D7115 CHANNEL  ; 热压C下层Hip测试气缸下降位延时设置
D7116 CHANNEL  ; 热压C上层有料感应延时设置
D7117 CHANNEL  ; 热压C下层有料感应延时设置
D7118 CHANNEL  ; #REF!
D7119 CHANNEL  ; #REF!
D7120 CHANNEL  ; 热压C上层极耳检查输入延时设置
D7121 CHANNEL  ; 热压C下层极耳检查输入延时设置
D7122 CHANNEL  ; 进出料转移伺服准备好延时设置
D7123 CHANNEL  ; 进出料转移伺服报警延时设置
D7124 CHANNEL  ; 伸缩伺服准备好延时设置
D7125 CHANNEL  ; 伸缩伺服报警延时设置
D7126 CHANNEL  ; #REF!
D7127 CHANNEL  ; 备用11延时设置
D7128 CHANNEL  ; 加热A跳闸延时设置
D7129 CHANNEL  ; 加热B跳闸延时设置
D7130 CHANNEL  ; 加热C跳闸延时设置
D7131 CHANNEL  ; 副PLC 0.03延时设置
D7132 CHANNEL  ; 副PLC 0.04延时设置
D7133 CHANNEL  ; 副PLC 0.05延时设置
D7134 CHANNEL  ; 副PLC 0.06延时设置
D7135 CHANNEL  ; 副PLC 0.07延时设置
D7136 CHANNEL  ; 副PLC 0.08延时设置
D7137 CHANNEL  ; 副PLC 0.09延时设置
D7138 CHANNEL  ; 副PLC 0.10延时设置
D7139 CHANNEL  ; 副PLC 0.11延时设置
D7140 CHANNEL  ; 延时设置
D7141 CHANNEL  ; 延时设置
D7142 CHANNEL  ; 延时设置
D7143 CHANNEL  ; 延时设置
D7144 CHANNEL  ; 副PLC 1.00延时设置
D7145 CHANNEL  ; 副PLC 1.01延时设置
D7146 CHANNEL  ; 副PLC 1.02延时设置
D7147 CHANNEL  ; 副PLC 1.03延时设置
D7148 CHANNEL  ; 副PLC 1.04延时设置
D7149 CHANNEL  ; 副PLC 1.05延时设置
D7150 CHANNEL  ; 副PLC 1.06延时设置
D7151 CHANNEL  ; 副PLC 1.07延时设置
D7152 CHANNEL  ; 副PLC 1.08延时设置
D7153 CHANNEL  ; 副PLC 1.09延时设置
D7154 CHANNEL  ; 副PLC 1.10延时设置
D7155 CHANNEL  ; 副PLC 1.11延时设置
D7156 CHANNEL  ; 延时设置
D7157 CHANNEL  ; 延时设置
D7158 CHANNEL  ; 延时设置
D7159 CHANNEL  ; 延时设置
D7160 CHANNEL  ; 延时设置
D7161 CHANNEL  ; 出料转移机构A上升位延时设置
D7162 CHANNEL  ; 出料转移夹爪A下降位延时设置
D7163 CHANNEL  ; 出料转移夹爪A上升位延时设置
D7164 CHANNEL  ; 出料转移夹爪A1松开位延时设置
D7165 CHANNEL  ; 出料转移夹爪A1夹紧位延时设置
D7166 CHANNEL  ; 出料转移夹爪A2松开位延时设置
D7167 CHANNEL  ; 出料转移夹爪A2夹紧位延时设置
D7168 CHANNEL  ; 出料转移夹爪A3松开位延时设置
D7169 CHANNEL  ; 出料转移夹爪A3夹紧位延时设置
D7170 CHANNEL  ; 出料转移夹爪A4松开位延时设置
D7171 CHANNEL  ; 出料转移夹爪A4夹紧位延时设置
D7174 CHANNEL  ; 出料转移夹爪A1左托起张开位延时设置
D7175 CHANNEL  ; 出料转移夹爪A1左托起托起位延时设置
D7176 CHANNEL  ; 出料转移夹爪A1右托起张开位延时设置
D7177 CHANNEL  ; 出料转移夹爪A1右托起托起位延时设置
D7178 CHANNEL  ; 出料转移夹爪A2左托起张开位延时设置
D7179 CHANNEL  ; 出料转移夹爪A2左托起托起位延时设置
D7180 CHANNEL  ; 出料转移夹爪A2右托起张开位延时设置
D7181 CHANNEL  ; 出料转移夹爪A2右托起托起位延时设置
D7182 CHANNEL  ; 出料转移夹爪A3左托起张开位延时设置
D7183 CHANNEL  ; 出料转移夹爪A3左托起托起位延时设置
D7184 CHANNEL  ; 出料转移夹爪A3右托起张开位延时设置
D7185 CHANNEL  ; 出料转移夹爪A3右托起托起位延时设置
D7186 CHANNEL  ; 出料转移夹爪A4左托起张开位延时设置
D7187 CHANNEL  ; 出料转移夹爪A4左托起托起位延时设置
D7188 CHANNEL  ; 出料转移夹爪A4右托起张开位延时设置
D7189 CHANNEL  ; 出料转移夹爪A4右托起托起位延时设置
D7194 CHANNEL  ; 出料转移夹爪A1真空延时设置
D7195 CHANNEL  ; 出料转移夹爪A2真空延时设置
D7196 CHANNEL  ; 出料转移夹爪A3真空延时设置
D7197 CHANNEL  ; 出料转移夹爪A4真空延时设置
D7199 CHANNEL  ; 进料转移机构B下降位延时设置
D7200 CHANNEL  ; 进料转移机构B上升位延时设置
D7201 CHANNEL  ; 进料转移夹爪B下降位延时设置
D7202 CHANNEL  ; 进料转移夹爪B上升位延时设置
D7203 CHANNEL  ; 进料转移夹爪B1松开位延时设置
D7204 CHANNEL  ; 进料转移夹爪B1夹紧位延时设置
D7205 CHANNEL  ; 进料转移夹爪B2松开位延时设置
D7206 CHANNEL  ; 进料转移夹爪B2夹紧位延时设置
D7207 CHANNEL  ; 进料转移夹爪B3松开位延时设置
D7208 CHANNEL  ; 进料转移夹爪B3夹紧位延时设置
D7209 CHANNEL  ; 进料转移夹爪B4松开位延时设置
D7210 CHANNEL  ; 进料转移夹爪B4夹紧位延时设置
D7213 CHANNEL  ; 进料转移爪B1左上升位延时设置
D7214 CHANNEL  ; 进料转移爪B1右上升位延时设置
D7215 CHANNEL  ; 进料转移爪B2左上升位延时设置
D7216 CHANNEL  ; 进料转移爪B2右上升位延时设置
D7217 CHANNEL  ; 进料转移爪B3左上升位延时设置
D7218 CHANNEL  ; 进料转移爪B3右上升位延时设置
D7219 CHANNEL  ; 进料转移爪B4左上升位延时设置
D7220 CHANNEL  ; 进料转移爪B4右上升位延时设置
D7223 CHANNEL  ; 进料转移爪B1中间上升位延时设置
D7224 CHANNEL  ; 进料转移爪B2中间上升位延时设置
D7225 CHANNEL  ; 进料转移爪B3中间上升位延时设置
D7226 CHANNEL  ; 进料转移爪B4中间上升位延时设置
D7228 CHANNEL  ; 进料转移爪B1有料反射延时设置
D7229 CHANNEL  ; 进料转移爪B2有料反射延时设置
D7230 CHANNEL  ; 进料转移爪B3有料反射延时设置
D7231 CHANNEL  ; 进料转移爪B4有料反射延时设置
D7233 CHANNEL  ; 出料转移机构B下降位延时设置
D7234 CHANNEL  ; 出料转移机构B上升位延时设置
D7235 CHANNEL  ; 出料转移夹爪B下降位延时设置
D7236 CHANNEL  ; 出料转移夹爪B上升位延时设置
D7237 CHANNEL  ; 出料转移夹爪B1松开位延时设置
D7238 CHANNEL  ; 出料转移夹爪B1夹紧位延时设置
D7239 CHANNEL  ; 出料转移夹爪B2松开位延时设置
D7240 CHANNEL  ; 出料转移夹爪B2夹紧位延时设置
D7241 CHANNEL  ; 出料转移夹爪B3松开位延时设置
D7242 CHANNEL  ; 出料转移夹爪B3夹紧位延时设置
D7243 CHANNEL  ; 出料转移夹爪B4松开位延时设置
D7244 CHANNEL  ; 出料转移夹爪B4夹紧位延时设置
D7247 CHANNEL  ; 出料转移夹爪B1左托起张开位延时设置
D7248 CHANNEL  ; 出料转移夹爪B1左托起托起位延时设置
D7249 CHANNEL  ; 出料转移夹爪B1右托起张开位延时设置
D7250 CHANNEL  ; 出料转移夹爪B1右托起托起位延时设置
D7251 CHANNEL  ; 出料转移夹爪B2左托起张开位延时设置
D7252 CHANNEL  ; 出料转移夹爪B2左托起托起位延时设置
D7253 CHANNEL  ; 出料转移夹爪B2右托起张开位延时设置
D7254 CHANNEL  ; 出料转移夹爪B2右托起托起位延时设置
D7255 CHANNEL  ; 出料转移夹爪B3左托起张开位延时设置
D7256 CHANNEL  ; 出料转移夹爪B3左托起托起位延时设置
D7257 CHANNEL  ; 出料转移夹爪B3右托起张开位延时设置
D7258 CHANNEL  ; 出料转移夹爪B3右托起托起位延时设置
D7259 CHANNEL  ; 出料转移夹爪B4左托起张开位延时设置
D7260 CHANNEL  ; 出料转移夹爪B4左托起托起位延时设置
D7261 CHANNEL  ; 出料转移夹爪B4右托起张开位延时设置
D7262 CHANNEL  ; 出料转移夹爪B4右托起托起位延时设置
D7267 CHANNEL  ; 出料转移夹爪B1真空延时设置
D7268 CHANNEL  ; 出料转移夹爪B2真空延时设置
D7269 CHANNEL  ; 出料转移夹爪B3真空延时设置
D7270 CHANNEL  ; 出料转移夹爪B4真空延时设置
D7272 CHANNEL  ; 热压A1层加热开关延时设置
D7273 CHANNEL  ; 热压A2层加热开关延时设置
D7274 CHANNEL  ; 热压A3层加热开关延时设置
D7275 CHANNEL  ; 热压A4层加热开关延时设置
D7276 CHANNEL  ; 热压A5层加热开关延时设置
D7277 CHANNEL  ; 热压A1下压板A侧位置延时设置
D7278 CHANNEL  ; 热压A1下压板B侧位置延时设置
D7281 CHANNEL  ; 热压A3下压板A侧位置延时设置
D7282 CHANNEL  ; 热压A3下压板B侧位置延时设置
D7283 CHANNEL  ; 热压A4下压板A侧位置延时设置
D7284 CHANNEL  ; 热压A4下压板B侧位置延时设置
D7285 CHANNEL  ; 热压A5下压板A侧位置延时设置
D7286 CHANNEL  ; 热压A5下压板B侧位置延时设置
D7287 CHANNEL  ; 热压A1有料对射延时设置
D7288 CHANNEL  ; 热压A2有料对射延时设置
D7289 CHANNEL  ; 热压A3有料对射延时设置
D7290 CHANNEL  ; 热压A4有料对射延时设置
D7291 CHANNEL  ; 热压A5有料对射延时设置
D7292 CHANNEL  ; 热压A上预压平移气缸等待位延时设置
D7293 CHANNEL  ; 热压A上预压平移气缸预压位延时设置
D7294 CHANNEL  ; 热压A下预压平移气缸等待位延时设置
D7295 CHANNEL  ; 热压A下预压平移气缸预压位延时设置
D7296 CHANNEL  ; 热压A垫高气缸移出位延时设置
D7297 CHANNEL  ; 热压A垫高气缸热压位延时设置
D7298 CHANNEL  ; 热压A1HIP测试上升位延时设置
D7299 CHANNEL  ; 热压A1HIP测试下降位延时设置
D7300 CHANNEL  ; 热压A2HIP测试上升位延时设置
D7301 CHANNEL  ; 热压A2HIP测试下降位延时设置
D7302 CHANNEL  ; 热压A3HIP测试上升位延时设置
D7303 CHANNEL  ; 热压A3HIP测试下降位延时设置
D7304 CHANNEL  ; 热压A4HIP测试上升位延时设置
D7305 CHANNEL  ; 热压A4HIP测试下降位延时设置
D7306 CHANNEL  ; 热压A5HIP测试上升位延时设置
D7307 CHANNEL  ; 热压A5HIP测试下降位延时设置
D7308 CHANNEL  ; 热压A1顶升气缸缩回位延时设置
D7309 CHANNEL  ; 热压A1顶升气缸伸出位延时设置
D7310 CHANNEL  ; 热压A2顶升气缸左缩回位延时设置
D7311 CHANNEL  ; 热压A2顶升气缸左伸出位延时设置
D7312 CHANNEL  ; 热压A2顶升气缸右缩回位延时设置
D7313 CHANNEL  ; 热压A2顶升气缸右伸出位延时设置
D7314 CHANNEL  ; 热压A3顶升气缸左缩回位延时设置
D7315 CHANNEL  ; 热压A3顶升气缸左伸出位延时设置
D7316 CHANNEL  ; 热压A3顶升气缸右缩回位延时设置
D7317 CHANNEL  ; 热压A3顶升气缸右伸出位延时设置
D7318 CHANNEL  ; 热压A4顶升气缸左缩回位延时设置
D7319 CHANNEL  ; 热压A4顶升气缸左伸出位延时设置
D7320 CHANNEL  ; 热压A4顶升气缸右缩回位延时设置
D7321 CHANNEL  ; 热压A4顶升气缸右伸出位延时设置
D7322 CHANNEL  ; 热压A5顶升气缸左缩回位延时设置
D7323 CHANNEL  ; 热压A5顶升气缸左伸出位延时设置
D7324 CHANNEL  ; 热压A5顶升气缸右缩回位延时设置
D7325 CHANNEL  ; 热压A5顶升气缸右伸出位延时设置
D7326 CHANNEL  ; 热压B1层加热开关延时设置
D7327 CHANNEL  ; 热压B2层加热开关延时设置
D7328 CHANNEL  ; 热压B3层加热开关延时设置
D7329 CHANNEL  ; 热压B4层加热开关延时设置
D7330 CHANNEL  ; 热压B5层加热开关延时设置
D7331 CHANNEL  ; 热压B1下压板A侧位置延时设置
D7332 CHANNEL  ; 热压B1下压板B侧位置延时设置
D7333 CHANNEL  ; 热压B2下压板A侧位置延时设置
D7334 CHANNEL  ; 热压B2下压板B侧位置延时设置
D7335 CHANNEL  ; 热压B3下压板A侧位置延时设置
D7336 CHANNEL  ; 热压B3下压板B侧位置延时设置
D7337 CHANNEL  ; 热压B4下压板A侧位置延时设置
D7338 CHANNEL  ; 热压B4下压板B侧位置延时设置
D7339 CHANNEL  ; 热压B5下压板A侧位置延时设置
D7340 CHANNEL  ; 热压B5下压板B侧位置延时设置
D7341 CHANNEL  ; 热压B1有料对射延时设置
D7342 CHANNEL  ; 热压B2有料对射延时设置
D7343 CHANNEL  ; 热压B3有料对射延时设置
D7344 CHANNEL  ; 热压B4有料对射延时设置
D7345 CHANNEL  ; 热压B5有料对射延时设置
D7346 CHANNEL  ; 热压B上预压平移气缸等待位延时设置
D7347 CHANNEL  ; 热压B上预压平移气缸预压位延时设置
D7348 CHANNEL  ; 热压B下预压平移气缸等待位延时设置
D7349 CHANNEL  ; 热压B下预压平移气缸预压位延时设置
D7350 CHANNEL  ; 热压B垫高气缸移出位延时设置
D7351 CHANNEL  ; 热压B垫高气缸热压位延时设置
D7352 CHANNEL  ; 热压B1HIP测试上升位延时设置
D7353 CHANNEL  ; 热压B1HIP测试下降位延时设置
D7354 CHANNEL  ; 热压B2HIP测试上升位延时设置
D7355 CHANNEL  ; 热压B2HIP测试下降位延时设置
D7356 CHANNEL  ; 热压B3HIP测试上升位延时设置
D7357 CHANNEL  ; 热压B3HIP测试下降位延时设置
D7358 CHANNEL  ; 热压B4HIP测试上升位延时设置
D7359 CHANNEL  ; 热压B4HIP测试下降位延时设置
D7360 CHANNEL  ; 热压B5HIP测试上升位延时设置
D7361 CHANNEL  ; 热压B5HIP测试下降位延时设置
D7362 CHANNEL  ; 热压B1顶升气缸缩回位延时设置
D7363 CHANNEL  ; 热压B1顶升气缸伸出位延时设置
D7364 CHANNEL  ; 热压B2顶升气缸左缩回位延时设置
D7365 CHANNEL  ; 热压B2顶升气缸左伸出位延时设置
D7366 CHANNEL  ; 热压B2顶升气缸右缩回位延时设置
D7367 CHANNEL  ; 热压B2顶升气缸右伸出位延时设置
D7368 CHANNEL  ; 热压B3顶升气缸左缩回位延时设置
D7369 CHANNEL  ; 热压B3顶升气缸左伸出位延时设置
D7370 CHANNEL  ; 热压B3顶升气缸右缩回位延时设置
D7371 CHANNEL  ; 热压B3顶升气缸右伸出位延时设置
D7372 CHANNEL  ; 热压B4顶升气缸左缩回位延时设置
D7373 CHANNEL  ; 热压B4顶升气缸左伸出位延时设置
D7374 CHANNEL  ; 热压B4顶升气缸右缩回位延时设置
D7375 CHANNEL  ; 热压B4顶升气缸右伸出位延时设置
D7376 CHANNEL  ; 热压B5顶升气缸左缩回位延时设置
D7377 CHANNEL  ; 热压B5顶升气缸左伸出位延时设置
D7378 CHANNEL  ; 热压B5顶升气缸右缩回位延时设置
D7379 CHANNEL  ; 热压B5顶升气缸右伸出位延时设置
D7380 CHANNEL  ; 下料定位A下降位延时设置
D7381 CHANNEL  ; 下料定位A上升位延时设置
D7382 CHANNEL  ; 下料定位A水平位延时设置
D7383 CHANNEL  ; 下料定位A垂直位延时设置
D7384 CHANNEL  ; 下料定位A1左右松开位延时设置
D7385 CHANNEL  ; 下料定位A1左右夹紧位延时设置
D7386 CHANNEL  ; 下料定位A2左右松开位延时设置
D7387 CHANNEL  ; 下料定位A2左右夹紧位延时设置
D7388 CHANNEL  ; 下料定位A3左右松开位延时设置
D7389 CHANNEL  ; 下料定位A3左右夹紧位延时设置
D7390 CHANNEL  ; 下料定位A4左右松开位延时设置
D7391 CHANNEL  ; 下料定位A4左右夹紧位延时设置
D7394 CHANNEL  ; 下料定位A1前后松开位延时设置
D7395 CHANNEL  ; 下料定位A1前后夹紧位延时设置
D7396 CHANNEL  ; 下料定位A2前后松开位延时设置
D7397 CHANNEL  ; 下料定位A2前后夹紧位延时设置
D7398 CHANNEL  ; 下料定位A3前后松开位延时设置
D7399 CHANNEL  ; 下料定位A3前后夹紧位延时设置
D7400 CHANNEL  ; 下料定位A4前后松开位延时设置
D7401 CHANNEL  ; 下料定位A4前后夹紧位延时设置
D7404 CHANNEL  ; 下料定位A1有料感应延时设置
D7405 CHANNEL  ; 下料定位A2有料感应延时设置
D7406 CHANNEL  ; 下料定位A3有料感应延时设置
D7407 CHANNEL  ; 下料定位A4有料感应延时设置
D7409 CHANNEL  ; 下料定位A料平整检测（预留）延时设置
D7410 CHANNEL  ; 下料定位B下降位延时设置
D7411 CHANNEL  ; 下料定位B上升位延时设置
D7412 CHANNEL  ; 下料定位B水平位延时设置
D7413 CHANNEL  ; 下料定位B垂直位延时设置
D7414 CHANNEL  ; 下料定位B1左右松开位延时设置
D7415 CHANNEL  ; 下料定位B1左右夹紧位延时设置
D7416 CHANNEL  ; 下料定位B2左右松开位延时设置
D7417 CHANNEL  ; 下料定位B2左右夹紧位延时设置
D7418 CHANNEL  ; 下料定位B3左右松开位延时设置
D7419 CHANNEL  ; 下料定位B3左右夹紧位延时设置
D7420 CHANNEL  ; 下料定位B4左右松开位延时设置
D7421 CHANNEL  ; 下料定位B4左右夹紧位延时设置
D7424 CHANNEL  ; 下料定位B1前后松开位延时设置
D7425 CHANNEL  ; 下料定位B1前后夹紧位延时设置
D7426 CHANNEL  ; 下料定位B2前后松开位延时设置
D7427 CHANNEL  ; 下料定位B2前后夹紧位延时设置
D7428 CHANNEL  ; 下料定位B3前后松开位延时设置
D7429 CHANNEL  ; 下料定位B3前后夹紧位延时设置
D7430 CHANNEL  ; 下料定位B4前后松开位延时设置
D7431 CHANNEL  ; 下料定位B4前后夹紧位延时设置
D7434 CHANNEL  ; 下料定位B1有料感应延时设置
D7435 CHANNEL  ; 下料定位B2有料感应延时设置
D7436 CHANNEL  ; 下料定位B3有料感应延时设置
D7437 CHANNEL  ; 下料定位B4有料感应延时设置
D7439 CHANNEL  ; 下料定位B料平整检测（预留）延时设置
D7440 CHANNEL  ; R2左夹紧气缸1松开位延时设置
D7441 CHANNEL  ; R2左夹紧气缸1夹紧位延时设置
D7442 CHANNEL  ; R2右夹紧气缸1松开位延时设置
D7443 CHANNEL  ; R2右夹紧气缸1夹紧位延时设置
D7444 CHANNEL  ; R2左夹紧气缸2松开位延时设置
D7445 CHANNEL  ; R2左夹紧气缸2夹紧位延时设置
D7446 CHANNEL  ; R2右夹紧气缸2松开位延时设置
D7447 CHANNEL  ; R2右夹紧气缸2夹紧位延时设置
D7448 CHANNEL  ; R2左夹紧气缸3松开位延时设置
D7449 CHANNEL  ; R2左夹紧气缸3夹紧位延时设置
D7450 CHANNEL  ; R2右夹紧气缸3松开位延时设置
D7451 CHANNEL  ; R2右夹紧气缸3夹紧位延时设置
D7452 CHANNEL  ; R2左夹紧气缸4松开位延时设置
D7453 CHANNEL  ; R2左夹紧气缸4夹紧位延时设置
D7454 CHANNEL  ; R2右夹紧气缸4松开位延时设置
D7455 CHANNEL  ; R2右夹紧气缸4夹紧位延时设置
D7460 CHANNEL  ; R2左压紧1上升位延时设置
D7461 CHANNEL  ; R2右压紧1上升位延时设置
D7462 CHANNEL  ; R2左压紧2上升位延时设置
D7463 CHANNEL  ; R2右压紧2上升位延时设置
D7464 CHANNEL  ; R2左压紧3上升位延时设置
D7465 CHANNEL  ; R2右压紧3上升位延时设置
D7466 CHANNEL  ; R2左压紧4上升位延时设置
D7467 CHANNEL  ; R2右压紧4上升位延时设置
D7470 CHANNEL  ; R2有料反射光电感应1延时设置
D7471 CHANNEL  ; R2有料反射光电感应2延时设置
D7472 CHANNEL  ; R2有料反射光电感应3延时设置
D7473 CHANNEL  ; R2有料反射光电感应4延时设置
D7475 CHANNEL  ; R2下料柔性报警1延时设置
D7476 CHANNEL  ; R2下料柔性报警2延时设置
D7477 CHANNEL  ; R2下料柔性报警3延时设置
D7478 CHANNEL  ; R2下料柔性报警4延时设置
D7480 CHANNEL  ; 下料R程序运行过程中延时设置
D7481 CHANNEL  ; 下料R程序复位中延时设置
D7482 CHANNEL  ; 下料R报警中延时设置
D7483 CHANNEL  ; 下料R位置辅助1延时设置
D7484 CHANNEL  ; 下料R位置辅助2延时设置
D7486 CHANNEL  ; 下料R位置辅助4延时设置
D7492 CHANNEL  ; 接料治具有料反射1延时设置
D7493 CHANNEL  ; 接料治具有料反射2延时设置
D7494 CHANNEL  ; 接料治具有料反射3延时设置
D7495 CHANNEL  ; 接料治具有料反射4延时设置
D7496 CHANNEL  ; 接料治具有料反射5延时设置
D7497 CHANNEL  ; 接料治具有料反射6延时设置
D7498 CHANNEL  ; 接料治具有料反射7延时设置
D7499 CHANNEL  ; 接料治具有料反射8延时设置
D7500 CHANNEL  ; 扫码NG有料对射光电1延时设置
D7501 CHANNEL  ; 扫码NG有料对射光电2延时设置
D7502 CHANNEL  ; 扫码NG有料对射光电3延时设置
D7503 CHANNEL  ; 扫码NG有料对射光电4延时设置
D7505 CHANNEL  ; 扫码NG满料对射光电延时设置
D7506 CHANNEL  ; 扫码NG拉带接近1延时设置
D7507 CHANNEL  ; 扫码NG拉带接近2延时设置
D7508 CHANNEL  ; HIPNG有料对射光电1延时设置
D7509 CHANNEL  ; HIPNG有料对射光电2延时设置
D7510 CHANNEL  ; HIPNG有料对射光电3延时设置
D7511 CHANNEL  ; HIPNG有料对射光电4延时设置
D7512 CHANNEL  ; HIPNG有料对射光电5延时设置
D7513 CHANNEL  ; HIPNG满料对射光电延时设置
D7514 CHANNEL  ; HIPNG拉带接近1延时设置
D7515 CHANNEL  ; HIPNG拉带接近2延时设置
D7516 CHANNEL  ; HIPNG有料对射光电1延时设置
D7517 CHANNEL  ; 工艺NG有料对射光电2延时设置
D7518 CHANNEL  ; 工艺NG有料对射光电3延时设置
D7519 CHANNEL  ; 工艺NG有料对射光电4延时设置
D7520 CHANNEL  ; 工艺NG有料对射光电5延时设置
D7521 CHANNEL  ; 工艺NG满料对射光电延时设置
D7522 CHANNEL  ; 工艺NG拉带接近1延时设置
D7523 CHANNEL  ; 工艺NG拉带接近2延时设置
D7572 CHANNEL  ; $?St$Bk?_#[466] / 接料伺服READY延时设置 / $?St$Bk?_#[466]
D7573 CHANNEL  ; $?St$Bk?_#[467] / 接料伺服报警延时设置 / $?St$Bk?_#[467]
D7610 CHANNEL  ; 备用(上料机器人)延时设置
D7611 CHANNEL  ; 机器人不在取料区域延时设置
D7612 CHANNEL  ; 机器人不在NG区域延时设置
D7613 CHANNEL  ; 机器人不在放料A区域延时设置
D8000 CHANNEL  ; 热压模组A上压板温度设定值
D8001 CHANNEL  ; 热压模组A下压板A温度设定值
D8002 CHANNEL  ; 热压模组A下压板B温度设定值
D8003 CHANNEL  ; 热压模组A侧压板温度设定值
D8005 CHANNEL  ; 热压模组B上压板温度设定值
D8006 CHANNEL  ; 热压模组B下压板A温度设定值
D8007 CHANNEL  ; 热压模组B下压板B温度设定值
D8008 CHANNEL  ; 热压模组B侧压板温度设定值
D8010 CHANNEL  ; 热压模组A第1层上压板左温度显示值
D8011 CHANNEL  ; 热压模组A第1层上压板中温度显示值
D8012 CHANNEL  ; 热压模组A第1层上压板右温度显示值
D8013 CHANNEL  ; 热压模组A第1层下压板A左温度显示值
D8014 CHANNEL  ; 热压模组A第1层下压板A中温度显示值
D8015 CHANNEL  ; 热压模组A第1层下压板A右温度显示值
D8016 CHANNEL  ; 热压模组A第1层下压板B左温度显示值
D8017 CHANNEL  ; 热压模组A第1层下压板B中温度显示值
D8018 CHANNEL  ; 热压模组A第1层下压板B右温度显示值
D8019 CHANNEL  ; 热压模组A第1层左侧压板温度显示值
D8020 CHANNEL  ; 热压模组A第1层右侧压板温度显示值
D8025 CHANNEL  ; 1#副PLC在线信号
D8030 CHANNEL  ; 热压模组A第2层上压板左温度显示值
D8031 CHANNEL  ; 热压模组A第2层上压板中温度显示值
D8032 CHANNEL  ; 热压模组A第2层上压板右温度显示值
D8033 CHANNEL  ; 热压模组A第2层下压板A左温度显示值
D8034 CHANNEL  ; 热压模组A第2层下压板A中温度显示值
D8035 CHANNEL  ; 热压模组A第2层下压板A右温度显示值
D8036 CHANNEL  ; 热压模组A第2层下压板B左温度显示值
D8037 CHANNEL  ; 热压模组A第2层下压板B中温度显示值
D8038 CHANNEL  ; 热压模组A第2层下压板B右温度显示值
D8039 CHANNEL  ; 热压模组A第2层左侧压板温度显示值
D8040 CHANNEL  ; 热压模组A第2层右侧压板温度显示值
D8050 CHANNEL  ; 热压模组A第3层上压板左温度显示值
D8051 CHANNEL  ; 热压模组A第3层上压板中温度显示值
D8052 CHANNEL  ; 热压模组A第3层上压板右温度显示值
D8053 CHANNEL  ; 热压模组A第3层下压板A左温度显示值
D8054 CHANNEL  ; 热压模组A第3层下压板A中温度显示值
D8055 CHANNEL  ; 热压模组A第3层下压板A右温度显示值
D8056 CHANNEL  ; 热压模组A第3层下压板B左温度显示值
D8057 CHANNEL  ; 热压模组A第3层下压板B中温度显示值
D8058 CHANNEL  ; 热压模组A第3层下压板B右温度显示值
D8059 CHANNEL  ; 热压模组A第3层左侧压板温度显示值
D8060 CHANNEL  ; 热压模组A第3层右侧压板温度显示值
D8070 CHANNEL  ; 热压模组A第4层上压板左温度显示值
D8071 CHANNEL  ; 热压模组A第4层上压板中温度显示值
D8072 CHANNEL  ; 热压模组A第4层上压板右温度显示值
D8073 CHANNEL  ; 热压模组A第4层下压板A左温度显示值
D8074 CHANNEL  ; 热压模组A第4层下压板A中温度显示值
D8075 CHANNEL  ; 热压模组A第4层下压板A右温度显示值
D8076 CHANNEL  ; 热压模组A第4层下压板B左温度显示值
D8077 CHANNEL  ; 热压模组A第4层下压板B中温度显示值
D8078 CHANNEL  ; 热压模组A第4层下压板B右温度显示值
D8079 CHANNEL  ; 热压模组A第4层左侧压板温度显示值
D8080 CHANNEL  ; 热压模组A第4层右侧压板温度显示值
D8090 CHANNEL  ; 热压模组A第5层上压板左温度显示值
D8091 CHANNEL  ; 热压模组A第5层上压板中温度显示值
D8092 CHANNEL  ; 热压模组A第5层上压板右温度显示值
D8093 CHANNEL  ; 热压模组A第5层下压板A左温度显示值
D8094 CHANNEL  ; 热压模组A第5层下压板A中温度显示值
D8095 CHANNEL  ; 热压模组A第5层下压板A右温度显示值
D8096 CHANNEL  ; 热压模组A第5层下压板B左温度显示值
D8097 CHANNEL  ; 热压模组A第5层下压板B中温度显示值
D8098 CHANNEL  ; 热压模组A第5层下压板B右温度显示值
D8099 CHANNEL  ; 热压模组A第5层左侧压板温度显示值
D8100 CHANNEL  ; 热压模组A第5层右侧压板温度显示值
D8110 CHANNEL  ; 热压模组B第1层上压板左温度显示值
D8111 CHANNEL  ; 热压模组B第1层上压板中温度显示值
D8112 CHANNEL  ; 热压模组B第1层上压板右温度显示值
D8113 CHANNEL  ; 热压模组B第1层下压板A左温度显示值
D8114 CHANNEL  ; 热压模组B第1层下压板A中温度显示值
D8115 CHANNEL  ; 热压模组B第1层下压板A右温度显示值
D8116 CHANNEL  ; 热压模组B第1层下压板B左温度显示值
D8117 CHANNEL  ; 热压模组B第1层下压板B中温度显示值
D8118 CHANNEL  ; 热压模组B第1层下压板B右温度显示值
D8119 CHANNEL  ; 热压模组B第1层左侧压板温度显示值
D8120 CHANNEL  ; 热压模组B第1层右侧压板温度显示值
D8125 CHANNEL  ; 2#副PLC在线信号
D8130 CHANNEL  ; 热压模组B第2层上压板左温度显示值
D8131 CHANNEL  ; 热压模组B第2层上压板中温度显示值
D8132 CHANNEL  ; 热压模组B第2层上压板右温度显示值
D8133 CHANNEL  ; 热压模组B第2层下压板A左温度显示值
D8134 CHANNEL  ; 热压模组B第2层下压板A中温度显示值
D8135 CHANNEL  ; 热压模组B第2层下压板A右温度显示值
D8136 CHANNEL  ; 热压模组B第2层下压板B左温度显示值
D8137 CHANNEL  ; 热压模组B第2层下压板B中温度显示值
D8138 CHANNEL  ; 热压模组B第2层下压板B右温度显示值
D8139 CHANNEL  ; 热压模组B第2层左侧压板温度显示值
D8140 CHANNEL  ; 热压模组B第2层右侧压板温度显示值
D8150 CHANNEL  ; 热压模组B第3层上压板左温度显示值
D8151 CHANNEL  ; 热压模组B第3层上压板中温度显示值
D8152 CHANNEL  ; 热压模组B第3层上压板右温度显示值
D8153 CHANNEL  ; 热压模组B第3层下压板A左温度显示值
D8154 CHANNEL  ; 热压模组B第3层下压板A中温度显示值
D8155 CHANNEL  ; 热压模组B第3层下压板A右温度显示值
D8156 CHANNEL  ; 热压模组B第3层下压板B左温度显示值
D8157 CHANNEL  ; 热压模组B第3层下压板B中温度显示值
D8158 CHANNEL  ; 热压模组B第3层下压板B右温度显示值
D8159 CHANNEL  ; 热压模组B第3层左侧压板温度显示值
D8160 CHANNEL  ; 热压模组B第3层右侧压板温度显示值
D8170 CHANNEL  ; 热压模组B第4层上压板左温度显示值
D8171 CHANNEL  ; 热压模组B第4层上压板中温度显示值
D8172 CHANNEL  ; 热压模组B第4层上压板右温度显示值
D8173 CHANNEL  ; 热压模组B第4层下压板A左温度显示值
D8174 CHANNEL  ; 热压模组B第4层下压板A中温度显示值
D8175 CHANNEL  ; 热压模组B第4层下压板A右温度显示值
D8176 CHANNEL  ; 热压模组B第4层下压板B左温度显示值
D8177 CHANNEL  ; 热压模组B第4层下压板B中温度显示值
D8178 CHANNEL  ; 热压模组B第4层下压板B右温度显示值
D8179 CHANNEL  ; 热压模组B第4层左侧压板温度显示值
D8180 CHANNEL  ; 热压模组B第4层右侧压板温度显示值
D8190 CHANNEL  ; 热压模组B第5层上压板左温度显示值
D8191 CHANNEL  ; 热压模组B第5层上压板中温度显示值
D8192 CHANNEL  ; 热压模组B第5层上压板右温度显示值
D8193 CHANNEL  ; 热压模组B第5层下压板A左温度显示值
D8194 CHANNEL  ; 热压模组B第5层下压板A中温度显示值
D8195 CHANNEL  ; 热压模组B第5层下压板A右温度显示值
D8196 CHANNEL  ; 热压模组B第5层下压板B左温度显示值
D8197 CHANNEL  ; 热压模组B第5层下压板B中温度显示值
D8198 CHANNEL  ; 热压模组B第5层下压板B右温度显示值
D8199 CHANNEL  ; 热压模组B第5层左侧压板温度显示值
D8200 CHANNEL  ; 热压模组B第5层右侧压板温度显示值
D8201 CHANNEL  ; 加热控制字
D8201.00 BOOL  ; A工位加热控制全部开始
D8201.01 BOOL  ; A工位加热控制全部停止
D8201.02 BOOL  ; B工位加热控制全部开始
D8201.03 BOOL  ; B工位加热控制全部停止
D8201.04 BOOL  ; A工位AT控制全部开始
D8201.05 BOOL  ; A工位AT控制全部停止
D8201.06 BOOL  ; B工位AT控制全部开始
D8201.07 BOOL  ; B工位AT控制全部停止
D8202.00 BOOL  ; 紧急停止信号(写入副PLC)
D8202.01 BOOL  ; 复位信号(写入副PLC)
D8210 CHANNEL  ; 热压模组A加热开始
D8210.00 BOOL  ; 热压模组A第1层上压板左加热开始
D8210.01 BOOL  ; 热压模组A第1层上压板中加热开始
D8210.02 BOOL  ; 热压模组A第1层上压板右加热开始
D8210.03 BOOL  ; 热压模组A第1层下压板A左加热开始
D8210.04 BOOL  ; 热压模组A第1层下压板A中加热开始
D8210.05 BOOL  ; 热压模组A第1层下压板A右加热开始
D8210.06 BOOL  ; 热压模组A第1层下压板B左加热开始
D8210.07 BOOL  ; 热压模组A第1层下压板B中加热开始
D8210.08 BOOL  ; 热压模组A第1层下压板B右加热开始
D8210.09 BOOL  ; 热压模组A第1层左侧压板加热开始
D8210.10 BOOL  ; 热压模组A第1层右侧压板加热开始
D8211 CHANNEL  ; 热压模组B加热开始
D8211.00 BOOL  ; 热压模组A第2层上压板左加热开始
D8211.01 BOOL  ; 热压模组A第2层上压板中加热开始
D8211.02 BOOL  ; 热压模组A第2层上压板右加热开始
D8211.03 BOOL  ; 热压模组A第2层下压板A左加热开始
D8211.04 BOOL  ; 热压模组A第2层下压板A中加热开始
D8211.05 BOOL  ; 热压模组A第2层下压板A右加热开始
D8211.06 BOOL  ; 热压模组A第2层下压板B左加热开始
D8211.07 BOOL  ; 热压模组A第2层下压板B中加热开始
D8211.08 BOOL  ; 热压模组A第2层下压板B右加热开始
D8211.09 BOOL  ; 热压模组A第2层左侧压板加热开始
D8211.10 BOOL  ; 热压模组A第2层右侧压板加热开始
D8212 CHANNEL  ; 热压模组C加热开始
D8212.00 BOOL  ; 热压模组A第3层上压板左加热开始
D8212.01 BOOL  ; 热压模组A第3层上压板中加热开始
D8212.02 BOOL  ; 热压模组A第3层上压板右加热开始
D8212.03 BOOL  ; 热压模组A第3层下压板A左加热开始
D8212.04 BOOL  ; 热压模组A第3层下压板A中加热开始
D8212.05 BOOL  ; 热压模组A第3层下压板A右加热开始
D8212.06 BOOL  ; 热压模组A第3层下压板B左加热开始
D8212.07 BOOL  ; 热压模组A第3层下压板B中加热开始
D8212.08 BOOL  ; 热压模组A第3层下压板B右加热开始
D8212.09 BOOL  ; 热压模组A第3层左侧压板加热开始
D8212.10 BOOL  ; 热压模组A第3层右侧压板加热开始
D8213 CHANNEL  ; 热压模组A第4层加热开始
D8213.00 BOOL  ; 热压模组A第4层上压板左加热开始
D8213.01 BOOL  ; 热压模组A第4层上压板中加热开始
D8213.02 BOOL  ; 热压模组A第4层上压板右加热开始
D8213.03 BOOL  ; 热压模组A第4层下压板A左加热开始
D8213.04 BOOL  ; 热压模组A第4层下压板A中加热开始
D8213.05 BOOL  ; 热压模组A第4层下压板A右加热开始
D8213.06 BOOL  ; 热压模组A第4层下压板B左加热开始
D8213.07 BOOL  ; 热压模组A第4层下压板B中加热开始
D8213.08 BOOL  ; 热压模组A第4层下压板B右加热开始
D8213.09 BOOL  ; 热压模组A第4层左侧压板加热开始
D8213.10 BOOL  ; 热压模组A第4层右侧压板加热开始
D8214 CHANNEL  ; 热压模组A第5层加热开始
D8214.00 BOOL  ; 热压模组A第5层上压板左加热开始
D8214.01 BOOL  ; 热压模组A第5层上压板中加热开始
D8214.02 BOOL  ; 热压模组A第5层上压板右加热开始
D8214.03 BOOL  ; 热压模组A第5层下压板A左加热开始
D8214.04 BOOL  ; 热压模组A第5层下压板A中加热开始
D8214.05 BOOL  ; 热压模组A第5层下压板A右加热开始
D8214.06 BOOL  ; 热压模组A第5层下压板B左加热开始
D8214.07 BOOL  ; 热压模组A第5层下压板B中加热开始
D8214.08 BOOL  ; 热压模组A第5层下压板B右加热开始
D8214.09 BOOL  ; 热压模组A第5层左侧压板加热开始
D8214.10 BOOL  ; 热压模组A第5层右侧压板加热开始
D8215 CHANNEL  ; 热压模组B第1层加热开始
D8215.00 BOOL  ; 热压模组B第1层上压板左加热开始
D8215.01 BOOL  ; 热压模组B第1层上压板中加热开始
D8215.02 BOOL  ; 热压模组B第1层上压板右加热开始
D8215.03 BOOL  ; 热压模组B第1层下压板A左加热开始
D8215.04 BOOL  ; 热压模组B第1层下压板A中加热开始
D8215.05 BOOL  ; 热压模组B第1层下压板A右加热开始
D8215.06 BOOL  ; 热压模组B第1层下压板B左加热开始
D8215.07 BOOL  ; 热压模组B第1层下压板B中加热开始
D8215.08 BOOL  ; 热压模组B第1层下压板B右加热开始
D8215.09 BOOL  ; 热压模组B第1层左侧压板加热开始
D8215.10 BOOL  ; 热压模组B第1层右侧压板加热开始
D8216 CHANNEL  ; 热压模组B第2层加热开始
D8216.00 BOOL  ; 热压模组B第2层上压板左加热开始
D8216.01 BOOL  ; 热压模组B第2层上压板中加热开始
D8216.02 BOOL  ; 热压模组B第2层上压板右加热开始
D8216.03 BOOL  ; 热压模组B第2层下压板A左加热开始
D8216.04 BOOL  ; 热压模组B第2层下压板A中加热开始
D8216.05 BOOL  ; 热压模组B第2层下压板A右加热开始
D8216.06 BOOL  ; 热压模组B第2层下压板B左加热开始
D8216.07 BOOL  ; 热压模组B第2层下压板B中加热开始
D8216.08 BOOL  ; 热压模组B第2层下压板B右加热开始
D8216.09 BOOL  ; 热压模组B第2层左侧压板加热开始
D8216.10 BOOL  ; 热压模组B第2层右侧压板加热开始
D8217 CHANNEL  ; 热压模组B第3层加热开始
D8217.00 BOOL  ; 热压模组B第3层上压板左加热开始
D8217.01 BOOL  ; 热压模组B第3层上压板中加热开始
D8217.02 BOOL  ; 热压模组B第3层上压板右加热开始
D8217.03 BOOL  ; 热压模组B第3层下压板A左加热开始
D8217.04 BOOL  ; 热压模组B第3层下压板A中加热开始
D8217.05 BOOL  ; 热压模组B第3层下压板A右加热开始
D8217.06 BOOL  ; 热压模组B第3层下压板B左加热开始
D8217.07 BOOL  ; 热压模组B第3层下压板B中加热开始
D8217.08 BOOL  ; 热压模组B第3层下压板B右加热开始
D8217.09 BOOL  ; 热压模组B第3层左侧压板加热开始
D8217.10 BOOL  ; 热压模组B第3层右侧压板加热开始
D8218 CHANNEL  ; 热压模组B第4层加热开始
D8218.00 BOOL  ; 热压模组B第4层上压板左加热开始
D8218.01 BOOL  ; 热压模组B第4层上压板中加热开始
D8218.02 BOOL  ; 热压模组B第4层上压板右加热开始
D8218.03 BOOL  ; 热压模组B第4层下压板A左加热开始
D8218.04 BOOL  ; 热压模组B第4层下压板A中加热开始
D8218.05 BOOL  ; 热压模组B第4层下压板A右加热开始
D8218.06 BOOL  ; 热压模组B第4层下压板B左加热开始
D8218.07 BOOL  ; 热压模组B第4层下压板B中加热开始
D8218.08 BOOL  ; 热压模组B第4层下压板B右加热开始
D8218.09 BOOL  ; 热压模组B第4层左侧压板加热开始
D8218.10 BOOL  ; 热压模组B第4层右侧压板加热开始
D8219 CHANNEL  ; 热压模组B第5层加热开始
D8219.00 BOOL  ; 热压模组B第5层上压板左加热开始
D8219.01 BOOL  ; 热压模组B第5层上压板中加热开始
D8219.02 BOOL  ; 热压模组B第5层上压板右加热开始
D8219.03 BOOL  ; 热压模组B第5层下压板A左加热开始
D8219.04 BOOL  ; 热压模组B第5层下压板A中加热开始
D8219.05 BOOL  ; 热压模组B第5层下压板A右加热开始
D8219.06 BOOL  ; 热压模组B第5层下压板B左加热开始
D8219.07 BOOL  ; 热压模组B第5层下压板B中加热开始
D8219.08 BOOL  ; 热压模组B第5层下压板B右加热开始
D8219.09 BOOL  ; 热压模组B第5层左侧压板加热开始
D8219.10 BOOL  ; 热压模组B第5层右侧压板加热开始
D8220 CHANNEL  ; 热压模组A第1层温度自整定开始
D8220.00 BOOL  ; 热压模组A第1层上压板左温度自整定开始
D8220.01 BOOL  ; 热压模组A第1层上压板中温度自整定开始
D8220.02 BOOL  ; 热压模组A第1层上压板右温度自整定开始
D8220.03 BOOL  ; 热压模组A第1层下压板A左温度自整定开始
D8220.04 BOOL  ; 热压模组A第1层下压板A中温度自整定开始
D8220.05 BOOL  ; 热压模组A第1层下压板A右温度自整定开始
D8220.06 BOOL  ; 热压模组A第1层下压板B左温度自整定开始
D8220.07 BOOL  ; 热压模组A第1层下压板B中温度自整定开始
D8220.08 BOOL  ; 热压模组A第1层下压板B右温度自整定开始
D8220.09 BOOL  ; 热压模组A第1层左侧压板温度自整定开始
D8220.10 BOOL  ; 热压模组A第1层右侧压板温度自整定开始
D8221 CHANNEL  ; 热压模组A第2层温度自整定开始
D8221.00 BOOL  ; 热压模组A第2层上压板左温度自整定开始
D8221.01 BOOL  ; 热压模组A第2层上压板中温度自整定开始
D8221.02 BOOL  ; 热压模组A第2层上压板右温度自整定开始
D8221.03 BOOL  ; 热压模组A第2层下压板A左温度自整定开始
D8221.04 BOOL  ; 热压模组A第2层下压板A中温度自整定开始
D8221.05 BOOL  ; 热压模组A第2层下压板A右温度自整定开始
D8221.06 BOOL  ; 热压模组A第2层下压板B左温度自整定开始
D8221.07 BOOL  ; 热压模组A第2层下压板B中温度自整定开始
D8221.08 BOOL  ; 热压模组A第2层下压板B右温度自整定开始
D8221.09 BOOL  ; 热压模组A第2层左侧压板温度自整定开始
D8221.10 BOOL  ; 热压模组A第2层右侧压板温度自整定开始
D8222 CHANNEL  ; 热压模组A第3层温度自整定开始
D8222.00 BOOL  ; 热压模组A第3层上压板左温度自整定开始
D8222.01 BOOL  ; 热压模组A第3层上压板中温度自整定开始
D8222.02 BOOL  ; 热压模组A第3层上压板右温度自整定开始
D8222.03 BOOL  ; 热压模组A第3层下压板A左温度自整定开始
D8222.04 BOOL  ; 热压模组A第3层下压板A中温度自整定开始
D8222.05 BOOL  ; 热压模组A第3层下压板A右温度自整定开始
D8222.06 BOOL  ; 热压模组A第3层下压板B左温度自整定开始
D8222.07 BOOL  ; 热压模组A第3层下压板B中温度自整定开始
D8222.08 BOOL  ; 热压模组A第3层下压板B右温度自整定开始
D8222.09 BOOL  ; 热压模组A第3层左侧压板温度自整定开始
D8222.10 BOOL  ; 热压模组A第3层右侧压板温度自整定开始
D8223 CHANNEL  ; 热压模组A第4层温度自整定开始
D8223.00 BOOL  ; 热压模组A第4层上压板左温度自整定开始
D8223.01 BOOL  ; 热压模组A第4层上压板中温度自整定开始
D8223.02 BOOL  ; 热压模组A第4层上压板右温度自整定开始
D8223.03 BOOL  ; 热压模组A第4层下压板A左温度自整定开始
D8223.04 BOOL  ; 热压模组A第4层下压板A中温度自整定开始
D8223.05 BOOL  ; 热压模组A第4层下压板A右温度自整定开始
D8223.06 BOOL  ; 热压模组A第4层下压板B左温度自整定开始
D8223.07 BOOL  ; 热压模组A第4层下压板B中温度自整定开始
D8223.08 BOOL  ; 热压模组A第4层下压板B右温度自整定开始
D8223.09 BOOL  ; 热压模组A第4层左侧压板温度自整定开始
D8223.10 BOOL  ; 热压模组A第4层右侧压板温度自整定开始
D8224 CHANNEL  ; 热压模组A温度自整定停止
D8224.00 BOOL  ; 热压模组A第5层上压板左温度自整定开始
D8224.01 BOOL  ; 热压模组A第5层上压板中温度自整定开始
D8224.02 BOOL  ; 热压模组A第5层上压板右温度自整定开始
D8224.03 BOOL  ; 热压模组A第5层下压板A左温度自整定开始
D8224.04 BOOL  ; 热压模组A第5层下压板A中温度自整定开始
D8224.05 BOOL  ; 热压模组A第5层下压板A右温度自整定开始
D8224.06 BOOL  ; 热压模组A第5层下压板B左温度自整定开始
D8224.07 BOOL  ; 热压模组A第5层下压板B中温度自整定开始
D8224.08 BOOL  ; 热压模组A第5层下压板B右温度自整定开始
D8224.09 BOOL  ; 热压模组A第5层左侧压板温度自整定开始
D8224.10 BOOL  ; 热压模组A第5层右侧压板温度自整定开始
D8225 CHANNEL  ; 热压模组B温度自整定停止
D8225.00 BOOL  ; 热压模组B第1层上压板左温度自整定开始
D8225.01 BOOL  ; 热压模组B第1层上压板中温度自整定开始
D8225.02 BOOL  ; 热压模组B第1层上压板右温度自整定开始
D8225.03 BOOL  ; 热压模组B第1层下压板A左温度自整定开始
D8225.04 BOOL  ; 热压模组B第1层下压板A中温度自整定开始
D8225.05 BOOL  ; 热压模组B第1层下压板A右温度自整定开始
D8225.06 BOOL  ; 热压模组B第1层下压板B左温度自整定开始
D8225.07 BOOL  ; 热压模组B第1层下压板B中温度自整定开始
D8225.08 BOOL  ; 热压模组B第1层下压板B右温度自整定开始
D8225.09 BOOL  ; 热压模组B第1层左侧压板温度自整定开始
D8225.10 BOOL  ; 热压模组B第1层右侧压板温度自整定开始
D8226 CHANNEL  ; 热压模组C温度自整定停止
D8226.00 BOOL  ; 热压模组B第2层上压板左温度自整定开始
D8226.01 BOOL  ; 热压模组B第2层上压板中温度自整定开始
D8226.02 BOOL  ; 热压模组B第2层上压板右温度自整定开始
D8226.03 BOOL  ; 热压模组B第2层下压板A左温度自整定开始
D8226.04 BOOL  ; 热压模组B第2层下压板A中温度自整定开始
D8226.05 BOOL  ; 热压模组B第2层下压板A右温度自整定开始
D8226.06 BOOL  ; 热压模组B第2层下压板B左温度自整定开始
D8226.07 BOOL  ; 热压模组B第2层下压板B中温度自整定开始
D8226.08 BOOL  ; 热压模组B第2层下压板B右温度自整定开始
D8226.09 BOOL  ; 热压模组B第2层左侧压板温度自整定开始
D8226.10 BOOL  ; 热压模组B第2层右侧压板温度自整定开始
D8227 CHANNEL  ; 热压模组B第3层温度自整定开始
D8227.00 BOOL  ; 热压模组B第3层上压板左温度自整定开始
D8227.01 BOOL  ; 热压模组B第3层上压板中温度自整定开始
D8227.02 BOOL  ; 热压模组B第3层上压板右温度自整定开始
D8227.03 BOOL  ; 热压模组B第3层下压板A左温度自整定开始
D8227.04 BOOL  ; 热压模组B第3层下压板A中温度自整定开始
D8227.05 BOOL  ; 热压模组B第3层下压板A右温度自整定开始
D8227.06 BOOL  ; 热压模组B第3层下压板B左温度自整定开始
D8227.07 BOOL  ; 热压模组B第3层下压板B中温度自整定开始
D8227.08 BOOL  ; 热压模组B第3层下压板B右温度自整定开始
D8227.09 BOOL  ; 热压模组B第3层左侧压板温度自整定开始
D8227.10 BOOL  ; 热压模组B第3层右侧压板温度自整定开始
D8228 CHANNEL  ; 热压模组B第4层温度自整定开始
D8228.00 BOOL  ; 热压模组B第4层上压板左温度自整定开始
D8228.01 BOOL  ; 热压模组B第4层上压板中温度自整定开始
D8228.02 BOOL  ; 热压模组B第4层上压板右温度自整定开始
D8228.03 BOOL  ; 热压模组B第4层下压板A左温度自整定开始
D8228.04 BOOL  ; 热压模组B第4层下压板A中温度自整定开始
D8228.05 BOOL  ; 热压模组B第4层下压板A右温度自整定开始
D8228.06 BOOL  ; 热压模组B第4层下压板B左温度自整定开始
D8228.07 BOOL  ; 热压模组B第4层下压板B中温度自整定开始
D8228.08 BOOL  ; 热压模组B第4层下压板B右温度自整定开始
D8228.09 BOOL  ; 热压模组B第4层左侧压板温度自整定开始
D8228.10 BOOL  ; 热压模组B第4层右侧压板温度自整定开始
D8229 CHANNEL  ; 热压模组B第5层温度自整定开始
D8229.00 BOOL  ; 热压模组B第5层上压板左温度自整定开始
D8229.01 BOOL  ; 热压模组B第5层上压板中温度自整定开始
D8229.02 BOOL  ; 热压模组B第5层上压板右温度自整定开始
D8229.03 BOOL  ; 热压模组B第5层下压板A左温度自整定开始
D8229.04 BOOL  ; 热压模组B第5层下压板A中温度自整定开始
D8229.05 BOOL  ; 热压模组B第5层下压板A右温度自整定开始
D8229.06 BOOL  ; 热压模组B第5层下压板B左温度自整定开始
D8229.07 BOOL  ; 热压模组B第5层下压板B中温度自整定开始
D8229.08 BOOL  ; 热压模组B第5层下压板B右温度自整定开始
D8229.09 BOOL  ; 热压模组B第5层左侧压板温度自整定开始
D8229.10 BOOL  ; 热压模组B第5层右侧压板温度自整定开始
D8230 CHANNEL  ; 热压模组A第1层温度自整定状态
D8230.00 BOOL  ; 热压模组A第1层上压板左温度自整定中
D8230.01 BOOL  ; 热压模组A第1层上压板中温度自整定中
D8230.02 BOOL  ; 热压模组A第1层上压板右温度自整定中
D8230.03 BOOL  ; 热压模组A第1层下压板A左温度自整定中
D8230.04 BOOL  ; 热压模组A第1层下压板A中温度自整定中
D8230.05 BOOL  ; 热压模组A第1层下压板A右温度自整定中
D8230.06 BOOL  ; 热压模组A第1层下压板B左温度自整定中
D8230.07 BOOL  ; 热压模组A第1层下压板B中温度自整定中
D8230.08 BOOL  ; 热压模组A第1层下压板B右温度自整定中
D8230.09 BOOL  ; 热压模组A第1层左侧压板温度自整定中
D8230.10 BOOL  ; 热压模组A第1层右侧压板温度自整定中
D8231 CHANNEL  ; 热压模组A第2层温度自整定状态
D8231.00 BOOL  ; 热压模组A第2层上压板左温度自整定中
D8231.01 BOOL  ; 热压模组A第2层上压板中温度自整定中
D8231.02 BOOL  ; 热压模组A第2层上压板右温度自整定中
D8231.03 BOOL  ; 热压模组A第2层下压板A左温度自整定中
D8231.04 BOOL  ; 热压模组A第2层下压板A中温度自整定中
D8231.05 BOOL  ; 热压模组A第2层下压板A右温度自整定中
D8231.06 BOOL  ; 热压模组A第2层下压板B左温度自整定中
D8231.07 BOOL  ; 热压模组A第2层下压板B中温度自整定中
D8231.08 BOOL  ; 热压模组A第2层下压板B右温度自整定中
D8231.09 BOOL  ; 热压模组A第2层左侧压板温度自整定中
D8231.10 BOOL  ; 热压模组A第2层右侧压板温度自整定中
D8232 CHANNEL  ; 热压模组A第3层温度自整定状态
D8232.00 BOOL  ; 热压模组A第3层上压板左温度自整定中
D8232.01 BOOL  ; 热压模组A第3层上压板中温度自整定中
D8232.02 BOOL  ; 热压模组A第3层上压板右温度自整定中
D8232.03 BOOL  ; 热压模组A第3层下压板A左温度自整定中
D8232.04 BOOL  ; 热压模组A第3层下压板A中温度自整定中
D8232.05 BOOL  ; 热压模组A第3层下压板A右温度自整定中
D8232.06 BOOL  ; 热压模组A第3层下压板B左温度自整定中
D8232.07 BOOL  ; 热压模组A第3层下压板B中温度自整定中
D8232.08 BOOL  ; 热压模组A第3层下压板B右温度自整定中
D8232.09 BOOL  ; 热压模组A第3层左侧压板温度自整定中
D8232.10 BOOL  ; 热压模组A第3层右侧压板温度自整定中
D8233 CHANNEL  ; 热压模组A第4层温度自整定状态
D8233.00 BOOL  ; 热压模组A第4层上压板左温度自整定中
D8233.01 BOOL  ; 热压模组A第4层上压板中温度自整定中
D8233.02 BOOL  ; 热压模组A第4层上压板右温度自整定中
D8233.03 BOOL  ; 热压模组A第4层下压板A左温度自整定中
D8233.04 BOOL  ; 热压模组A第4层下压板A中温度自整定中
D8233.05 BOOL  ; 热压模组A第4层下压板A右温度自整定中
D8233.06 BOOL  ; 热压模组A第4层下压板B左温度自整定中
D8233.07 BOOL  ; 热压模组A第4层下压板B中温度自整定中
D8233.08 BOOL  ; 热压模组A第4层下压板B右温度自整定中
D8233.09 BOOL  ; 热压模组A第4层左侧压板温度自整定中
D8233.10 BOOL  ; 热压模组A第4层右侧压板温度自整定中
D8234 CHANNEL  ; 热压模组A第5层温度自整定状态
D8234.00 BOOL  ; 热压模组A第5层上压板左温度自整定中
D8234.01 BOOL  ; 热压模组A第5层上压板中温度自整定中
D8234.02 BOOL  ; 热压模组A第5层上压板右温度自整定中
D8234.03 BOOL  ; 热压模组A第5层下压板A左温度自整定中
D8234.04 BOOL  ; 热压模组A第5层下压板A中温度自整定中
D8234.05 BOOL  ; 热压模组A第5层下压板A右温度自整定中
D8234.06 BOOL  ; 热压模组A第5层下压板B左温度自整定中
D8234.07 BOOL  ; 热压模组A第5层下压板B中温度自整定中
D8234.08 BOOL  ; 热压模组A第5层下压板B右温度自整定中
D8234.09 BOOL  ; 热压模组A第5层左侧压板温度自整定中
D8234.10 BOOL  ; 热压模组A第5层右侧压板温度自整定中
D8235 CHANNEL  ; 热压模组B第1层温度自整定中状态
D8235.00 BOOL  ; 热压模组B第1层上压板左温度自整定中
D8235.01 BOOL  ; 热压模组B第1层上压板中温度自整定中
D8235.02 BOOL  ; 热压模组B第1层上压板右温度自整定中
D8235.03 BOOL  ; 热压模组B第1层下压板A左温度自整定中
D8235.04 BOOL  ; 热压模组B第1层下压板A中温度自整定中
D8235.05 BOOL  ; 热压模组B第1层下压板A右温度自整定中
D8235.06 BOOL  ; 热压模组B第1层下压板B左温度自整定中
D8235.07 BOOL  ; 热压模组B第1层下压板B中温度自整定中
D8235.08 BOOL  ; 热压模组B第1层下压板B右温度自整定中
D8235.09 BOOL  ; 热压模组B第1层左侧压板温度自整定中
D8235.10 BOOL  ; 热压模组B第1层右侧压板温度自整定中
D8236 CHANNEL  ; 热压模组B第2层温度自整定中状态
D8236.00 BOOL  ; 热压模组B第2层上压板左温度自整定中
D8236.01 BOOL  ; 热压模组B第2层上压板中温度自整定中
D8236.02 BOOL  ; 热压模组B第2层上压板右温度自整定中
D8236.03 BOOL  ; 热压模组B第2层下压板A左温度自整定中
D8236.04 BOOL  ; 热压模组B第2层下压板A中温度自整定中
D8236.05 BOOL  ; 热压模组B第2层下压板A右温度自整定中
D8236.06 BOOL  ; 热压模组B第2层下压板B左温度自整定中
D8236.07 BOOL  ; 热压模组B第2层下压板B中温度自整定中
D8236.08 BOOL  ; 热压模组B第2层下压板B右温度自整定中
D8236.09 BOOL  ; 热压模组B第2层左侧压板温度自整定中
D8236.10 BOOL  ; 热压模组B第2层右侧压板温度自整定中
D8237 CHANNEL  ; 热压模组B第3层温度自整定中状态
D8237.00 BOOL  ; 热压模组B第3层上压板左温度自整定中
D8237.01 BOOL  ; 热压模组B第3层上压板中温度自整定中
D8237.02 BOOL  ; 热压模组B第3层上压板右温度自整定中
D8237.03 BOOL  ; 热压模组B第3层下压板A左温度自整定中
D8237.04 BOOL  ; 热压模组B第3层下压板A中温度自整定中
D8237.05 BOOL  ; 热压模组B第3层下压板A右温度自整定中
D8237.06 BOOL  ; 热压模组B第3层下压板B左温度自整定中
D8237.07 BOOL  ; 热压模组B第3层下压板B中温度自整定中
D8237.08 BOOL  ; 热压模组B第3层下压板B右温度自整定中
D8237.09 BOOL  ; 热压模组B第3层左侧压板温度自整定中
D8237.10 BOOL  ; 热压模组B第3层右侧压板温度自整定中
D8238 CHANNEL  ; 热压模组B第4层温度自整定中状态
D8238.00 BOOL  ; 热压模组B第4层上压板左温度自整定中
D8238.01 BOOL  ; 热压模组B第4层上压板中温度自整定中
D8238.02 BOOL  ; 热压模组B第4层上压板右温度自整定中
D8238.03 BOOL  ; 热压模组B第4层下压板A左温度自整定中
D8238.04 BOOL  ; 热压模组B第4层下压板A中温度自整定中
D8238.05 BOOL  ; 热压模组B第4层下压板A右温度自整定中
D8238.06 BOOL  ; 热压模组B第4层下压板B左温度自整定中
D8238.07 BOOL  ; 热压模组B第4层下压板B中温度自整定中
D8238.08 BOOL  ; 热压模组B第4层下压板B右温度自整定中
D8238.09 BOOL  ; 热压模组B第4层左侧压板温度自整定中
D8238.10 BOOL  ; 热压模组B第4层右侧压板温度自整定中
D8239 CHANNEL  ; 热压模组B第5层温度自整定中状态
D8239.00 BOOL  ; 热压模组B第5层上压板左温度自整定中
D8239.01 BOOL  ; 热压模组B第5层上压板中温度自整定中
D8239.02 BOOL  ; 热压模组B第5层上压板右温度自整定中
D8239.03 BOOL  ; 热压模组B第5层下压板A左温度自整定中
D8239.04 BOOL  ; 热压模组B第5层下压板A中温度自整定中
D8239.05 BOOL  ; 热压模组B第5层下压板A右温度自整定中
D8239.06 BOOL  ; 热压模组B第5层下压板B左温度自整定中
D8239.07 BOOL  ; 热压模组B第5层下压板B中温度自整定中
D8239.08 BOOL  ; 热压模组B第5层下压板B右温度自整定中
D8239.09 BOOL  ; 热压模组B第5层左侧压板温度自整定中
D8239.10 BOOL  ; 热压模组B第5层右侧压板温度自整定中
D8240 CHANNEL  ; 热压模组A1-4层报警
D8240.00 BOOL  ; 热压模组A第1层上压板左温度传感器断线
D8240.01 BOOL  ; 热压模组A第1层上压板左温度超过保护设定范围
D8240.02 BOOL  ; 热压模组A第1层上压板左温度超限NG
D8240.03 BOOL  ; 热压模组A第1层上压板中温度传感器断线
D8240.04 BOOL  ; 热压模组A第1层上压板中温度超过保护设定范围
D8240.05 BOOL  ; 热压模组A第1层上压板中温度超限NG
D8240.06 BOOL  ; 热压模组A第1层上压板右温度传感器断线
D8240.07 BOOL  ; 热压模组A第1层上压板右温度超过保护设定范围
D8240.08 BOOL  ; 热压模组A第1层上压板右温度超限NG
D8240.09 BOOL  ; 热压模组A第1层下压板A左温度传感器断线
D8240.10 BOOL  ; 热压模组A第1层下压板A左温度超过保护设定范围
D8240.11 BOOL  ; 热压模组A第1层下压板A左温度超限NG
D8240.12 BOOL  ; 热压模组A第1层下压板A中温度传感器断线
D8240.13 BOOL  ; 热压模组A第1层下压板A中温度超过保护设定范围
D8240.14 BOOL  ; 热压模组A第1层下压板A中温度超限NG
D8240.15 BOOL  ; 热压模组A第1层下压板A右温度传感器断线
D8241 CHANNEL  ; 热压模组A1-4层报警
D8241.00 BOOL  ; 热压模组A第1层下压板A右温度超过保护设定范围
D8241.01 BOOL  ; 热压模组A第1层下压板A右温度超限NG
D8241.02 BOOL  ; 热压模组A第1层下压板B左温度传感器断线
D8241.03 BOOL  ; 热压模组A第1层下压板B左温度超过保护设定范围
D8241.04 BOOL  ; 热压模组A第1层下压板B左温度超限NG
D8241.05 BOOL  ; 热压模组A第1层下压板B中温度传感器断线
D8241.06 BOOL  ; 热压模组A第1层下压板B中温度超过保护设定范围
D8241.07 BOOL  ; 热压模组A第1层下压板B中温度超限NG
D8241.08 BOOL  ; 热压模组A第1层下压板B右温度传感器断线
D8241.09 BOOL  ; 热压模组A第1层下压板B右温度超过保护设定范围
D8241.10 BOOL  ; 热压模组A第1层下压板B右温度超限NG
D8241.11 BOOL  ; 热压模组A第1层左侧压板温度传感器断线
D8241.12 BOOL  ; 热压模组A第1层左侧压板温度超过保护设定范围
D8241.13 BOOL  ; 热压模组A第1层左侧压板温度超限NG
D8241.14 BOOL  ; 热压模组A第1层右侧压板温度传感器断线
D8241.15 BOOL  ; 热压模组A第1层右侧压板温度超过保护设定范围
D8242 CHANNEL  ; 热压模组A1-4层报警
D8242.00 BOOL  ; 热压模组A第2层上压板左温度传感器断线
D8242.01 BOOL  ; 热压模组A第2层上压板左温度超过保护设定范围
D8242.02 BOOL  ; 热压模组A第2层上压板左温度超限NG
D8242.03 BOOL  ; 热压模组A第2层上压板中温度传感器断线
D8242.04 BOOL  ; 热压模组A第2层上压板中温度超过保护设定范围
D8242.05 BOOL  ; 热压模组A第2层上压板中温度超限NG
D8242.06 BOOL  ; 热压模组A第2层上压板右温度传感器断线
D8242.07 BOOL  ; 热压模组A第2层上压板右温度超过保护设定范围
D8242.08 BOOL  ; 热压模组A第2层上压板右温度超限NG
D8242.09 BOOL  ; 热压模组A第2层下压板A左温度传感器断线
D8242.10 BOOL  ; 热压模组A第2层下压板A左温度超过保护设定范围
D8242.11 BOOL  ; 热压模组A第2层下压板A左温度超限NG
D8242.12 BOOL  ; 热压模组A第2层下压板A中温度传感器断线
D8242.13 BOOL  ; 热压模组A第2层下压板A中温度超过保护设定范围
D8242.14 BOOL  ; 热压模组A第2层下压板A中温度超限NG
D8242.15 BOOL  ; 热压模组A第2层下压板A右温度传感器断线
D8243 CHANNEL  ; 热压模组A1-4层报警
D8243.00 BOOL  ; 热压模组A第2层下压板A右温度超过保护设定范围
D8243.01 BOOL  ; 热压模组A第2层下压板A右温度超限NG
D8243.02 BOOL  ; 热压模组A第2层下压板B左温度传感器断线
D8243.03 BOOL  ; 热压模组A第2层下压板B左温度超过保护设定范围
D8243.04 BOOL  ; 热压模组A第2层下压板B左温度超限NG
D8243.05 BOOL  ; 热压模组A第2层下压板B中温度传感器断线
D8243.06 BOOL  ; 热压模组A第2层下压板B中温度超过保护设定范围
D8243.07 BOOL  ; 热压模组A第2层下压板B中温度超限NG
D8243.08 BOOL  ; 热压模组A第2层下压板B右温度传感器断线
D8243.09 BOOL  ; 热压模组A第2层下压板B右温度超过保护设定范围
D8243.10 BOOL  ; 热压模组A第2层下压板B右温度超限NG
D8243.11 BOOL  ; 热压模组A第2层左侧压板温度传感器断线
D8243.12 BOOL  ; 热压模组A第2层左侧压板温度超过保护设定范围
D8243.13 BOOL  ; 热压模组A第2层左侧压板温度超限NG
D8243.14 BOOL  ; 热压模组A第2层右侧压板温度传感器断线
D8243.15 BOOL  ; 热压模组A第2层右侧压板温度超过保护设定范围
D8244 CHANNEL  ; 热压模组A1-4层报警
D8244.00 BOOL  ; 热压模组A第3层上压板左温度传感器断线
D8244.01 BOOL  ; 热压模组A第3层上压板左温度超过保护设定范围
D8244.02 BOOL  ; 热压模组A第3层上压板左温度超限NG
D8244.03 BOOL  ; 热压模组A第3层上压板中温度传感器断线
D8244.04 BOOL  ; 热压模组A第3层上压板中温度超过保护设定范围
D8244.05 BOOL  ; 热压模组A第3层上压板中温度超限NG
D8244.06 BOOL  ; 热压模组A第3层上压板右温度传感器断线
D8244.07 BOOL  ; 热压模组A第3层上压板右温度超过保护设定范围
D8244.08 BOOL  ; 热压模组A第3层上压板右温度超限NG
D8244.09 BOOL  ; 热压模组A第3层下压板A左温度传感器断线
D8244.10 BOOL  ; 热压模组A第3层下压板A左温度超过保护设定范围
D8244.11 BOOL  ; 热压模组A第3层下压板A左温度超限NG
D8244.12 BOOL  ; 热压模组A第3层下压板A中温度传感器断线
D8244.13 BOOL  ; 热压模组A第3层下压板A中温度超过保护设定范围
D8244.14 BOOL  ; 热压模组A第3层下压板A中温度超限NG
D8244.15 BOOL  ; 热压模组A第3层下压板A右温度传感器断线
D8245 CHANNEL  ; 热压模组A1-4层报警
D8245.00 BOOL  ; 热压模组A第3层下压板A右温度超过保护设定范围
D8245.01 BOOL  ; 热压模组A第3层下压板A右温度超限NG
D8245.02 BOOL  ; 热压模组A第3层下压板B左温度传感器断线
D8245.03 BOOL  ; 热压模组A第3层下压板B左温度超过保护设定范围
D8245.04 BOOL  ; 热压模组A第3层下压板B左温度超限NG
D8245.05 BOOL  ; 热压模组A第3层下压板B中温度传感器断线
D8245.06 BOOL  ; 热压模组A第3层下压板B中温度超过保护设定范围
D8245.07 BOOL  ; 热压模组A第3层下压板B中温度超限NG
D8245.08 BOOL  ; 热压模组A第3层下压板B右温度传感器断线
D8245.09 BOOL  ; 热压模组A第3层下压板B右温度超过保护设定范围
D8245.10 BOOL  ; 热压模组A第3层下压板B右温度超限NG
D8245.11 BOOL  ; 热压模组A第3层左侧压板温度传感器断线
D8245.12 BOOL  ; 热压模组A第3层左侧压板温度超过保护设定范围
D8245.13 BOOL  ; 热压模组A第3层左侧压板温度超限NG
D8245.14 BOOL  ; 热压模组A第3层右侧压板温度传感器断线
D8245.15 BOOL  ; 热压模组A第3层右侧压板温度超过保护设定范围
D8246 CHANNEL  ; 热压模组A1-4层报警
D8246.00 BOOL  ; 热压模组A第4层上压板左温度传感器断线
D8246.01 BOOL  ; 热压模组A第4层上压板左温度超过保护设定范围
D8246.02 BOOL  ; 热压模组A第4层上压板左温度超限NG
D8246.03 BOOL  ; 热压模组A第4层上压板中温度传感器断线
D8246.04 BOOL  ; 热压模组A第4层上压板中温度超过保护设定范围
D8246.05 BOOL  ; 热压模组A第4层上压板中温度超限NG
D8246.06 BOOL  ; 热压模组A第4层上压板右温度传感器断线
D8246.07 BOOL  ; 热压模组A第4层上压板右温度超过保护设定范围
D8246.08 BOOL  ; 热压模组A第4层上压板右温度超限NG
D8246.09 BOOL  ; 热压模组A第4层下压板A左温度传感器断线
D8246.10 BOOL  ; 热压模组A第4层下压板A左温度超过保护设定范围
D8246.11 BOOL  ; 热压模组A第4层下压板A左温度超限NG
D8246.12 BOOL  ; 热压模组A第4层下压板A中温度传感器断线
D8246.13 BOOL  ; 热压模组A第4层下压板A中温度超过保护设定范围
D8246.14 BOOL  ; 热压模组A第4层下压板A中温度超限NG
D8246.15 BOOL  ; 热压模组A第4层下压板A右温度传感器断线
D8247 CHANNEL  ; 热压模组A1-4层报警
D8247.00 BOOL  ; 热压模组A第4层下压板A右温度超过保护设定范围
D8247.01 BOOL  ; 热压模组A第4层下压板A右温度超限NG
D8247.02 BOOL  ; 热压模组A第4层下压板B左温度传感器断线
D8247.03 BOOL  ; 热压模组A第4层下压板B左温度超过保护设定范围
D8247.04 BOOL  ; 热压模组A第4层下压板B左温度超限NG
D8247.05 BOOL  ; 热压模组A第4层下压板B中温度传感器断线
D8247.06 BOOL  ; 热压模组A第4层下压板B中温度超过保护设定范围
D8247.07 BOOL  ; 热压模组A第4层下压板B中温度超限NG
D8247.08 BOOL  ; 热压模组A第4层下压板B右温度传感器断线
D8247.09 BOOL  ; 热压模组A第4层下压板B右温度超过保护设定范围
D8247.10 BOOL  ; 热压模组A第4层下压板B右温度超限NG
D8247.11 BOOL  ; 热压模组A第4层左侧压板温度传感器断线
D8247.12 BOOL  ; 热压模组A第4层左侧压板温度超过保护设定范围
D8247.13 BOOL  ; 热压模组A第4层左侧压板温度超限NG
D8247.14 BOOL  ; 热压模组A第4层右侧压板温度传感器断线
D8247.15 BOOL  ; 热压模组A第4层右侧压板温度超过保护设定范围
D8248 CHANNEL  ; 热压模组A1-4层报警
D8248.00 BOOL  ; 热压模组A第1层右侧压板温度超限NG
D8248.01 BOOL  ; 热压模组A第2层右侧压板温度超限NG
D8248.02 BOOL  ; 热压模组A第3层右侧压板温度超限NG
D8248.03 BOOL  ; 热压模组A第4层右侧压板温度超限NG
D8249 CHANNEL  ; 热压模组A1-4层报警
D8250 CHANNEL  ; 热压模组B1-4层报警
D8250.00 BOOL  ; 热压模组B第1层上压板左温度传感器断线
D8250.01 BOOL  ; 热压模组B第1层上压板左温度超过保护设定范围
D8250.02 BOOL  ; 热压模组B第1层上压板左温度超限NG
D8250.03 BOOL  ; 热压模组B第1层上压板中温度传感器断线
D8250.04 BOOL  ; 热压模组B第1层上压板中温度超过保护设定范围
D8250.05 BOOL  ; 热压模组B第1层上压板中温度超限NG
D8250.06 BOOL  ; 热压模组B第1层上压板右温度传感器断线
D8250.07 BOOL  ; 热压模组B第1层上压板右温度超过保护设定范围
D8250.08 BOOL  ; 热压模组B第1层上压板右温度超限NG
D8250.09 BOOL  ; 热压模组B第1层下压板A左温度传感器断线
D8250.10 BOOL  ; 热压模组B第1层下压板A左温度超过保护设定范围
D8250.11 BOOL  ; 热压模组B第1层下压板A左温度超限NG
D8250.12 BOOL  ; 热压模组B第1层下压板A中温度传感器断线
D8250.13 BOOL  ; 热压模组B第1层下压板A中温度超过保护设定范围
D8250.14 BOOL  ; 热压模组B第1层下压板A中温度超限NG
D8250.15 BOOL  ; 热压模组B第1层下压板A右温度传感器断线
D8251 CHANNEL  ; 热压模组B1-4层报警
D8251.00 BOOL  ; 热压模组B第1层下压板A右温度超过保护设定范围
D8251.01 BOOL  ; 热压模组B第1层下压板A右温度超限NG
D8251.02 BOOL  ; 热压模组B第1层下压板B左温度传感器断线
D8251.03 BOOL  ; 热压模组B第1层下压板B左温度超过保护设定范围
D8251.04 BOOL  ; 热压模组B第1层下压板B左温度超限NG
D8251.05 BOOL  ; 热压模组B第1层下压板B中温度传感器断线
D8251.06 BOOL  ; 热压模组B第1层下压板B中温度超过保护设定范围
D8251.07 BOOL  ; 热压模组B第1层下压板B中温度超限NG
D8251.08 BOOL  ; 热压模组B第1层下压板B右温度传感器断线
D8251.09 BOOL  ; 热压模组B第1层下压板B右温度超过保护设定范围
D8251.10 BOOL  ; 热压模组B第1层下压板B右温度超限NG
D8251.11 BOOL  ; 热压模组B第1层左侧压板温度传感器断线
D8251.12 BOOL  ; 热压模组B第1层左侧压板温度超过保护设定范围
D8251.13 BOOL  ; 热压模组B第1层左侧压板温度超限NG
D8251.14 BOOL  ; 热压模组B第1层右侧压板温度传感器断线
D8251.15 BOOL  ; 热压模组B第1层右侧压板温度超过保护设定范围
D8252 CHANNEL  ; 热压模组B1-4层报警
D8252.00 BOOL  ; 热压模组B第2层上压板左温度传感器断线
D8252.01 BOOL  ; 热压模组B第2层上压板左温度超过保护设定范围
D8252.02 BOOL  ; 热压模组B第2层上压板左温度超限NG
D8252.03 BOOL  ; 热压模组B第2层上压板中温度传感器断线
D8252.04 BOOL  ; 热压模组B第2层上压板中温度超过保护设定范围
D8252.05 BOOL  ; 热压模组B第2层上压板中温度超限NG
D8252.06 BOOL  ; 热压模组B第2层上压板右温度传感器断线
D8252.07 BOOL  ; 热压模组B第2层上压板右温度超过保护设定范围
D8252.08 BOOL  ; 热压模组B第2层上压板右温度超限NG
D8252.09 BOOL  ; 热压模组B第2层下压板A左温度传感器断线
D8252.10 BOOL  ; 热压模组B第2层下压板A左温度超过保护设定范围
D8252.11 BOOL  ; 热压模组B第2层下压板A左温度超限NG
D8252.12 BOOL  ; 热压模组B第2层下压板A中温度传感器断线
D8252.13 BOOL  ; 热压模组B第2层下压板A中温度超过保护设定范围
D8252.14 BOOL  ; 热压模组B第2层下压板A中温度超限NG
D8252.15 BOOL  ; 热压模组B第2层下压板A右温度传感器断线
D8253 CHANNEL  ; 热压模组B1-4层报警
D8253.00 BOOL  ; 热压模组B第2层下压板A右温度超过保护设定范围
D8253.01 BOOL  ; 热压模组B第2层下压板A右温度超限NG
D8253.02 BOOL  ; 热压模组B第2层下压板B左温度传感器断线
D8253.03 BOOL  ; 热压模组B第2层下压板B左温度超过保护设定范围
D8253.04 BOOL  ; 热压模组B第2层下压板B左温度超限NG
D8253.05 BOOL  ; 热压模组B第2层下压板B中温度传感器断线
D8253.06 BOOL  ; 热压模组B第2层下压板B中温度超过保护设定范围
D8253.07 BOOL  ; 热压模组B第2层下压板B中温度超限NG
D8253.08 BOOL  ; 热压模组B第2层下压板B右温度传感器断线
D8253.09 BOOL  ; 热压模组B第2层下压板B右温度超过保护设定范围
D8253.10 BOOL  ; 热压模组B第2层下压板B右温度超限NG
D8253.11 BOOL  ; 热压模组B第2层左侧压板温度传感器断线
D8253.12 BOOL  ; 热压模组B第2层左侧压板温度超过保护设定范围
D8253.13 BOOL  ; 热压模组B第2层左侧压板温度超限NG
D8253.14 BOOL  ; 热压模组B第2层右侧压板温度传感器断线
D8253.15 BOOL  ; 热压模组B第2层右侧压板温度超过保护设定范围
D8254 CHANNEL  ; 热压模组B1-4层报警
D8254.00 BOOL  ; 热压模组B第3层上压板左温度传感器断线
D8254.01 BOOL  ; 热压模组B第3层上压板左温度超过保护设定范围
D8254.02 BOOL  ; 热压模组B第3层上压板左温度超限NG
D8254.03 BOOL  ; 热压模组B第3层上压板中温度传感器断线
D8254.04 BOOL  ; 热压模组B第3层上压板中温度超过保护设定范围
D8254.05 BOOL  ; 热压模组B第3层上压板中温度超限NG
D8254.06 BOOL  ; 热压模组B第3层上压板右温度传感器断线
D8254.07 BOOL  ; 热压模组B第3层上压板右温度超过保护设定范围
D8254.08 BOOL  ; 热压模组B第3层上压板右温度超限NG
D8254.09 BOOL  ; 热压模组B第3层下压板A左温度传感器断线
D8254.10 BOOL  ; 热压模组B第3层下压板A左温度超过保护设定范围
D8254.11 BOOL  ; 热压模组B第3层下压板A左温度超限NG
D8254.12 BOOL  ; 热压模组B第3层下压板A中温度传感器断线
D8254.13 BOOL  ; 热压模组B第3层下压板A中温度超过保护设定范围
D8254.14 BOOL  ; 热压模组B第3层下压板A中温度超限NG
D8254.15 BOOL  ; 热压模组B第3层下压板A右温度传感器断线
D8255 CHANNEL  ; 热压模组B1-4层报警
D8255.00 BOOL  ; 热压模组B第3层下压板A右温度超过保护设定范围
D8255.01 BOOL  ; 热压模组B第3层下压板A右温度超限NG
D8255.02 BOOL  ; 热压模组B第3层下压板B左温度传感器断线
D8255.03 BOOL  ; 热压模组B第3层下压板B左温度超过保护设定范围
D8255.04 BOOL  ; 热压模组B第3层下压板B左温度超限NG
D8255.05 BOOL  ; 热压模组B第3层下压板B中温度传感器断线
D8255.06 BOOL  ; 热压模组B第3层下压板B中温度超过保护设定范围
D8255.07 BOOL  ; 热压模组B第3层下压板B中温度超限NG
D8255.08 BOOL  ; 热压模组B第3层下压板B右温度传感器断线
D8255.09 BOOL  ; 热压模组B第3层下压板B右温度超过保护设定范围
D8255.10 BOOL  ; 热压模组B第3层下压板B右温度超限NG
D8255.11 BOOL  ; 热压模组B第3层左侧压板温度传感器断线
D8255.12 BOOL  ; 热压模组B第3层左侧压板温度超过保护设定范围
D8255.13 BOOL  ; 热压模组B第3层左侧压板温度超限NG
D8255.14 BOOL  ; 热压模组B第3层右侧压板温度传感器断线
D8255.15 BOOL  ; 热压模组B第3层右侧压板温度超过保护设定范围
D8256 CHANNEL  ; 热压模组B1-4层报警
D8256.00 BOOL  ; 热压模组B第4层上压板左温度传感器断线
D8256.01 BOOL  ; 热压模组B第4层上压板左温度超过保护设定范围
D8256.02 BOOL  ; 热压模组B第4层上压板左温度超限NG
D8256.03 BOOL  ; 热压模组B第4层上压板中温度传感器断线
D8256.04 BOOL  ; 热压模组B第4层上压板中温度超过保护设定范围
D8256.05 BOOL  ; 热压模组B第4层上压板中温度超限NG
D8256.06 BOOL  ; 热压模组B第4层上压板右温度传感器断线
D8256.07 BOOL  ; 热压模组B第4层上压板右温度超过保护设定范围
D8256.08 BOOL  ; 热压模组B第4层上压板右温度超限NG
D8256.09 BOOL  ; 热压模组B第4层下压板A左温度传感器断线
D8256.10 BOOL  ; 热压模组B第4层下压板A左温度超过保护设定范围
D8256.11 BOOL  ; 热压模组B第4层下压板A左温度超限NG
D8256.12 BOOL  ; 热压模组B第4层下压板A中温度传感器断线
D8256.13 BOOL  ; 热压模组B第4层下压板A中温度超过保护设定范围
D8256.14 BOOL  ; 热压模组B第4层下压板A中温度超限NG
D8256.15 BOOL  ; 热压模组B第4层下压板A右温度传感器断线
D8257 CHANNEL  ; 热压模组B1-4层报警
D8257.00 BOOL  ; 热压模组B第4层下压板A右温度超过保护设定范围
D8257.01 BOOL  ; 热压模组B第4层下压板A右温度超限NG
D8257.02 BOOL  ; 热压模组B第4层下压板B左温度传感器断线
D8257.03 BOOL  ; 热压模组B第4层下压板B左温度超过保护设定范围
D8257.04 BOOL  ; 热压模组B第4层下压板B左温度超限NG
D8257.05 BOOL  ; 热压模组B第4层下压板B中温度传感器断线
D8257.06 BOOL  ; 热压模组B第4层下压板B中温度超过保护设定范围
D8257.07 BOOL  ; 热压模组B第4层下压板B中温度超限NG
D8257.08 BOOL  ; 热压模组B第4层下压板B右温度传感器断线
D8257.09 BOOL  ; 热压模组B第4层下压板B右温度超过保护设定范围
D8257.10 BOOL  ; 热压模组B第4层下压板B右温度超限NG
D8257.11 BOOL  ; 热压模组B第4层左侧压板温度传感器断线
D8257.12 BOOL  ; 热压模组B第4层左侧压板温度超过保护设定范围
D8257.13 BOOL  ; 热压模组B第4层左侧压板温度超限NG
D8257.14 BOOL  ; 热压模组B第4层右侧压板温度传感器断线
D8257.15 BOOL  ; 热压模组B第4层右侧压板温度超过保护设定范围
D8258 CHANNEL  ; 热压模组B1-4层报警
D8258.00 BOOL  ; 热压模组B第1层右侧压板温度超限NG
D8258.01 BOOL  ; 热压模组B第2层右侧压板温度超限NG
D8258.02 BOOL  ; 热压模组B第3层右侧压板温度超限NG
D8258.03 BOOL  ; 热压模组B第4层右侧压板温度超限NG
D8259 CHANNEL  ; 热压模组B1-4层报警
D8260 CHANNEL  ; 热压模组A5层报警
D8261 CHANNEL  ; 热压模组A5层报警
D8262 CHANNEL  ; 热压模组B5层报警
D8263 CHANNEL  ; 热压模组B5层报警
D8264 CHANNEL  ; 热压模组AB5层报警
D8270 CHANNEL  ; 副PLC输入点0CH 映射地址
D8271 CHANNEL  ; 1#副PLC输入点1CH状态
D8272 CHANNEL  ; 1#副PLC输出点100CH状态
D8273 CHANNEL  ; 1#副PLC输出点101CH状态
D8274 CHANNEL  ; 1#副PLC输出点102CH状态
D8275 CHANNEL  ; 1#副PLC输出点103CH状态
D8276 CHANNEL  ; 1#副PLC输出点104CH状态
D8277 CHANNEL  ; 1#副PLC输出点105CH状态
D8280 CHANNEL  ; 2#副PLC输入点0CH状态
D8281 CHANNEL  ; 2#副PLC输入点1CH状态
D8282 CHANNEL  ; 2#副PLC输出点100CH状态
D8283 CHANNEL  ; 2#副PLC输出点101CH状态
D8284 CHANNEL  ; 2#副PLC输出点102CH状态
D8285 CHANNEL  ; 2#副PLC输出点103CH状态
D8286 CHANNEL  ; 2#副PLC输出点104CH状态
D8287 CHANNEL  ; 2#副PLC输出点105CH状态
D8290 CHANNEL  ; 3#副PLC输入点0CH状态
D8291 CHANNEL  ; 3#副PLC输入点1CH状态
D8292 CHANNEL  ; 3#副PLC输出点100CH状态
D8293 CHANNEL  ; 3#副PLC输出点101CH状态
D8294 CHANNEL  ; 3#副PLC输出点102CH状态
D8295 CHANNEL  ; 3#副PLC输出点103CH状态
D8296 CHANNEL  ; 3#副PLC输出点104CH状态
D8297 CHANNEL  ; 3#副PLC输出点105CH状态
D8300 CHANNEL  ; 超温保护上偏差
D8301 CHANNEL  ; 侧压温度报警偏差
D8302 CHANNEL  ; 上下温度报警偏差
D8310 CHANNEL  ; 热压模组A第1层上压板左温度补偿值
D8311 CHANNEL  ; 热压模组A第1层上压板中温度补偿值
D8312 CHANNEL  ; 热压模组A第1层上压板右温度补偿值
D8313 CHANNEL  ; 热压模组A第1层下压板A左温度补偿值
D8314 CHANNEL  ; 热压模组A第1层下压板A中温度补偿值
D8315 CHANNEL  ; 热压模组A第1层下压板A右温度补偿值
D8316 CHANNEL  ; 热压模组A第1层下压板B左温度补偿值
D8317 CHANNEL  ; 热压模组A第1层下压板B中温度补偿值
D8318 CHANNEL  ; 热压模组A第1层下压板B右温度补偿值
D8319 CHANNEL  ; 热压模组A第1层左侧压板温度补偿值
D8320 CHANNEL  ; 热压模组A第1层右侧压板温度补偿值
D8330 CHANNEL  ; 热压模组A第2层上压板左温度补偿值
D8331 CHANNEL  ; 热压模组A第2层上压板中温度补偿值
D8332 CHANNEL  ; 热压模组A第2层上压板右温度补偿值
D8333 CHANNEL  ; 热压模组A第2层下压板A左温度补偿值
D8334 CHANNEL  ; 热压模组A第2层下压板A中温度补偿值
D8335 CHANNEL  ; 热压模组A第2层下压板A右温度补偿值
D8336 CHANNEL  ; 热压模组A第2层下压板B左温度补偿值
D8337 CHANNEL  ; 热压模组A第2层下压板B中温度补偿值
D8338 CHANNEL  ; 热压模组A第2层下压板B右温度补偿值
D8339 CHANNEL  ; 热压模组A第2层左侧压板温度补偿值
D8340 CHANNEL  ; 热压模组A第2层右侧压板温度补偿值
D8345.00 BOOL  ; 模组A加热全部开始
D8345.01 BOOL  ; 模组A加热全部停止
D8345.02 BOOL  ; 模组A_AT全部开始
D8345.03 BOOL  ; 模组A_AT全部停止
D8346.00 BOOL  ; 紧急停止(写入1#副PLC）
D8346.01 BOOL  ; 复位信号(写入1#副PLC）
D8346.02 BOOL  ; 五层使用(H2.00)
D8346.03 BOOL  ; 侧压启用 1-启用(H4.00)
D8346.04 BOOL  ; A模组加热屏蔽(1-屏蔽)
D8347 CHANNEL  ; 模组A加热开关报警字(0-4位)
D8350 CHANNEL  ; 热压模组A第3层上压板左温度补偿值
D8351 CHANNEL  ; 热压模组A第3层上压板中温度补偿值
D8352 CHANNEL  ; 热压模组A第3层上压板右温度补偿值
D8353 CHANNEL  ; 热压模组A第3层下压板A左温度补偿值
D8354 CHANNEL  ; 热压模组A第3层下压板A中温度补偿值
D8355 CHANNEL  ; 热压模组A第3层下压板A右温度补偿值
D8356 CHANNEL  ; 热压模组A第3层下压板B左温度补偿值
D8357 CHANNEL  ; 热压模组A第3层下压板B中温度补偿值
D8358 CHANNEL  ; 热压模组A第3层下压板B右温度补偿值
D8359 CHANNEL  ; 热压模组A第3层左侧压板温度补偿值
D8360 CHANNEL  ; 热压模组A第3层右侧压板温度补偿值
D8370 CHANNEL  ; 热压模组A第4层上压板左温度补偿值
D8371 CHANNEL  ; 热压模组A第4层上压板中温度补偿值
D8372 CHANNEL  ; 热压模组A第4层上压板右温度补偿值
D8373 CHANNEL  ; 热压模组A第4层下压板A左温度补偿值
D8374 CHANNEL  ; 热压模组A第4层下压板A中温度补偿值
D8375 CHANNEL  ; 热压模组A第4层下压板A右温度补偿值
D8376 CHANNEL  ; 热压模组A第4层下压板B左温度补偿值
D8377 CHANNEL  ; 热压模组A第4层下压板B中温度补偿值
D8378 CHANNEL  ; 热压模组A第4层下压板B右温度补偿值
D8379 CHANNEL  ; 热压模组A第4层左侧压板温度补偿值
D8380 CHANNEL  ; 热压模组A第4层右侧压板温度补偿值
D8390 CHANNEL  ; 热压模组A第5层上压板左温度补偿值
D8391 CHANNEL  ; 热压模组A第5层上压板中温度补偿值
D8392 CHANNEL  ; 热压模组A第5层上压板右温度补偿值
D8393 CHANNEL  ; 热压模组A第5层下压板A左温度补偿值
D8394 CHANNEL  ; 热压模组A第5层下压板A中温度补偿值
D8395 CHANNEL  ; 热压模组A第5层下压板A右温度补偿值
D8396 CHANNEL  ; 热压模组A第5层下压板B左温度补偿值
D8397 CHANNEL  ; 热压模组A第5层下压板B中温度补偿值
D8398 CHANNEL  ; 热压模组A第5层下压板B右温度补偿值
D8399 CHANNEL  ; 热压模组A第5层左侧压板温度补偿值
D8400 CHANNEL  ; 热压模组A第5层右侧压板温度补偿值
D8410 CHANNEL  ; 热压模组B第1层上压板左温度补偿值
D8411 CHANNEL  ; 热压模组B第1层上压板中温度补偿值
D8412 CHANNEL  ; 热压模组B第1层上压板右温度补偿值
D8413 CHANNEL  ; 热压模组B第1层下压板A左温度补偿值
D8414 CHANNEL  ; 热压模组B第1层下压板A中温度补偿值
D8415 CHANNEL  ; 热压模组B第1层下压板A右温度补偿值
D8416 CHANNEL  ; 热压模组B第1层下压板B左温度补偿值
D8417 CHANNEL  ; 热压模组B第1层下压板B中温度补偿值
D8418 CHANNEL  ; 热压模组B第1层下压板B右温度补偿值
D8419 CHANNEL  ; 热压模组B第1层左侧压板温度补偿值
D8420 CHANNEL  ; 热压模组B第1层右侧压板温度补偿值
D8430 CHANNEL  ; 热压模组B第2层上压板左温度补偿值
D8431 CHANNEL  ; 热压模组B第2层上压板中温度补偿值
D8432 CHANNEL  ; 热压模组B第2层上压板右温度补偿值
D8433 CHANNEL  ; 热压模组B第2层下压板A左温度补偿值
D8434 CHANNEL  ; 热压模组B第2层下压板A中温度补偿值
D8435 CHANNEL  ; 热压模组B第2层下压板A右温度补偿值
D8436 CHANNEL  ; 热压模组B第2层下压板B左温度补偿值
D8437 CHANNEL  ; 热压模组B第2层下压板B中温度补偿值
D8438 CHANNEL  ; 热压模组B第2层下压板B右温度补偿值
D8439 CHANNEL  ; 热压模组B第2层左侧压板温度补偿值
D8440 CHANNEL  ; 热压模组B第2层右侧压板温度补偿值
D8445.00 BOOL  ; 模组B加热全部开始
D8445.01 BOOL  ; 模组B加热全部停止
D8445.02 BOOL  ; 模组B_AT全部开始
D8445.03 BOOL  ; 模组B_AT全部停止
D8446.00 BOOL  ; 紧急停止(写入2#副PLC）
D8446.01 BOOL  ; 复位信号(写入2#副PLC）
D8446.02 BOOL  ; 五层使用(H2.00)
D8446.03 BOOL  ; 侧压启用 1-启用(H4.00)
D8446.04 BOOL  ; B模组加热屏蔽(1-屏蔽)
D8447 CHANNEL  ; 模组B加热开关报警字(0-4位)
D8450 CHANNEL  ; 热压模组B第3层上压板左温度补偿值
D8451 CHANNEL  ; 热压模组B第3层上压板中温度补偿值
D8452 CHANNEL  ; 热压模组B第3层上压板右温度补偿值
D8453 CHANNEL  ; 热压模组B第3层下压板A左温度补偿值
D8454 CHANNEL  ; 热压模组B第3层下压板A中温度补偿值
D8455 CHANNEL  ; 热压模组B第3层下压板A右温度补偿值
D8456 CHANNEL  ; 热压模组B第3层下压板B左温度补偿值
D8457 CHANNEL  ; 热压模组B第3层下压板B中温度补偿值
D8458 CHANNEL  ; 热压模组B第3层下压板B右温度补偿值
D8459 CHANNEL  ; 热压模组B第3层左侧压板温度补偿值
D8460 CHANNEL  ; 热压模组B第3层右侧压板温度补偿值
D8470 CHANNEL  ; 热压模组B第4层上压板左温度补偿值
D8471 CHANNEL  ; 热压模组B第4层上压板中温度补偿值
D8472 CHANNEL  ; 热压模组B第4层上压板右温度补偿值
D8473 CHANNEL  ; 热压模组B第4层下压板A左温度补偿值
D8474 CHANNEL  ; 热压模组B第4层下压板A中温度补偿值
D8475 CHANNEL  ; 热压模组B第4层下压板A右温度补偿值
D8476 CHANNEL  ; 热压模组B第4层下压板B左温度补偿值
D8477 CHANNEL  ; 热压模组B第4层下压板B中温度补偿值
D8478 CHANNEL  ; 热压模组B第4层下压板B右温度补偿值
D8479 CHANNEL  ; 热压模组B第4层左侧压板温度补偿值
D8480 CHANNEL  ; 热压模组B第4层右侧压板温度补偿值
D8489 CHANNEL  ; 热压模组B第5层右侧压板温度补偿值
D8490 CHANNEL  ; 热压模组B第5层上压板左温度补偿值
D8491 CHANNEL  ; 热压模组B第5层上压板中温度补偿值
D8492 CHANNEL  ; 热压模组B第5层上压板右温度补偿值
D8493 CHANNEL  ; 热压模组B第5层下压板A左温度补偿值
D8494 CHANNEL  ; 热压模组B第5层下压板A中温度补偿值
D8495 CHANNEL  ; 热压模组B第5层下压板A右温度补偿值
D8496 CHANNEL  ; 热压模组B第5层下压板B左温度补偿值
D8497 CHANNEL  ; 热压模组B第5层下压板B中温度补偿值
D8498 CHANNEL  ; 热压模组B第5层下压板B右温度补偿值
D8499 CHANNEL  ; 热压模组B第5层左侧压板温度补偿值
D8500 CHANNEL  ; 读取的测试档位值(int)
D8501 CHANNEL  ; ST5520_A 测试速度输入设定值(I)
D8502 CHANNEL  ; ST5520_A 测试模式输入设定值(I)
D8503 CHANNEL  ; 测试电压（V）设定值
D8505 CHANNEL  ; 测试时间（S）设定值
D8507 CHANNEL  ; 电阻上限（MΩ）设定值
D8509 CHANNEL  ; 电阻下限（MΩ）设定值
D8512 CHANNEL  ; 读取的测试档位值(int)
D8522 CHANNEL  ; 读取的测试模式值(int)
D8523 CHANNEL  ; 仪器1当前测试电压（V）
D8525 CHANNEL  ; ST5520_A1 绝缘测试仪测试时间读取值(Float)
D8529 CHANNEL  ; ST5520_A1 绝缘电阻下限读取值(兆欧)
D8531 CHANNEL  ; A1测量值
D8533 CHANNEL  ; 热压A1 NG类型
D8535 CHANNEL  ; A1 测试结果
D8537 CHANNEL  ; 热压A1测试时电压
D8551 CHANNEL  ; A2测量值
D8553 CHANNEL  ; 热压A2 NG类型
D8555 CHANNEL  ; 热压A2测试结果
D8557 CHANNEL  ; 热压A2测试时电压
D8571 CHANNEL  ; A3测量值
D8573 CHANNEL  ; 热压A3 NG类型
D8575 CHANNEL  ; 热压A3测试结果
D8577 CHANNEL  ; 热压A3测试时电压
D8591 CHANNEL  ; A4测量值
D8593 CHANNEL  ; 热压A4 NG类型
D8595 CHANNEL  ; 热压A4测试结果
D8597 CHANNEL  ; 热压A4测试时电压
D8611 CHANNEL  ; B1测量值
D8613 CHANNEL  ; 热压B1  NG类型
D8615 CHANNEL  ; 热压B1测试结果
D8617 CHANNEL  ; 热压B1测试时电压
D8631 CHANNEL  ; B2测量值
D8633 CHANNEL  ; 热压B2 NG类型
D8635 CHANNEL  ; 热压B2测试结果
D8637 CHANNEL  ; 热压B2测试时电压
D8651 CHANNEL  ; B3测量值
D8653 CHANNEL  ; 热压B3 NG类型
D8655 CHANNEL  ; 热压B3测试结果
D8657 CHANNEL  ; 热压B3测试时电压
D8671 CHANNEL  ; B4测量值
D8673 CHANNEL  ; 热压B4测试结果
D8675 CHANNEL  ; 热压B4测试结果
D8677 CHANNEL  ; 热压B4测试时电压
D8750 CHANNEL  ; 通讯测试
D8750.00 BOOL  ; ST5520_通讯全测试按钮（T）
D8750.10 BOOL  ; ST5520_B10 通讯测试按钮（T）
D8751 CHANNEL  ; 参数全写入
D8751.00 BOOL  ; ST5520_参数全写入按钮（T）
D8751.10 BOOL  ; ST5520_B10参数写入按钮（T）
D8752.01 BOOL  ; 热压A1测试完成
D8752.02 BOOL  ; 热压A2测试完成
D8752.03 BOOL  ; 热压A3测试完成
D8752.04 BOOL  ; 热压A4测试完成
D8752.06 BOOL  ; 热压B6测试完成
D8752.07 BOOL  ; 热压B2测试完成
D8752.08 BOOL  ; 热压B3测试完成
D8752.09 BOOL  ; 热压B4测试完成
D8753.01 BOOL  ; ST5520_A1 通讯测试异常
D8753.02 BOOL  ; ST5520_A2 通讯测试异常
D8753.03 BOOL  ; ST5520_A3 通讯异常异常
D8753.04 BOOL  ; ST5520_A4 通讯测试异常
D8753.06 BOOL  ; ST5520_A6 通讯测试异常
D8753.07 BOOL  ; ST5520_B2 通讯测试异常
D8753.08 BOOL  ; ST5520_B3 通讯测试异常
D8753.09 BOOL  ; ST5520_B4 通讯测试异常
D8760.01 BOOL  ; 4ST_A A1手动测电阻
D8760.02 BOOL  ; 4ST_A A2手动测电阻
D8760.03 BOOL  ; 4ST_A A3手动测电阻
D8760.04 BOOL  ; 4ST_A A4手动测电阻
D8760.05 BOOL  ; 4ST_B B1手动测电阻
D8760.06 BOOL  ; 4ST_B B2手动测电阻
D8760.07 BOOL  ; 4ST_B B3手动测电阻
D8760.08 BOOL  ; 4ST_B B4手动测电阻
D8760.09 BOOL  ; 4ST_A A5手动测电阻
D8760.10 BOOL  ; 4ST_B B5手动测电阻
D8761.01 BOOL  ; 热压A1触发测试电阻
D8761.02 BOOL  ; 热压A2触发测试电阻
D8761.03 BOOL  ; 热压A3触发测试电阻
D8761.04 BOOL  ; 热压A4触发测试电阻
D8761.05 BOOL  ; 热压B1触发测试电阻
D8761.06 BOOL  ; 热压B2触发测试电阻
D8761.07 BOOL  ; 热压B3触发测试电阻
D8761.08 BOOL  ; 热压B4触发测试电阻
D8761.09 BOOL  ; 热压A5触发测试电阻
D8761.10 BOOL  ; 热压B5触发测试电阻
D8762.01 BOOL  ; 热压A1测试完成
D8762.02 BOOL  ; 热压A2测试完成
D8762.03 BOOL  ; 热压A3测试完成
D8762.04 BOOL  ; 热压A4测试完成
D8762.05 BOOL  ; 热压B1测试完成
D8762.06 BOOL  ; 热压B2测试完成
D8762.07 BOOL  ; 热压B3测试完成
D8762.08 BOOL  ; 热压B4测试完成
D8762.09 BOOL  ; 热压A5测试完成
D8762.10 BOOL  ; 热压B5测试完成
D8763.01 BOOL  ; ST5520_A1 通讯测试异常
D8763.02 BOOL  ; ST5520_A2 通讯测试异常
D8763.03 BOOL  ; ST5520_A3 通讯异常异常
D8763.04 BOOL  ; ST5520_A4 通讯测试异常
D8763.05 BOOL  ; ST5520_B1 通讯测试异常
D8763.06 BOOL  ; ST5520_B2 通讯测试异常
D8763.07 BOOL  ; ST5520_B3 通讯测试异常
D8763.08 BOOL  ; ST5520_B4 通讯测试异常
D8763.09 BOOL  ; ST5520_B4 通讯测试异常
D8770 CHANNEL  ; ST5520_A数据接收延时时间
D8771 CHANNEL  ; ST5520_A Hipot测试完成取数据延时设定
D8775 CHANNEL  ; 测试时间
D8778 CHANNEL  ; 复测试次数设置
E0_10 CHANNEL  ; 短行程气缸报警延时
E0_11 CHANNEL  ; 长行程气缸报警延时
E0_12 CHANNEL  ; 平台吹气时间
E0_12100 CHANNEL  ; 进料R电芯冷却时间
E0_13 CHANNEL  ; 压板吹气时间
E0_14100 CHANNEL  ; 进料定位A电芯冷却时间
E0_15100 CHANNEL  ; 进料定位B电芯冷却时间
E0_16100 CHANNEL  ; 进出料转移进料爪A电芯冷却时间
E0_17100 CHANNEL  ; 进出料转移B进料爪电芯冷却时间
E0_18000 CHANNEL  ; 4ST_A A面数据
E0_19000 CHANNEL  ; 4ST_A B面数据
E0_20000 CHANNEL  ; 4ST_B A面数据
E0_21000 CHANNEL  ; 4ST_B B侧数据
E0_22000 CHANNEL  ; 4ST_A 热压位条码
E0_22050 CHANNEL  ; A1热压工位号1-10
E0_22051 CHANNEL  ; A1上板左温度（0.1℃）PV
E0_22052 CHANNEL  ; A1上板中温度（0.1℃）PV
E0_22053 CHANNEL  ; A1上板右温度（0.1℃）PV
E0_22054 CHANNEL  ; A1下板左温度（0.1℃）PV
E0_22055 CHANNEL  ; A1下板中温度（0.1℃）PV
E0_22056 CHANNEL  ; A1下板右温度（0.1℃）PV
E0_22057 CHANNEL  ; A1侧板左温度（0.1℃）PV
E0_22058 CHANNEL  ; A1侧板右温度（0.1℃）PV
E0_22059 CHANNEL  ; A1预压时间  PV
E0_22060 CHANNEL  ; A1热压时间1（0.1S）PV
E0_22061 CHANNEL  ; A1判定结果
E0_22061.00 BOOL  ; A1电阻OK
E0_22061.01 BOOL  ; A1压力OK
E0_22061.02 BOOL  ; A1温度OK
E0_22061.03 BOOL  ; A1时间OK
E0_22061.04 BOOL  ; A1工艺时间OK
E0_22061.05 BOOL  ; A1高度OK
E0_22061.06 BOOL  ; A1宽度OK
E0_22061.07 BOOL  ; A1极耳检测OK
E0_22061.12 BOOL  ; A1总结果OK
E0_22070 CHANNEL  ; A1上压力（KG/CM2）PV
E0_22072 CHANNEL  ; A1下压力（KG/CM2）PV
E0_22074 CHANNEL  ; A1左侧压力（KG/CM2）PV
E0_22076 CHANNEL  ; A1右侧压力（KG/CM2）PV
E0_22092 CHANNEL  ; A1测试电压（V）PV
E0_22096 CHANNEL  ; A1绝缘电阻MΩ
E0_22100 CHANNEL  ; 4A电芯冷却时间
E0_22250 CHANNEL  ; A2热压工位号1-10
E0_22251 CHANNEL  ; A2上板左温度（0.1℃）PV
E0_22254 CHANNEL  ; A2下板左温度（0.1℃）PV
E0_22257 CHANNEL  ; A2侧板左温度（0.1℃）PV
E0_22258 CHANNEL  ; A2侧板右温度（0.1℃）PV
E0_22259 CHANNEL  ; A2预压时间  PV
E0_22260 CHANNEL  ; A2热压时间1（0.1S）PV
E0_22261 CHANNEL  ; A2判定结果
E0_22261.00 BOOL  ; A2电阻OK
E0_22261.01 BOOL  ; A2压力OK
E0_22261.02 BOOL  ; A2温度OK
E0_22261.03 BOOL  ; A2热压时间OK
E0_22261.04 BOOL  ; A2工艺时间OK
E0_22261.05 BOOL  ; A2高度OK
E0_22261.06 BOOL  ; A2宽度OK
E0_22261.07 BOOL  ; A2极耳检测OK
E0_22261.12 BOOL  ; A2结果OK
E0_22270 CHANNEL  ; A2上压力（KG/CM2）PV
E0_22272 CHANNEL  ; A2下压力（KG/CM2）PV
E0_22274 CHANNEL  ; A2左侧压力（KG/CM2）PV
E0_22276 CHANNEL  ; A2右侧压力（KG/CM2）PV
E0_22292 CHANNEL  ; A2测试电压（V）PV
E0_22296 CHANNEL  ; A2绝缘电阻MΩ
E0_22450 CHANNEL  ; A3热压工位号1-10
E0_22451 CHANNEL  ; A3上板左温度（0.1℃）PV
E0_22452 CHANNEL  ; A3上板中温度（0.1℃）PV
E0_22453 CHANNEL  ; A3上板右温度（0.1℃）PV
E0_22454 CHANNEL  ; A3下板左温度（0.1℃）PV
E0_22455 CHANNEL  ; A3下板中温度（0.1℃）PV
E0_22456 CHANNEL  ; A3下板右温度（0.1℃）PV
E0_22457 CHANNEL  ; A3侧板左温度（0.1℃）PV
E0_22458 CHANNEL  ; A3侧板右温度（0.1℃）PV
E0_22459 CHANNEL  ; A3预压时间  PV
E0_22460 CHANNEL  ; A3热压时间1（0.1S）PV
E0_22461 CHANNEL  ; A3判定结果
E0_22461.00 BOOL  ; A3电阻OK
E0_22461.01 BOOL  ; A3压力OK
E0_22461.02 BOOL  ; A3温度OK
E0_22461.03 BOOL  ; A3热压时间OK
E0_22461.04 BOOL  ; A3工艺时间OK
E0_22461.05 BOOL  ; A3高度OK
E0_22461.06 BOOL  ; A3宽度OK
E0_22461.07 BOOL  ; A3极耳检测OK
E0_22461.12 BOOL  ; A3总结果OK
E0_22470 CHANNEL  ; A3上压力（KG/CM2）PV
E0_22472 CHANNEL  ; A3下压力（KG/CM2）PV
E0_22474 CHANNEL  ; A3左侧压力（KG/CM2）PV
E0_22476 CHANNEL  ; A3右侧压力（KG/CM2）PV
E0_22492 CHANNEL  ; A3测试电压（V）PV
E0_22496 CHANNEL  ; A3绝缘电阻MΩ
E0_22650 CHANNEL  ; A4热压工位号1-10
E0_22651 CHANNEL  ; A4上板左温度（0.1℃）PV
E0_22652 CHANNEL  ; A4上板中温度（0.1℃）PV
E0_22653 CHANNEL  ; A4上板右温度（0.1℃）PV
E0_22654 CHANNEL  ; A4下板左温度（0.1℃）PV
E0_22655 CHANNEL  ; A4下板中温度（0.1℃）PV
E0_22656 CHANNEL  ; A4下板右温度（0.1℃）PV
E0_22657 CHANNEL  ; A4侧板左温度（0.1℃）PV
E0_22658 CHANNEL  ; A4侧板右温度（0.1℃）PV
E0_22659 CHANNEL  ; A4预压时间  PV
E0_22660 CHANNEL  ; A4热压时间1（0.1S）PV
E0_22661 CHANNEL  ; A4判定结果
E0_22661.00 BOOL  ; A4电阻OK
E0_22661.01 BOOL  ; A4压力OK
E0_22661.02 BOOL  ; A4温度OK
E0_22661.03 BOOL  ; A4热压时间OK
E0_22661.04 BOOL  ; A4工艺时间OK
E0_22661.05 BOOL  ; A4高度OK
E0_22661.06 BOOL  ; A4宽度OK
E0_22661.07 BOOL  ; A4极耳检测OK
E0_22661.12 BOOL  ; A4总结果OK
E0_22670 CHANNEL  ; A4上压力（KG/CM2）PV
E0_22672 CHANNEL  ; A4下压力（KG/CM2）PV
E0_22674 CHANNEL  ; A4左侧压力（KG/CM2）PV
E0_22676 CHANNEL  ; A4右侧压力（KG/CM2）PV
E0_22692 CHANNEL  ; A4测试电压（V）PV
E0_22696 CHANNEL  ; A4绝缘电阻MΩ
E0_22850 CHANNEL  ; A5热压工位号1-10
E0_22851 CHANNEL  ; A5上板左温度（0.1℃）PV
E0_22852 CHANNEL  ; A5上板中温度（0.1℃）PV
E0_22853 CHANNEL  ; A5上板右温度（0.1℃）PV
E0_22854 CHANNEL  ; A5下板左温度（0.1℃）PV
E0_22855 CHANNEL  ; A5下板中温度（0.1℃）PV
E0_22856 CHANNEL  ; A5下板右温度（0.1℃）PV
E0_22857 CHANNEL  ; A5侧板左温度（0.1℃）PV
E0_22858 CHANNEL  ; A5侧板右温度（0.1℃）PV
E0_22859 CHANNEL  ; A5预压时间  PV
E0_22860 CHANNEL  ; A5热压时间1（0.1S）PV
E0_22861 CHANNEL  ; A5判定结果
E0_22861.00 BOOL  ; A5电阻OK
E0_22861.01 BOOL  ; A5压力OK
E0_22861.02 BOOL  ; A5温度OK
E0_22861.03 BOOL  ; A5热压时间OK
E0_22861.04 BOOL  ; A5工艺时间OK
E0_22861.05 BOOL  ; A5高度OK
E0_22861.06 BOOL  ; A5宽度OK
E0_22861.07 BOOL  ; A5极耳检测OK
E0_22861.12 BOOL  ; A5总结果OK
E0_22870 CHANNEL  ; A5上压力（KG/CM2）PV
E0_22872 CHANNEL  ; A5下压力（KG/CM2）PV
E0_22874 CHANNEL  ; A5左侧压力（KG/CM2）PV
E0_22876 CHANNEL  ; A5右侧压力（KG/CM2）PV
E0_22892 CHANNEL  ; A5测试电压（V）PV
E0_22896 CHANNEL  ; A5绝缘电阻MΩ
E0_23000 CHANNEL  ; 4ST_B 热压位数据
E0_23050 CHANNEL  ; B1热压工位号1-10
E0_23051 CHANNEL  ; B1上板左温度（0.1℃）PV
E0_23052 CHANNEL  ; B1上板中温度（0.1℃）PV
E0_23053 CHANNEL  ; B1上板右温度（0.1℃）PV
E0_23054 CHANNEL  ; B1下板左温度（0.1℃）PV
E0_23055 CHANNEL  ; B1下板中温度（0.1℃）PV
E0_23056 CHANNEL  ; B1下板右温度（0.1℃）PV
E0_23057 CHANNEL  ; B1侧板左温度（0.1℃）PV
E0_23058 CHANNEL  ; B1侧板右温度（0.1℃）PV
E0_23059 CHANNEL  ; B1预压时间  PV
E0_23060 CHANNEL  ; B1热压时间1（0.1S）PV
E0_23061 CHANNEL  ; B1判定结果
E0_23061.00 BOOL  ; B1电阻OK
E0_23061.01 BOOL  ; B1压力OK
E0_23061.02 BOOL  ; B1温度OK
E0_23061.03 BOOL  ; B1时间OK
E0_23061.04 BOOL  ; B1工艺时间OK
E0_23061.05 BOOL  ; B1高度OK
E0_23061.06 BOOL  ; B1宽度OK
E0_23061.07 BOOL  ; B1极耳检测OK
E0_23061.12 BOOL  ; B1总结果OK
E0_23070 CHANNEL  ; B1上压力（KG/CM2）PV
E0_23072 CHANNEL  ; B1下压力（KG/CM2）PV
E0_23074 CHANNEL  ; B1左侧压力（KG/CM2）PV
E0_23076 CHANNEL  ; B1右侧压力（KG/CM2）PV
E0_23092 CHANNEL  ; B1测试电压（V）PV
E0_23096 CHANNEL  ; B1绝缘电阻MΩ
E0_23100 CHANNEL  ; B热压电芯冷却时间
E0_23250 CHANNEL  ; B2热压工位号1-10
E0_23251 CHANNEL  ; B2上板左温度（0.1℃）PV
E0_23254 CHANNEL  ; B2下板左温度（0.1℃）PV
E0_23257 CHANNEL  ; B2侧板左温度（0.1℃）PV
E0_23258 CHANNEL  ; B2侧板右温度（0.1℃）PV
E0_23259 CHANNEL  ; B2预压时间  PV
E0_23260 CHANNEL  ; B2热压时间1（0.1S）PV
E0_23261 CHANNEL  ; B2判定结果
E0_23261.00 BOOL  ; B2电阻OK
E0_23261.01 BOOL  ; B2压力OK
E0_23261.02 BOOL  ; B2温度OK
E0_23261.03 BOOL  ; B2时间OK
E0_23261.04 BOOL  ; B2工艺时间OK
E0_23261.05 BOOL  ; B2高度OK
E0_23261.06 BOOL  ; B2宽度OK
E0_23261.07 BOOL  ; B2极耳检测OK
E0_23270 CHANNEL  ; B2上压力（KG/CM2）PV
E0_23272 CHANNEL  ; B2下压力（KG/CM2）PV
E0_23274 CHANNEL  ; B2左侧压力（KG/CM2）PV
E0_23276 CHANNEL  ; B2右侧压力（KG/CM2）PV
E0_23292 CHANNEL  ; B2测试电压（V）PV
E0_23296 CHANNEL  ; B2绝缘电阻MΩ
E0_23450 CHANNEL  ; B3热压工位号1-10
E0_23451 CHANNEL  ; B3上板左温度（0.1℃）PV
E0_23452 CHANNEL  ; B3上板中温度（0.1℃）PV
E0_23453 CHANNEL  ; B3上板右温度（0.1℃）PV
E0_23454 CHANNEL  ; B3下板左温度（0.1℃）PV
E0_23455 CHANNEL  ; B3下板中温度（0.1℃）PV
E0_23456 CHANNEL  ; B3下板右温度（0.1℃）PV
E0_23457 CHANNEL  ; B3侧板左温度（0.1℃）PV
E0_23458 CHANNEL  ; B3侧板右温度（0.1℃）PV
E0_23459 CHANNEL  ; B3预压时间  PV
E0_23460 CHANNEL  ; B3热压时间1（0.1S）PV
E0_23461 CHANNEL  ; B3判定结果
E0_23461.00 BOOL  ; B3电阻OK
E0_23461.01 BOOL  ; B3压力OK
E0_23461.02 BOOL  ; B3温度OK
E0_23461.03 BOOL  ; B3时间OK
E0_23461.04 BOOL  ; B3工艺时间OK
E0_23461.05 BOOL  ; B3高度OK
E0_23461.06 BOOL  ; B3宽度OK
E0_23461.07 BOOL  ; B3极耳检测OK
E0_23461.12 BOOL  ; B3总结果OK
E0_23470 CHANNEL  ; B3上压力（KG/CM2）PV
E0_23472 CHANNEL  ; B3下压力（KG/CM2）PV
E0_23474 CHANNEL  ; B3左侧压力（KG/CM2）PV
E0_23476 CHANNEL  ; B3右侧压力（KG/CM2）PV
E0_23492 CHANNEL  ; B3测试电压（V）PV
E0_23496 CHANNEL  ; B3绝缘电阻MΩ
E0_23650 CHANNEL  ; B4热压工位号1-10
E0_23651 CHANNEL  ; B4上板左温度（0.1℃）PV
E0_23652 CHANNEL  ; B4上板中温度（0.1℃）PV
E0_23653 CHANNEL  ; B4上板右温度（0.1℃）PV
E0_23654 CHANNEL  ; B4下板左温度（0.1℃）PV
E0_23655 CHANNEL  ; B4下板中温度（0.1℃）PV
E0_23656 CHANNEL  ; B4下板右温度（0.1℃）PV
E0_23657 CHANNEL  ; B4侧板左温度（0.1℃）PV
E0_23658 CHANNEL  ; B4侧板右温度（0.1℃）PV
E0_23659 CHANNEL  ; B4预压时间  PV
E0_23660 CHANNEL  ; B4热压时间1（0.1S）PV
E0_23661 CHANNEL  ; B4判定结果
E0_23661.00 BOOL  ; B4电阻OK
E0_23661.01 BOOL  ; B4压力OK
E0_23661.02 BOOL  ; B4温度OK
E0_23661.03 BOOL  ; B4时间OK
E0_23661.04 BOOL  ; B4工艺时间OK
E0_23661.05 BOOL  ; B4高度OK
E0_23661.06 BOOL  ; B4宽度OK
E0_23661.07 BOOL  ; B4极耳检测OK
E0_23661.12 BOOL  ; B4总结果OK
E0_23670 CHANNEL  ; B4上压力（KG/CM2）PV
E0_23672 CHANNEL  ; B4下压力（KG/CM2）PV
E0_23674 CHANNEL  ; B4左侧压力（KG/CM2）PV
E0_23676 CHANNEL  ; B4右侧压力（KG/CM2）PV
E0_23692 CHANNEL  ; B4测试电压（V）PV
E0_23696 CHANNEL  ; B4绝缘电阻MΩ
E0_23850 CHANNEL  ; B5热压工位号1-10
E0_23851 CHANNEL  ; B5上板左温度（0.1℃）PV
E0_23852 CHANNEL  ; B5上板中温度（0.1℃）PV
E0_23853 CHANNEL  ; B5上板右温度（0.1℃）PV
E0_23854 CHANNEL  ; B5下板左温度（0.1℃）PV
E0_23855 CHANNEL  ; B5下板中温度（0.1℃）PV
E0_23856 CHANNEL  ; B5下板右温度（0.1℃）PV
E0_23857 CHANNEL  ; B5侧板左温度（0.1℃）PV
E0_23858 CHANNEL  ; B5侧板右温度（0.1℃）PV
E0_23859 CHANNEL  ; B5预压时间  PV
E0_23860 CHANNEL  ; B5热压时间1（0.1S）PV
E0_23861 CHANNEL  ; B5判定结果
E0_23861.00 BOOL  ; B5电阻OK
E0_23861.01 BOOL  ; B5压力OK
E0_23861.02 BOOL  ; B5温度OK
E0_23861.03 BOOL  ; B5时间OK
E0_23861.04 BOOL  ; B5工艺时间OK
E0_23861.05 BOOL  ; B5高度OK
E0_23861.06 BOOL  ; B5宽度OK
E0_23861.07 BOOL  ; B5极耳检测OK
E0_23861.12 BOOL  ; B5总结果OK
E0_23870 CHANNEL  ; B5上压力（KG/CM2）PV
E0_23872 CHANNEL  ; B5下压力（KG/CM2）PV
E0_23874 CHANNEL  ; B5左侧压力（KG/CM2）PV
E0_23876 CHANNEL  ; B5右侧压力（KG/CM2）PV
E0_23892 CHANNEL  ; B5测试电压（V）PV
E0_23896 CHANNEL  ; B5绝缘电阻MΩ
E0_30061.00 BOOL  ; A1HipotNG
E0_30061.12 BOOL  ; A1电芯总结果OK
E0_30261.00 BOOL  ; A2HipotNG
E0_30261.12 BOOL  ; A2电芯总结果OK
E0_30461.00 BOOL  ; A3HipotNG
E0_30461.12 BOOL  ; A3电芯总结果OK
E0_30661.00 BOOL  ; A4HipotNG
E0_30661.12 BOOL  ; A4电芯总结果OK
E0_30861.00 BOOL  ; A5HipotNG
E0_30861.12 BOOL  ; A5电芯总结果OK
E0_31061.00 BOOL  ; B1HipotNG
E0_31061.12 BOOL  ; B1电芯总结果OK
E0_31261.00 BOOL  ; B2HipotNG
E0_31261.12 BOOL  ; B2电芯总结果OK
E0_31461.00 BOOL  ; B3HipotNG
E0_31461.12 BOOL  ; B3电芯总结果OK
E0_31661.00 BOOL  ; B4HipotNG
E0_31661.12 BOOL  ; B4电芯总结果OK
E0_31861.00 BOOL  ; B5HipotNG
E0_31861.12 BOOL  ; B5电芯总结果OK
E0_4 CHANNEL  ; 伺服定位条件延时
E0_8000.00 BOOL  ; 设备上电状态
E0_8000.01 BOOL  ; 设备复位状态
E0_8000.02 BOOL  ; 设备自动状态
E0_8000.03 BOOL  ; 设备停止状态
E0_8000.04 BOOL  ; 设备启动状态
E0_8000.05 BOOL  ; 设备待料状态
E0_8000.06 BOOL  ; 设备手动状态
E0_8000.07 BOOL  ; 设备出错状态
E0_8000.08 BOOL  ; 设备急停状态
E0_8000.09 BOOL  ; 设备急停状态
E0_8010 CHANNEL  ; 入站就绪通知1
E0_8011 CHANNEL  ; 入站就绪通知2
E0_8012 CHANNEL  ; 入站就绪通知3
E0_8013 CHANNEL  ; 入站就绪通知4
E0_8014 CHANNEL  ; 入站就绪通知5
E0_8015 CHANNEL  ; 入站就绪通知6
E0_8016 CHANNEL  ; 入站就绪通知7
E0_8017 CHANNEL  ; 入站就绪通知8
E0_8018 CHANNEL  ; 入站就绪通知9
E0_8019 CHANNEL  ; 入站就绪通知10
E0_8020 CHANNEL  ; 入站就绪确认1
E0_8021 CHANNEL  ; 入站就绪确认2
E0_8022 CHANNEL  ; 入站就绪确认3
E0_8023 CHANNEL  ; 入站就绪确认4
E0_8024 CHANNEL  ; 入站就绪确认5
E0_8025 CHANNEL  ; 入站就绪确认6
E0_8026 CHANNEL  ; 入站就绪确认7
E0_8027 CHANNEL  ; 入站就绪确认8
E0_8028 CHANNEL  ; 入站就绪确认9
E0_8029 CHANNEL  ; 入站就绪确认10
E0_8030 CHANNEL  ; PC读取条码就绪确认1
E0_8031 CHANNEL  ; PC读取条码就绪确认2
E0_8032 CHANNEL  ; PC读取条码就绪确认3
E0_8033 CHANNEL  ; PC读取条码就绪确认4
E0_8034 CHANNEL  ; PC读取条码就绪确认5
E0_8035 CHANNEL  ; PC读取条码就绪确认6
E0_8036 CHANNEL  ; PC读取条码就绪确认7
E0_8037 CHANNEL  ; PC读取条码就绪确认8
E0_8038 CHANNEL  ; PC读取条码就绪确认9
E0_8039 CHANNEL  ; PC读取条码就绪确认10
E0_8040 CHANNEL  ; PLC读取条码就绪确认1
E0_8041 CHANNEL  ; PLC读取条码就绪确认2
E0_8042 CHANNEL  ; PLC读取条码就绪确认3
E0_8043 CHANNEL  ; PLC读取条码就绪确认4
E0_8044 CHANNEL  ; PLC读取条码就绪确认5
E0_8045 CHANNEL  ; PLC读取条码就绪确认6
E0_8046 CHANNEL  ; PLC读取条码就绪确认7
E0_8047 CHANNEL  ; PLC读取条码就绪确认8
E0_8048 CHANNEL  ; PLC读取条码就绪确认9
E0_8049 CHANNEL  ; PLC读取条码就绪确认10
E0_8050 CHANNEL  ; 出站就绪通知1
E0_8051 CHANNEL  ; 出站就绪通知2
E0_8052 CHANNEL  ; 出站就绪通知3
E0_8053 CHANNEL  ; 出站就绪通知4
E0_8054 CHANNEL  ; 出站就绪通知5
E0_8055 CHANNEL  ; 出站就绪通知6
E0_8056 CHANNEL  ; 出站就绪通知7
E0_8057 CHANNEL  ; 出站就绪通知8
E0_8058 CHANNEL  ; 出站就绪通知9
E0_8059 CHANNEL  ; 出站就绪通知10
E0_8060 CHANNEL  ; 出站就绪确认1
E0_8061 CHANNEL  ; 出站就绪确认2
E0_8062 CHANNEL  ; 出站就绪确认3
E0_8063 CHANNEL  ; 出站就绪确认4
E0_8064 CHANNEL  ; 出站就绪确认5
E0_8065 CHANNEL  ; 出站就绪确认6
E0_8066 CHANNEL  ; 出站就绪确认7
E0_8067 CHANNEL  ; 出站就绪确认8
E0_8068 CHANNEL  ; 出站就绪确认9
E0_8069 CHANNEL  ; 出站就绪确认10
E0_8070 CHANNEL  ; 出站工位编号1
E0_8071 CHANNEL  ; 出站工位编号2
E0_8072 CHANNEL  ; 出站工位编号3
E0_8073 CHANNEL  ; 出站工位编号4
E0_8074 CHANNEL  ; 出站工位编号5
E0_8075 CHANNEL  ; 出站工位编号6
E0_8076 CHANNEL  ; 出站工位编号7
E0_8077 CHANNEL  ; 出站工位编号8
E0_8078 CHANNEL  ; 出站工位编号9
E0_8079 CHANNEL  ; 出站工位编号10
E0_9000 CHANNEL  ; 入站条码1
E0_9001 CHANNEL  ; 入站条码1
E0_9002 CHANNEL  ; 入站条码1
E0_9003 CHANNEL  ; 入站条码1
E0_9004 CHANNEL  ; 入站条码1
E0_9005 CHANNEL  ; 入站条码1
E0_9006 CHANNEL  ; 入站条码1
E0_9007 CHANNEL  ; 入站条码1
E0_9008 CHANNEL  ; 入站条码1
E0_9009 CHANNEL  ; 入站条码1
E0_9010 CHANNEL  ; 入站条码1
E0_9011 CHANNEL  ; 入站条码1
E0_9012 CHANNEL  ; 入站条码1
E0_9013 CHANNEL  ; 入站条码1
E0_9014 CHANNEL  ; 入站条码1
E0_9015 CHANNEL  ; 入站条码1
E0_9016 CHANNEL  ; 入站条码1
E0_9017 CHANNEL  ; 入站条码1
E0_9018 CHANNEL  ; 入站条码1
E0_9019 CHANNEL  ; 入站条码1
E0_9020 CHANNEL  ; 入站条码1
E0_9021 CHANNEL  ; 入站条码1
E0_9022 CHANNEL  ; 入站条码1
E0_9023 CHANNEL  ; 入站条码1
E0_9024 CHANNEL  ; 入站条码1
E0_9025 CHANNEL  ; 入站条码1
E0_9026 CHANNEL  ; 入站条码1
E0_9027 CHANNEL  ; 入站条码1
E0_9028 CHANNEL  ; 入站条码1
E0_9029 CHANNEL  ; 入站条码1
E0_9030 CHANNEL  ; 入站条码1
E0_9031 CHANNEL  ; 入站条码1
E0_9032 CHANNEL  ; 入站条码1
E0_9033 CHANNEL  ; 入站条码1
E0_9034 CHANNEL  ; 入站条码1
E0_9035 CHANNEL  ; 入站条码1
E0_9036 CHANNEL  ; 入站条码1
E0_9037 CHANNEL  ; 入站条码1
E0_9038 CHANNEL  ; 入站条码1
E0_9039 CHANNEL  ; 入站条码1
E0_9040 CHANNEL  ; 入站条码1
E0_9041 CHANNEL  ; 入站条码1
E0_9042 CHANNEL  ; 入站条码1
E0_9043 CHANNEL  ; 入站条码1
E0_9044 CHANNEL  ; 入站条码1
E0_9045 CHANNEL  ; 入站条码1
E0_9046 CHANNEL  ; 入站条码1
E0_9047 CHANNEL  ; 入站条码1
E0_9048 CHANNEL  ; 入站条码1
E0_9049 CHANNEL  ; 入站条码1
E0_9100 CHANNEL  ; 入站条码2
E0_9101 CHANNEL  ; 入站条码2
E0_9102 CHANNEL  ; 入站条码2
E0_9103 CHANNEL  ; 入站条码2
E0_9104 CHANNEL  ; 入站条码2
E0_9105 CHANNEL  ; 入站条码2
E0_9106 CHANNEL  ; 入站条码2
E0_9107 CHANNEL  ; 入站条码2
E0_9108 CHANNEL  ; 入站条码2
E0_9109 CHANNEL  ; 入站条码2
E0_9110 CHANNEL  ; 入站条码2
E0_9111 CHANNEL  ; 入站条码2
E0_9112 CHANNEL  ; 入站条码2
E0_9113 CHANNEL  ; 入站条码2
E0_9114 CHANNEL  ; 入站条码2
E0_9115 CHANNEL  ; 入站条码2
E0_9116 CHANNEL  ; 入站条码2
E0_9117 CHANNEL  ; 入站条码2
E0_9118 CHANNEL  ; 入站条码2
E0_9119 CHANNEL  ; 入站条码2
E0_9120 CHANNEL  ; 入站条码2
E0_9121 CHANNEL  ; 入站条码2
E0_9122 CHANNEL  ; 入站条码2
E0_9123 CHANNEL  ; 入站条码2
E0_9124 CHANNEL  ; 入站条码2
E0_9125 CHANNEL  ; 入站条码2
E0_9126 CHANNEL  ; 入站条码2
E0_9127 CHANNEL  ; 入站条码2
E0_9128 CHANNEL  ; 入站条码2
E0_9129 CHANNEL  ; 入站条码2
E0_9130 CHANNEL  ; 入站条码2
E0_9131 CHANNEL  ; 入站条码2
E0_9132 CHANNEL  ; 入站条码2
E0_9133 CHANNEL  ; 入站条码2
E0_9134 CHANNEL  ; 入站条码2
E0_9135 CHANNEL  ; 入站条码2
E0_9136 CHANNEL  ; 入站条码2
E0_9137 CHANNEL  ; 入站条码2
E0_9138 CHANNEL  ; 入站条码2
E0_9139 CHANNEL  ; 入站条码2
E0_9140 CHANNEL  ; 入站条码2
E0_9141 CHANNEL  ; 入站条码2
E0_9142 CHANNEL  ; 入站条码2
E0_9143 CHANNEL  ; 入站条码2
E0_9144 CHANNEL  ; 入站条码2
E0_9145 CHANNEL  ; 入站条码2
E0_9146 CHANNEL  ; 入站条码2
E0_9147 CHANNEL  ; 入站条码2
E0_9148 CHANNEL  ; 入站条码2
E0_9149 CHANNEL  ; 入站条码2
E0_9200 CHANNEL  ; 入站条码3
E0_9201 CHANNEL  ; 入站条码3
E0_9202 CHANNEL  ; 入站条码3
E0_9203 CHANNEL  ; 入站条码3
E0_9204 CHANNEL  ; 入站条码3
E0_9205 CHANNEL  ; 入站条码3
E0_9206 CHANNEL  ; 入站条码3
E0_9207 CHANNEL  ; 入站条码3
E0_9208 CHANNEL  ; 入站条码3
E0_9209 CHANNEL  ; 入站条码3
E0_9210 CHANNEL  ; 入站条码3
E0_9211 CHANNEL  ; 入站条码3
E0_9212 CHANNEL  ; 入站条码3
E0_9213 CHANNEL  ; 入站条码3
E0_9214 CHANNEL  ; 入站条码3
E0_9215 CHANNEL  ; 入站条码3
E0_9216 CHANNEL  ; 入站条码3
E0_9217 CHANNEL  ; 入站条码3
E0_9218 CHANNEL  ; 入站条码3
E0_9219 CHANNEL  ; 入站条码3
E0_9220 CHANNEL  ; 入站条码3
E0_9221 CHANNEL  ; 入站条码3
E0_9222 CHANNEL  ; 入站条码3
E0_9223 CHANNEL  ; 入站条码3
E0_9224 CHANNEL  ; 入站条码3
E0_9225 CHANNEL  ; 入站条码3
E0_9226 CHANNEL  ; 入站条码3
E0_9227 CHANNEL  ; 入站条码3
E0_9228 CHANNEL  ; 入站条码3
E0_9229 CHANNEL  ; 入站条码3
E0_9230 CHANNEL  ; 入站条码3
E0_9231 CHANNEL  ; 入站条码3
E0_9232 CHANNEL  ; 入站条码3
E0_9233 CHANNEL  ; 入站条码3
E0_9234 CHANNEL  ; 入站条码3
E0_9235 CHANNEL  ; 入站条码3
E0_9236 CHANNEL  ; 入站条码3
E0_9237 CHANNEL  ; 入站条码3
E0_9238 CHANNEL  ; 入站条码3
E0_9239 CHANNEL  ; 入站条码3
E0_9240 CHANNEL  ; 入站条码3
E0_9241 CHANNEL  ; 入站条码3
E0_9242 CHANNEL  ; 入站条码3
E0_9243 CHANNEL  ; 入站条码3
E0_9244 CHANNEL  ; 入站条码3
E0_9245 CHANNEL  ; 入站条码3
E0_9246 CHANNEL  ; 入站条码3
E0_9247 CHANNEL  ; 入站条码3
E0_9248 CHANNEL  ; 入站条码3
E0_9249 CHANNEL  ; 入站条码3
E0_9300 CHANNEL  ; 入站条码4
E0_9301 CHANNEL  ; 入站条码4
E0_9302 CHANNEL  ; 入站条码4
E0_9303 CHANNEL  ; 入站条码4
E0_9304 CHANNEL  ; 入站条码4
E0_9305 CHANNEL  ; 入站条码4
E0_9306 CHANNEL  ; 入站条码4
E0_9307 CHANNEL  ; 入站条码4
E0_9308 CHANNEL  ; 入站条码4
E0_9309 CHANNEL  ; 入站条码4
E0_9310 CHANNEL  ; 入站条码4
E0_9311 CHANNEL  ; 入站条码4
E0_9312 CHANNEL  ; 入站条码4
E0_9313 CHANNEL  ; 入站条码4
E0_9314 CHANNEL  ; 入站条码4
E0_9315 CHANNEL  ; 入站条码4
E0_9316 CHANNEL  ; 入站条码4
E0_9317 CHANNEL  ; 入站条码4
E0_9318 CHANNEL  ; 入站条码4
E0_9319 CHANNEL  ; 入站条码4
E0_9320 CHANNEL  ; 入站条码4
E0_9321 CHANNEL  ; 入站条码4
E0_9322 CHANNEL  ; 入站条码4
E0_9323 CHANNEL  ; 入站条码4
E0_9324 CHANNEL  ; 入站条码4
E0_9325 CHANNEL  ; 入站条码4
E0_9326 CHANNEL  ; 入站条码4
E0_9327 CHANNEL  ; 入站条码4
E0_9328 CHANNEL  ; 入站条码4
E0_9329 CHANNEL  ; 入站条码4
E0_9330 CHANNEL  ; 入站条码4
E0_9331 CHANNEL  ; 入站条码4
E0_9332 CHANNEL  ; 入站条码4
E0_9333 CHANNEL  ; 入站条码4
E0_9334 CHANNEL  ; 入站条码4
E0_9335 CHANNEL  ; 入站条码4
E0_9336 CHANNEL  ; 入站条码4
E0_9337 CHANNEL  ; 入站条码4
E0_9338 CHANNEL  ; 入站条码4
E0_9339 CHANNEL  ; 入站条码4
E0_9340 CHANNEL  ; 入站条码4
E0_9341 CHANNEL  ; 入站条码4
E0_9342 CHANNEL  ; 入站条码4
E0_9343 CHANNEL  ; 入站条码4
E0_9344 CHANNEL  ; 入站条码4
E0_9345 CHANNEL  ; 入站条码4
E0_9346 CHANNEL  ; 入站条码4
E0_9347 CHANNEL  ; 入站条码4
E0_9348 CHANNEL  ; 入站条码4
E0_9349 CHANNEL  ; 入站条码4
E0_9400 CHANNEL  ; 入站条码5
E0_9401 CHANNEL  ; 入站条码5
E0_9402 CHANNEL  ; 入站条码5
E0_9403 CHANNEL  ; 入站条码5
E0_9404 CHANNEL  ; 入站条码5
E0_9405 CHANNEL  ; 入站条码5
E0_9406 CHANNEL  ; 入站条码5
E0_9407 CHANNEL  ; 入站条码5
E0_9408 CHANNEL  ; 入站条码5
E0_9409 CHANNEL  ; 入站条码5
E0_9410 CHANNEL  ; 入站条码5
E0_9411 CHANNEL  ; 入站条码5
E0_9412 CHANNEL  ; 入站条码5
E0_9413 CHANNEL  ; 入站条码5
E0_9414 CHANNEL  ; 入站条码5
E0_9415 CHANNEL  ; 入站条码5
E0_9416 CHANNEL  ; 入站条码5
E0_9417 CHANNEL  ; 入站条码5
E0_9418 CHANNEL  ; 入站条码5
E0_9419 CHANNEL  ; 入站条码5
E0_9420 CHANNEL  ; 入站条码5
E0_9421 CHANNEL  ; 入站条码5
E0_9422 CHANNEL  ; 入站条码5
E0_9423 CHANNEL  ; 入站条码5
E0_9424 CHANNEL  ; 入站条码5
E0_9425 CHANNEL  ; 入站条码5
E0_9426 CHANNEL  ; 入站条码5
E0_9427 CHANNEL  ; 入站条码5
E0_9428 CHANNEL  ; 入站条码5
E0_9429 CHANNEL  ; 入站条码5
E0_9430 CHANNEL  ; 入站条码5
E0_9431 CHANNEL  ; 入站条码5
E0_9432 CHANNEL  ; 入站条码5
E0_9433 CHANNEL  ; 入站条码5
E0_9434 CHANNEL  ; 入站条码5
E0_9435 CHANNEL  ; 入站条码5
E0_9436 CHANNEL  ; 入站条码5
E0_9437 CHANNEL  ; 入站条码5
E0_9438 CHANNEL  ; 入站条码5
E0_9439 CHANNEL  ; 入站条码5
E0_9440 CHANNEL  ; 入站条码5
E0_9441 CHANNEL  ; 入站条码5
E0_9442 CHANNEL  ; 入站条码5
E0_9443 CHANNEL  ; 入站条码5
E0_9444 CHANNEL  ; 入站条码5
E0_9445 CHANNEL  ; 入站条码5
E0_9446 CHANNEL  ; 入站条码5
E0_9447 CHANNEL  ; 入站条码5
E0_9448 CHANNEL  ; 入站条码5
E0_9449 CHANNEL  ; 入站条码5
E0_9500 CHANNEL  ; 入站条码6
E0_9501 CHANNEL  ; 入站条码6
E0_9502 CHANNEL  ; 入站条码6
E0_9503 CHANNEL  ; 入站条码6
E0_9504 CHANNEL  ; 入站条码6
E0_9505 CHANNEL  ; 入站条码6
E0_9506 CHANNEL  ; 入站条码6
E0_9507 CHANNEL  ; 入站条码6
E0_9508 CHANNEL  ; 入站条码6
E0_9509 CHANNEL  ; 入站条码6
E0_9510 CHANNEL  ; 入站条码6
E0_9511 CHANNEL  ; 入站条码6
E0_9512 CHANNEL  ; 入站条码6
E0_9513 CHANNEL  ; 入站条码6
E0_9514 CHANNEL  ; 入站条码6
E0_9515 CHANNEL  ; 入站条码6
E0_9516 CHANNEL  ; 入站条码6
E0_9517 CHANNEL  ; 入站条码6
E0_9518 CHANNEL  ; 入站条码6
E0_9519 CHANNEL  ; 入站条码6
E0_9520 CHANNEL  ; 入站条码6
E0_9521 CHANNEL  ; 入站条码6
E0_9522 CHANNEL  ; 入站条码6
E0_9523 CHANNEL  ; 入站条码6
E0_9524 CHANNEL  ; 入站条码6
E0_9525 CHANNEL  ; 入站条码6
E0_9526 CHANNEL  ; 入站条码6
E0_9527 CHANNEL  ; 入站条码6
E0_9528 CHANNEL  ; 入站条码6
E0_9529 CHANNEL  ; 入站条码6
E0_9530 CHANNEL  ; 入站条码6
E0_9531 CHANNEL  ; 入站条码6
E0_9532 CHANNEL  ; 入站条码6
E0_9533 CHANNEL  ; 入站条码6
E0_9534 CHANNEL  ; 入站条码6
E0_9535 CHANNEL  ; 入站条码6
E0_9536 CHANNEL  ; 入站条码6
E0_9537 CHANNEL  ; 入站条码6
E0_9538 CHANNEL  ; 入站条码6
E0_9539 CHANNEL  ; 入站条码6
E0_9540 CHANNEL  ; 入站条码6
E0_9541 CHANNEL  ; 入站条码6
E0_9542 CHANNEL  ; 入站条码6
E0_9543 CHANNEL  ; 入站条码6
E0_9544 CHANNEL  ; 入站条码6
E0_9545 CHANNEL  ; 入站条码6
E0_9546 CHANNEL  ; 入站条码6
E0_9547 CHANNEL  ; 入站条码6
E0_9548 CHANNEL  ; 入站条码6
E0_9549 CHANNEL  ; 入站条码6
E0_9600 CHANNEL  ; 入站条码7
E0_9601 CHANNEL  ; 入站条码7
E0_9602 CHANNEL  ; 入站条码7
E0_9603 CHANNEL  ; 入站条码7
E0_9604 CHANNEL  ; 入站条码7
E0_9605 CHANNEL  ; 入站条码7
E0_9606 CHANNEL  ; 入站条码7
E0_9607 CHANNEL  ; 入站条码7
E0_9608 CHANNEL  ; 入站条码7
E0_9609 CHANNEL  ; 入站条码7
E0_9610 CHANNEL  ; 入站条码7
E0_9611 CHANNEL  ; 入站条码7
E0_9612 CHANNEL  ; 入站条码7
E0_9613 CHANNEL  ; 入站条码7
E0_9614 CHANNEL  ; 入站条码7
E0_9615 CHANNEL  ; 入站条码7
E0_9616 CHANNEL  ; 入站条码7
E0_9617 CHANNEL  ; 入站条码7
E0_9618 CHANNEL  ; 入站条码7
E0_9619 CHANNEL  ; 入站条码7
E0_9620 CHANNEL  ; 入站条码7
E0_9621 CHANNEL  ; 入站条码7
E0_9622 CHANNEL  ; 入站条码7
E0_9623 CHANNEL  ; 入站条码7
E0_9624 CHANNEL  ; 入站条码7
E0_9625 CHANNEL  ; 入站条码7
E0_9626 CHANNEL  ; 入站条码7
E0_9627 CHANNEL  ; 入站条码7
E0_9628 CHANNEL  ; 入站条码7
E0_9629 CHANNEL  ; 入站条码7
E0_9630 CHANNEL  ; 入站条码7
E0_9631 CHANNEL  ; 入站条码7
E0_9632 CHANNEL  ; 入站条码7
E0_9633 CHANNEL  ; 入站条码7
E0_9634 CHANNEL  ; 入站条码7
E0_9635 CHANNEL  ; 入站条码7
E0_9636 CHANNEL  ; 入站条码7
E0_9637 CHANNEL  ; 入站条码7
E0_9638 CHANNEL  ; 入站条码7
E0_9639 CHANNEL  ; 入站条码7
E0_9640 CHANNEL  ; 入站条码7
E0_9641 CHANNEL  ; 入站条码7
E0_9642 CHANNEL  ; 入站条码7
E0_9643 CHANNEL  ; 入站条码7
E0_9644 CHANNEL  ; 入站条码7
E0_9645 CHANNEL  ; 入站条码7
E0_9646 CHANNEL  ; 入站条码7
E0_9647 CHANNEL  ; 入站条码7
E0_9648 CHANNEL  ; 入站条码7
E0_9649 CHANNEL  ; 入站条码7
E0_9700 CHANNEL  ; 入站条码8
E0_9701 CHANNEL  ; 入站条码8
E0_9702 CHANNEL  ; 入站条码8
E0_9703 CHANNEL  ; 入站条码8
E0_9704 CHANNEL  ; 入站条码8
E0_9705 CHANNEL  ; 入站条码8
E0_9706 CHANNEL  ; 入站条码8
E0_9707 CHANNEL  ; 入站条码8
E0_9708 CHANNEL  ; 入站条码8
E0_9709 CHANNEL  ; 入站条码8
E0_9710 CHANNEL  ; 入站条码8
E0_9711 CHANNEL  ; 入站条码8
E0_9712 CHANNEL  ; 入站条码8
E0_9713 CHANNEL  ; 入站条码8
E0_9714 CHANNEL  ; 入站条码8
E0_9715 CHANNEL  ; 入站条码8
E0_9716 CHANNEL  ; 入站条码8
E0_9717 CHANNEL  ; 入站条码8
E0_9718 CHANNEL  ; 入站条码8
E0_9719 CHANNEL  ; 入站条码8
E0_9720 CHANNEL  ; 入站条码8
E0_9721 CHANNEL  ; 入站条码8
E0_9722 CHANNEL  ; 入站条码8
E0_9723 CHANNEL  ; 入站条码8
E0_9724 CHANNEL  ; 入站条码8
E0_9725 CHANNEL  ; 入站条码8
E0_9726 CHANNEL  ; 入站条码8
E0_9727 CHANNEL  ; 入站条码8
E0_9728 CHANNEL  ; 入站条码8
E0_9729 CHANNEL  ; 入站条码8
E0_9730 CHANNEL  ; 入站条码8
E0_9731 CHANNEL  ; 入站条码8
E0_9732 CHANNEL  ; 入站条码8
E0_9733 CHANNEL  ; 入站条码8
E0_9734 CHANNEL  ; 入站条码8
E0_9735 CHANNEL  ; 入站条码8
E0_9736 CHANNEL  ; 入站条码8
E0_9737 CHANNEL  ; 入站条码8
E0_9738 CHANNEL  ; 入站条码8
E0_9739 CHANNEL  ; 入站条码8
E0_9740 CHANNEL  ; 入站条码8
E0_9741 CHANNEL  ; 入站条码8
E0_9742 CHANNEL  ; 入站条码8
E0_9743 CHANNEL  ; 入站条码8
E0_9744 CHANNEL  ; 入站条码8
E0_9745 CHANNEL  ; 入站条码8
E0_9746 CHANNEL  ; 入站条码8
E0_9747 CHANNEL  ; 入站条码8
E0_9748 CHANNEL  ; 入站条码8
E0_9749 CHANNEL  ; 入站条码8
E0_9800 CHANNEL  ; 入站条码9
E0_9801 CHANNEL  ; 入站条码9
E0_9802 CHANNEL  ; 入站条码9
E0_9803 CHANNEL  ; 入站条码9
E0_9804 CHANNEL  ; 入站条码9
E0_9805 CHANNEL  ; 入站条码9
E0_9806 CHANNEL  ; 入站条码9
E0_9807 CHANNEL  ; 入站条码9
E0_9808 CHANNEL  ; 入站条码9
E0_9809 CHANNEL  ; 入站条码9
E0_9810 CHANNEL  ; 入站条码9
E0_9811 CHANNEL  ; 入站条码9
E0_9812 CHANNEL  ; 入站条码9
E0_9813 CHANNEL  ; 入站条码9
E0_9814 CHANNEL  ; 入站条码9
E0_9815 CHANNEL  ; 入站条码9
E0_9816 CHANNEL  ; 入站条码9
E0_9817 CHANNEL  ; 入站条码9
E0_9818 CHANNEL  ; 入站条码9
E0_9819 CHANNEL  ; 入站条码9
E0_9820 CHANNEL  ; 入站条码9
E0_9821 CHANNEL  ; 入站条码9
E0_9822 CHANNEL  ; 入站条码9
E0_9823 CHANNEL  ; 入站条码9
E0_9824 CHANNEL  ; 入站条码9
E0_9825 CHANNEL  ; 入站条码9
E0_9826 CHANNEL  ; 入站条码9
E0_9827 CHANNEL  ; 入站条码9
E0_9828 CHANNEL  ; 入站条码9
E0_9829 CHANNEL  ; 入站条码9
E0_9830 CHANNEL  ; 入站条码9
E0_9831 CHANNEL  ; 入站条码9
E0_9832 CHANNEL  ; 入站条码9
E0_9833 CHANNEL  ; 入站条码9
E0_9834 CHANNEL  ; 入站条码9
E0_9835 CHANNEL  ; 入站条码9
E0_9836 CHANNEL  ; 入站条码9
E0_9837 CHANNEL  ; 入站条码9
E0_9838 CHANNEL  ; 入站条码9
E0_9839 CHANNEL  ; 入站条码9
E0_9840 CHANNEL  ; 入站条码9
E0_9841 CHANNEL  ; 入站条码9
E0_9842 CHANNEL  ; 入站条码9
E0_9843 CHANNEL  ; 入站条码9
E0_9844 CHANNEL  ; 入站条码9
E0_9845 CHANNEL  ; 入站条码9
E0_9846 CHANNEL  ; 入站条码9
E0_9847 CHANNEL  ; 入站条码9
E0_9848 CHANNEL  ; 入站条码9
E0_9849 CHANNEL  ; 入站条码9
E0_9900 CHANNEL  ; 入站条码10
E0_9901 CHANNEL  ; 入站条码10
E0_9902 CHANNEL  ; 入站条码10
E0_9903 CHANNEL  ; 入站条码10
E0_9904 CHANNEL  ; 入站条码10
E0_9905 CHANNEL  ; 入站条码10
E0_9906 CHANNEL  ; 入站条码10
E0_9907 CHANNEL  ; 入站条码10
E0_9908 CHANNEL  ; 入站条码10
E0_9909 CHANNEL  ; 入站条码10
E0_9910 CHANNEL  ; 入站条码10
E0_9911 CHANNEL  ; 入站条码10
E0_9912 CHANNEL  ; 入站条码10
E0_9913 CHANNEL  ; 入站条码10
E0_9914 CHANNEL  ; 入站条码10
E0_9915 CHANNEL  ; 入站条码10
E0_9916 CHANNEL  ; 入站条码10
E0_9917 CHANNEL  ; 入站条码10
E0_9918 CHANNEL  ; 入站条码10
E0_9919 CHANNEL  ; 入站条码10
E0_9920 CHANNEL  ; 入站条码10
E0_9921 CHANNEL  ; 入站条码10
E0_9922 CHANNEL  ; 入站条码10
E0_9923 CHANNEL  ; 入站条码10
E0_9924 CHANNEL  ; 入站条码10
E0_9925 CHANNEL  ; 入站条码10
E0_9926 CHANNEL  ; 入站条码10
E0_9927 CHANNEL  ; 入站条码10
E0_9928 CHANNEL  ; 入站条码10
E0_9929 CHANNEL  ; 入站条码10
E0_9930 CHANNEL  ; 入站条码10
E0_9931 CHANNEL  ; 入站条码10
E0_9932 CHANNEL  ; 入站条码10
E0_9933 CHANNEL  ; 入站条码10
E0_9934 CHANNEL  ; 入站条码10
E0_9935 CHANNEL  ; 入站条码10
E0_9936 CHANNEL  ; 入站条码10
E0_9937 CHANNEL  ; 入站条码10
E0_9938 CHANNEL  ; 入站条码10
E0_9939 CHANNEL  ; 入站条码10
E0_9940 CHANNEL  ; 入站条码10
E0_9941 CHANNEL  ; 入站条码10
E0_9942 CHANNEL  ; 入站条码10
E0_9943 CHANNEL  ; 入站条码10
E0_9944 CHANNEL  ; 入站条码10
E0_9945 CHANNEL  ; 入站条码10
E0_9946 CHANNEL  ; 入站条码10
E0_9947 CHANNEL  ; 入站条码10
E0_9948 CHANNEL  ; 入站条码10
E0_9949 CHANNEL  ; 入站条码10
E1_0 CHANNEL  ; NC433_0 数据传送写字数
E1_1 CHANNEL  ; NC433_0 数据传送写源区域
E1_10 CHANNEL  ; NC433_0_X轴直接操作速度
E1_100 CHANNEL  ; NC433_1_Y轴存储器操作序列号
E1_1000 CHANNEL  ; 进出料横移伺服A自动速度
E1_1001 CHANNEL  ; 进出料横移伺服A自动速度
E1_1002 CHANNEL  ; 进出料横移伺服AJOG高速
E1_1003 CHANNEL  ; 进出料横移伺服AJOG高速
E1_1004 CHANNEL  ; 进出料横移伺服AJOG低速
E1_1005 CHANNEL  ; 进出料横移伺服AJOG低速
E1_1006 CHANNEL  ; 进出料横移伺服A加速时间
E1_1007 CHANNEL  ; 进出料横移伺服A加速时间
E1_1008 CHANNEL  ; 进出料横移伺服A减速时间
E1_1009 CHANNEL  ; 进出料横移伺服A减速时间
E1_101 CHANNEL  ; NC433_1_Y轴特殊操作Override
E1_1010 CHANNEL  ; 进出料横移伺服A原点偏移
E1_1011 CHANNEL  ; 进出料横移伺服A原点偏移
E1_1012 CHANNEL  ; 进出料横移伺服A正软极限
E1_1013 CHANNEL  ; 进出料横移伺服A正软极限
E1_1014 CHANNEL  ; 进出料横移伺服A负软极限
E1_1015 CHANNEL  ; 进出料横移伺服A负软极限
E1_102 CHANNEL  ; NC433_1_Y轴特殊操作示教地址
E1_1020 CHANNEL  ; 进出料横移伺服A进料位
E1_1021 CHANNEL  ; 进出料横移伺服A进料位
E1_1022 CHANNEL  ; 进出料横移伺服A进料等待位
E1_1023 CHANNEL  ; 进出料横移伺服A进料等待位
E1_1024 CHANNEL  ; 进出料横移伺服A上料位A
E1_1025 CHANNEL  ; 进出料横移伺服A上料位A
E1_1026 CHANNEL  ; 进出料横移伺服A上料位B
E1_1027 CHANNEL  ; 进出料横移伺服A上料位B
E1_1028 CHANNEL  ; 进出料横移伺服A下料位A
E1_1029 CHANNEL  ; 进出料横移伺服A下料位A
E1_103 CHANNEL  ; NC433_1_Y轴特殊操作预留
E1_1030 CHANNEL  ; 进出料横移伺服A下料位B
E1_1031 CHANNEL  ; 进出料横移伺服A下料位B
E1_1032 CHANNEL  ; 进出料横移伺服A出料等待位
E1_1033 CHANNEL  ; 进出料横移伺服A出料等待位
E1_1034 CHANNEL  ; 进出料横移伺服A出料位
E1_1035 CHANNEL  ; 进出料横移伺服A出料位
E1_1036 CHANNEL  ; 进出料横移伺服A9#位
E1_1037 CHANNEL  ; 进出料横移伺服A9#位
E1_1038 CHANNEL  ; 进出料横移伺服A10#位
E1_1039 CHANNEL  ; 进出料横移伺服A10#位
E1_104 CHANNEL  ; NC433_1_Z轴直接操作位置
E1_1040 CHANNEL  ; 进出料横移伺服A进料位_5
E1_1042 CHANNEL  ; 进出料横移伺服A进料等待位_5
E1_105 CHANNEL  ; NC433_1_Z轴直接操作位置
E1_1050 CHANNEL  ; 进出料伸缩伺服A自动速度
E1_1051 CHANNEL  ; 进出料伸缩伺服A自动速度
E1_1052 CHANNEL  ; 进出料伸缩伺服AJOG高速
E1_1053 CHANNEL  ; 进出料伸缩伺服AJOG高速
E1_1054 CHANNEL  ; 进出料伸缩伺服AJOG低速
E1_1055 CHANNEL  ; 进出料伸缩伺服AJOG低速
E1_1056 CHANNEL  ; 进出料伸缩伺服A加速时间
E1_1057 CHANNEL  ; 进出料伸缩伺服A加速时间
E1_1058 CHANNEL  ; 进出料伸缩伺服A减速时间
E1_1059 CHANNEL  ; 进出料伸缩伺服A减速时间
E1_106 CHANNEL  ; NC433_1_Z轴直接操作速度
E1_1060 CHANNEL  ; 进出料伸缩伺服A原点偏移
E1_1061 CHANNEL  ; 进出料伸缩伺服A原点偏移
E1_1062 CHANNEL  ; 进出料伸缩伺服A正软极限
E1_1063 CHANNEL  ; 进出料伸缩伺服A正软极限
E1_1064 CHANNEL  ; 进出料伸缩伺服A负软极限
E1_1065 CHANNEL  ; 负软极限
E1_107 CHANNEL  ; NC433_1_Z轴直接操作速度
E1_1070 CHANNEL  ; 进出料伸缩伺服A初始位
E1_1071 CHANNEL  ; 进出料伸缩伺服A初始位
E1_1072 CHANNEL  ; 进出料伸缩伺服A平台取料位
E1_1073 CHANNEL  ; 进出料伸缩伺服A平台取料位
E1_1074 CHANNEL  ; 进出料伸缩伺服A热压取放位
E1_1075 CHANNEL  ; 进出料伸缩伺服A热压取放位
E1_1076 CHANNEL  ; 进出料伸缩伺服A平台放料位
E1_1077 CHANNEL  ; 进出料伸缩伺服A平台放料位
E1_1078 CHANNEL  ; 进出料伸缩伺服A5#位
E1_1079 CHANNEL  ; 进出料伸缩伺服A5#位
E1_108 CHANNEL  ; NC433_1_Z轴直接操作加速时间
E1_1080 CHANNEL  ; 进出料伸缩伺服A6#位
E1_1081 CHANNEL  ; 进出料伸缩伺服A6#位
E1_1082 CHANNEL  ; 进出料伸缩伺服A7#位
E1_1083 CHANNEL  ; 进出料伸缩伺服A7#位
E1_1084 CHANNEL  ; 进出料伸缩伺服A8#位
E1_1085 CHANNEL  ; 进出料伸缩伺服A8#位
E1_1086 CHANNEL  ; 进出料伸缩伺服A9#位
E1_1087 CHANNEL  ; 进出料伸缩伺服A9#位
E1_1088 CHANNEL  ; 进出料伸缩伺服A10#位
E1_1089 CHANNEL  ; 进出料伸缩伺服A10#位
E1_109 CHANNEL  ; NC433_1_Z轴直接操作加速时间
E1_11 CHANNEL  ; NC433_0_X轴直接操作速度
E1_110 CHANNEL  ; NC433_1_Z轴直接操作减速时间
E1_1100 CHANNEL  ; 进出料横移伺服B自动速度
E1_1101 CHANNEL  ; 进出料横移伺服B自动速度
E1_1102 CHANNEL  ; 进出料横移伺服BJOG高速
E1_1103 CHANNEL  ; 进出料横移伺服BJOG高速
E1_1104 CHANNEL  ; 进出料横移伺服BJOG低速
E1_1105 CHANNEL  ; 进出料横移伺服BJOG低速
E1_1106 CHANNEL  ; 进出料横移伺服B加速时间
E1_1107 CHANNEL  ; 进出料横移伺服B加速时间
E1_1108 CHANNEL  ; 进出料横移伺服B减速时间
E1_1109 CHANNEL  ; 进出料横移伺服B减速时间
E1_111 CHANNEL  ; NC433_1_Z轴直接操作减速时间
E1_1110 CHANNEL  ; 进出料横移伺服B原点偏移
E1_1111 CHANNEL  ; 进出料横移伺服B原点偏移
E1_1112 CHANNEL  ; 进出料横移伺服B正软极限
E1_1113 CHANNEL  ; 进出料横移伺服B正软极限
E1_1114 CHANNEL  ; 进出料横移伺服B负软极限
E1_1115 CHANNEL  ; 负软极限
E1_112 CHANNEL  ; NC433_1_Z轴存储器操作序列号
E1_1120 CHANNEL  ; 进出料横移伺服B进料位
E1_1121 CHANNEL  ; 进出料横移伺服B进料位
E1_1122 CHANNEL  ; 进出料横移伺服B进料等待位
E1_1123 CHANNEL  ; 进出料横移伺服B进料等待位
E1_1124 CHANNEL  ; 进出料横移伺服B上料位A
E1_1125 CHANNEL  ; 进出料横移伺服B上料位A
E1_1126 CHANNEL  ; 进出料横移伺服B上料位B
E1_1127 CHANNEL  ; 进出料横移伺服B上料位B
E1_1128 CHANNEL  ; 进出料横移伺服B下料位A
E1_1129 CHANNEL  ; 进出料横移伺服B下料位A
E1_113 CHANNEL  ; NC433_1_Z轴特殊操作Override
E1_1130 CHANNEL  ; 进出料横移伺服B下料位B
E1_1131 CHANNEL  ; 进出料横移伺服B下料位B
E1_1132 CHANNEL  ; 进出料横移伺服B出料等待位
E1_1133 CHANNEL  ; 进出料横移伺服B出料等待位
E1_1134 CHANNEL  ; 进出料横移伺服B出料位
E1_1135 CHANNEL  ; 进出料横移伺服B出料位
E1_1136 CHANNEL  ; 进出料横移伺服B9#位
E1_1137 CHANNEL  ; 进出料横移伺服B9#位
E1_1138 CHANNEL  ; 进出料横移伺服B10#位
E1_1139 CHANNEL  ; 进出料横移伺服B10#位
E1_114 CHANNEL  ; NC433_1_Z轴特殊操作示教地址
E1_115 CHANNEL  ; NC433_1_Z轴特殊操作预留
E1_1150 CHANNEL  ; 进出料伸缩伺服B自动速度
E1_1151 CHANNEL  ; 进出料伸缩伺服B自动速度
E1_1152 CHANNEL  ; 进出料伸缩伺服BJOG高速
E1_1153 CHANNEL  ; 进出料伸缩伺服BJOG高速
E1_1154 CHANNEL  ; 进出料伸缩伺服BJOG低速
E1_1155 CHANNEL  ; 进出料伸缩伺服BJOG低速
E1_1156 CHANNEL  ; 进出料伸缩伺服B加速时间
E1_1157 CHANNEL  ; 进出料伸缩伺服B加速时间
E1_1158 CHANNEL  ; 进出料伸缩伺服B减速时间
E1_1159 CHANNEL  ; 进出料伸缩伺服B减速时间
E1_116 CHANNEL  ; NC433_1_U轴直接操作位置
E1_1160 CHANNEL  ; 进出料伸缩伺服B原点偏移
E1_1161 CHANNEL  ; 进出料伸缩伺服B原点偏移
E1_1162 CHANNEL  ; 进出料伸缩伺服B正软极限
E1_1163 CHANNEL  ; 进出料伸缩伺服B正软极限
E1_1164 CHANNEL  ; 进出料伸缩伺服B负软极限
E1_1165 CHANNEL  ; 负软极限
E1_117 CHANNEL  ; NC433_1_U轴直接操作位置
E1_1170 CHANNEL  ; 进出料伸缩伺服B初始位
E1_1171 CHANNEL  ; 进出料伸缩伺服B初始位
E1_1172 CHANNEL  ; 进出料伸缩伺服B平台取料位
E1_1173 CHANNEL  ; 进出料伸缩伺服B平台取料位
E1_1174 CHANNEL  ; 进出料伸缩伺服B热压取放位
E1_1175 CHANNEL  ; 进出料伸缩伺服B热压取放位
E1_1176 CHANNEL  ; 进出料伸缩伺服B平台放料位
E1_1177 CHANNEL  ; 进出料伸缩伺服B平台放料位
E1_1178 CHANNEL  ; 进出料伸缩伺服B5#位
E1_1179 CHANNEL  ; 进出料伸缩伺服B5#位
E1_118 CHANNEL  ; NC433_1_U轴直接操作速度
E1_1180 CHANNEL  ; 进出料伸缩伺服B6#位
E1_1181 CHANNEL  ; 进出料伸缩伺服B6#位
E1_1182 CHANNEL  ; 进出料伸缩伺服B7#位
E1_1183 CHANNEL  ; 进出料伸缩伺服B7#位
E1_1184 CHANNEL  ; 进出料伸缩伺服B8#位
E1_1185 CHANNEL  ; 进出料伸缩伺服B8#位
E1_1186 CHANNEL  ; 进出料伸缩伺服B9#位
E1_1187 CHANNEL  ; 进出料伸缩伺服B9#位
E1_1188 CHANNEL  ; 进出料伸缩伺服B10#位
E1_1189 CHANNEL  ; 进出料伸缩伺服B10#位
E1_119 CHANNEL  ; NC433_1_U轴直接操作速度
E1_12 CHANNEL  ; NC433_0_X轴直接操作加速时间
E1_120 CHANNEL  ; NC433_1_U轴直接操作加速时间
E1_1200 CHANNEL  ; 正压伺服A自动速度
E1_1201 CHANNEL  ; 正压伺服A自动速度
E1_1202 CHANNEL  ; 正压伺服AJOG高速
E1_1203 CHANNEL  ; 正压伺服AJOG高速
E1_1204 CHANNEL  ; 正压伺服AJOG低速
E1_1205 CHANNEL  ; 正压伺服AJOG低速
E1_1206 CHANNEL  ; 正压伺服A加速时间
E1_1207 CHANNEL  ; 正压伺服A加速时间
E1_1208 CHANNEL  ; 正压伺服A减速时间
E1_1209 CHANNEL  ; 正压伺服A减速时间
E1_121 CHANNEL  ; NC433_1_U轴直接操作加速时间
E1_1210 CHANNEL  ; 正压伺服A原点偏移
E1_1211 CHANNEL  ; 正压伺服A原点偏移
E1_1212 CHANNEL  ; 正压伺服A正软极限
E1_1213 CHANNEL  ; 正压伺服A正软极限
E1_1214 CHANNEL  ; 正压伺服A负软极限
E1_1215 CHANNEL  ; 负软极限
E1_1218 CHANNEL  ; 正压伺服A动态减速位
E1_122 CHANNEL  ; NC433_1_U轴直接操作减速时间
E1_1220 CHANNEL  ; 正压伺服A初始位
E1_1221 CHANNEL  ; 正压伺服A初始位
E1_1222 CHANNEL  ; 正压伺服A减速位
E1_1223 CHANNEL  ; 正压伺服A减速位
E1_1224 CHANNEL  ; 正压伺服A等距热压位
E1_1225 CHANNEL  ; 正压伺服A等距热压位
E1_1226 CHANNEL  ; 正压伺服A预压退回位
E1_1227 CHANNEL  ; 正压伺服A预压退回位
E1_1228 CHANNEL  ; 正压伺服AMASK测试位
E1_1229 CHANNEL  ; 正压伺服AMASK测试位
E1_123 CHANNEL  ; NC433_1_U轴直接操作减速时间
E1_1230 CHANNEL  ; 正压伺服A6#位
E1_1231 CHANNEL  ; 正压伺服A6#位
E1_1232 CHANNEL  ; 正压伺服A7#位
E1_1233 CHANNEL  ; 正压伺服A7#位
E1_1234 CHANNEL  ; 正压伺服A8#位
E1_1235 CHANNEL  ; 正压伺服A8#位
E1_1236 CHANNEL  ; 正压伺服A9#位
E1_1237 CHANNEL  ; 正压伺服A9#位
E1_1238 CHANNEL  ; 正压伺服A10#位
E1_1239 CHANNEL  ; 正压伺服A10#位
E1_124 CHANNEL  ; NC433_1_U轴存储器操作序列号
E1_1240 CHANNEL  ; 正压伺服A相对位移量
E1_1244 CHANNEL  ; 正压保护位
E1_1246 CHANNEL  ; A工位无料层高差
E1_125 CHANNEL  ; NC433_1_U轴特殊操作Override
E1_1250 CHANNEL  ; 压板平移伺服A自动速度
E1_1251 CHANNEL  ; 压板平移伺服A自动速度
E1_1252 CHANNEL  ; 压板平移伺服AJOG高速
E1_1253 CHANNEL  ; 压板平移伺服AJOG高速
E1_1254 CHANNEL  ; 压板平移伺服AJOG低速
E1_1255 CHANNEL  ; 压板平移伺服AJOG低速
E1_1256 CHANNEL  ; 压板平移伺服A加速时间
E1_1257 CHANNEL  ; 压板平移伺服A加速时间
E1_1258 CHANNEL  ; 压板平移伺服A减速时间
E1_1259 CHANNEL  ; 压板平移伺服A减速时间
E1_126 CHANNEL  ; NC433_1_U轴特殊操作示教地址
E1_1260 CHANNEL  ; 压板平移伺服A原点偏移
E1_1261 CHANNEL  ; 压板平移伺服A原点偏移
E1_1262 CHANNEL  ; 压板平移伺服A正软极限
E1_1263 CHANNEL  ; 压板平移伺服A正软极限
E1_1264 CHANNEL  ; 压板平移伺服A负软极限
E1_1265 CHANNEL  ; 负软极限
E1_127 CHANNEL  ; NC433_1_U轴特殊操作预留
E1_1270 CHANNEL  ; 压板平移伺服AA面取放位
E1_1271 CHANNEL  ; 压板平移伺服AA面取放位
E1_1272 CHANNEL  ; 压板平移伺服AB面取放位
E1_1273 CHANNEL  ; 压板平移伺服AB面取放位
E1_1274 CHANNEL  ; 压板平移伺服A3#位
E1_1275 CHANNEL  ; 压板平移伺服A3#位
E1_1276 CHANNEL  ; 压板平移伺服A4#位
E1_1277 CHANNEL  ; 压板平移伺服A4#位
E1_1278 CHANNEL  ; 压板平移伺服A5#位
E1_1279 CHANNEL  ; 压板平移伺服A5#位
E1_128 CHANNEL  ; NC433_1_X轴当前位置
E1_1280 CHANNEL  ; 压板平移伺服A6#位
E1_1281 CHANNEL  ; 压板平移伺服A6#位
E1_1282 CHANNEL  ; 压板平移伺服A7#位
E1_1283 CHANNEL  ; 压板平移伺服A7#位
E1_1284 CHANNEL  ; 压板平移伺服A8#位
E1_1285 CHANNEL  ; 压板平移伺服A8#位
E1_1286 CHANNEL  ; 压板平移伺服A9#位
E1_1287 CHANNEL  ; 压板平移伺服A9#位
E1_1288 CHANNEL  ; 压板平移伺服A10#位
E1_1289 CHANNEL  ; 压板平移伺服A10#位
E1_129 CHANNEL  ; NC433_1_X轴当前位置
E1_13 CHANNEL  ; NC433_0_X轴直接操作加速时间
E1_130 CHANNEL  ; NC433_1_X轴存储器操作正被执行序列号
E1_1300 CHANNEL  ; 侧压A1左伺服自动速度
E1_1301 CHANNEL  ; 侧压A1左伺服自动速度
E1_1302 CHANNEL  ; 侧压A1左伺服JOG高速
E1_1303 CHANNEL  ; 侧压A1左伺服JOG高速
E1_1304 CHANNEL  ; 侧压A1左伺服JOG低速
E1_1305 CHANNEL  ; 侧压A1左伺服JOG低速
E1_1306 CHANNEL  ; 侧压A1左伺服加速时间
E1_1307 CHANNEL  ; 侧压A1左伺服加速时间
E1_1308 CHANNEL  ; 侧压A1左伺服减速时间
E1_1309 CHANNEL  ; 侧压A1左伺服减速时间
E1_131 CHANNEL  ; NC433_1_X轴存储器操作正被执行序列号
E1_1310 CHANNEL  ; 侧压A1左伺服原点偏移
E1_1311 CHANNEL  ; 侧压A1左伺服原点偏移
E1_1312 CHANNEL  ; 侧压A1左伺服正软极限
E1_1313 CHANNEL  ; 侧压A1左伺服正软极限
E1_1314 CHANNEL  ; 侧压A1左伺服负软极限
E1_1315 CHANNEL  ; 负软极限
E1_132 CHANNEL  ; NC433_1_Y轴当前位置
E1_1320 CHANNEL  ; 侧压A1左伺服待机位
E1_1321 CHANNEL  ; 侧压A1左伺服待机位
E1_1322 CHANNEL  ; 侧压A1左伺服拨料退回位
E1_1323 CHANNEL  ; 侧压A1左伺服拨料退回位
E1_1324 CHANNEL  ; 侧压A1左伺服拨料位
E1_1325 CHANNEL  ; 侧压A1左伺服拨料位
E1_1326 CHANNEL  ; 侧压A1左伺服减速位
E1_1327 CHANNEL  ; 侧压A1左伺服减速位
E1_1328 CHANNEL  ; 侧压A1左伺服等距热压位
E1_1329 CHANNEL  ; 侧压A1左伺服等距热压位
E1_133 CHANNEL  ; NC433_1_Y轴当前位置
E1_1330 CHANNEL  ; 侧压A1左伺服6#位
E1_1331 CHANNEL  ; 侧压A1左伺服6#位
E1_1332 CHANNEL  ; 侧压A1左伺服7#位
E1_1333 CHANNEL  ; 侧压A1左伺服7#位
E1_1334 CHANNEL  ; 侧压A1左伺服8#位
E1_1335 CHANNEL  ; 侧压A1左伺服8#位
E1_1336 CHANNEL  ; 侧压A1左伺服9#位
E1_1337 CHANNEL  ; 侧压A1左伺服9#位
E1_1338 CHANNEL  ; 侧压A1左伺服10#位
E1_1339 CHANNEL  ; 侧压A1左伺服10#位
E1_134 CHANNEL  ; NC433_1_Y轴存储器操作正被执行序列号
E1_1340 CHANNEL  ; A1左伺服相对移位量
E1_1346 CHANNEL  ; A1两轴回原宽度
E1_135 CHANNEL  ; NC433_1_Y轴存储器操作正被执行序列号
E1_1350 CHANNEL  ; 侧压A1右伺服自动速度
E1_1351 CHANNEL  ; 侧压A1右伺服自动速度
E1_1352 CHANNEL  ; 侧压A1右伺服JOG高速
E1_1353 CHANNEL  ; 侧压A1右伺服JOG高速
E1_1354 CHANNEL  ; 侧压A1右伺服JOG低速
E1_1355 CHANNEL  ; 侧压A1右伺服JOG低速
E1_1356 CHANNEL  ; 侧压A1右伺服加速时间
E1_1357 CHANNEL  ; 侧压A1右伺服加速时间
E1_1358 CHANNEL  ; 侧压A1右伺服减速时间
E1_1359 CHANNEL  ; 侧压A1右伺服减速时间
E1_136 CHANNEL  ; NC433_1_Z轴当前位置
E1_1360 CHANNEL  ; 侧压A1右伺服原点偏移
E1_1361 CHANNEL  ; 侧压A1右伺服原点偏移
E1_1362 CHANNEL  ; 侧压A1右伺服正软极限
E1_1363 CHANNEL  ; 侧压A1右伺服正软极限
E1_1364 CHANNEL  ; 侧压A1右伺服负软极限
E1_1365 CHANNEL  ; 负软极限
E1_137 CHANNEL  ; NC433_1_Z轴当前位置
E1_1370 CHANNEL  ; 侧压A1右伺服待机位
E1_1371 CHANNEL  ; 侧压A1右伺服待机位
E1_1372 CHANNEL  ; 侧压A1右伺服拨料退回位
E1_1373 CHANNEL  ; 侧压A1右伺服拨料退回位
E1_1374 CHANNEL  ; 侧压A1右伺服拨料位
E1_1375 CHANNEL  ; 侧压A1右伺服拨料位
E1_1376 CHANNEL  ; 侧压A1右伺服减速位
E1_1377 CHANNEL  ; 侧压A1右伺服减速位
E1_1378 CHANNEL  ; 侧压A1右伺服等距热压位
E1_1379 CHANNEL  ; 侧压A1右伺服等距热压位
E1_138 CHANNEL  ; NC433_1_Z轴存储器操作正被执行序列号
E1_1380 CHANNEL  ; 侧压A1右伺服6#位
E1_1381 CHANNEL  ; 侧压A1右伺服6#位
E1_1382 CHANNEL  ; 侧压A1右伺服7#位
E1_1383 CHANNEL  ; 侧压A1右伺服7#位
E1_1384 CHANNEL  ; 侧压A1右伺服8#位
E1_1385 CHANNEL  ; 侧压A1右伺服8#位
E1_1386 CHANNEL  ; 侧压A1右伺服9#位
E1_1387 CHANNEL  ; 侧压A1右伺服9#位
E1_1388 CHANNEL  ; 侧压A1右伺服10#位
E1_1389 CHANNEL  ; 侧压A1右伺服10#位
E1_139 CHANNEL  ; NC433_1_Z轴存储器操作正被执行序列号
E1_1390 CHANNEL  ; A1右伺服相对移动量
E1_14 CHANNEL  ; NC433_0_X轴直接操作减速时间
E1_140 CHANNEL  ; NC433_1_U轴当前位置
E1_1400 CHANNEL  ; 侧压A2左伺服自动速度
E1_1401 CHANNEL  ; 侧压A2左伺服自动速度
E1_1402 CHANNEL  ; 侧压A2左伺服JOG高速
E1_1403 CHANNEL  ; 侧压A2左伺服JOG高速
E1_1404 CHANNEL  ; 侧压A2左伺服JOG低速
E1_1405 CHANNEL  ; 侧压A2左伺服JOG低速
E1_1406 CHANNEL  ; 侧压A2左伺服加速时间
E1_1407 CHANNEL  ; 侧压A2左伺服加速时间
E1_1408 CHANNEL  ; 侧压A2左伺服减速时间
E1_1409 CHANNEL  ; 侧压A2左伺服减速时间
E1_141 CHANNEL  ; NC433_1_U轴当前位置
E1_1410 CHANNEL  ; 侧压A2左伺服原点偏移
E1_1411 CHANNEL  ; 侧压A2左伺服原点偏移
E1_1412 CHANNEL  ; 侧压A2左伺服正软极限
E1_1413 CHANNEL  ; 侧压A2左伺服正软极限
E1_1414 CHANNEL  ; 侧压A2左伺服负软极限
E1_1415 CHANNEL  ; 负软极限
E1_142 CHANNEL  ; NC433_1_U轴存储器操作正被执行序列号
E1_1420 CHANNEL  ; 侧压A2左伺服待机位
E1_1421 CHANNEL  ; 侧压A2左伺服待机位
E1_1422 CHANNEL  ; 侧压A2左伺服拨料退回位
E1_1423 CHANNEL  ; 侧压A2左伺服拨料退回位
E1_1424 CHANNEL  ; 侧压A2左伺服拨料位
E1_1425 CHANNEL  ; 侧压A2左伺服拨料位
E1_1426 CHANNEL  ; 侧压A2左伺服减速位
E1_1427 CHANNEL  ; 侧压A2左伺服减速位
E1_1428 CHANNEL  ; 侧压A2左伺服等距热压位
E1_1429 CHANNEL  ; 侧压A2左伺服等距热压位
E1_143 CHANNEL  ; NC433_1_U轴存储器操作正被执行序列号
E1_1430 CHANNEL  ; 侧压A2左伺服6#位
E1_1431 CHANNEL  ; 侧压A2左伺服6#位
E1_1432 CHANNEL  ; 侧压A2左伺服7#位
E1_1433 CHANNEL  ; 侧压A2左伺服7#位
E1_1434 CHANNEL  ; 侧压A2左伺服8#位
E1_1435 CHANNEL  ; 侧压A2左伺服8#位
E1_1436 CHANNEL  ; 侧压A2左伺服9#位
E1_1437 CHANNEL  ; 侧压A2左伺服9#位
E1_1438 CHANNEL  ; 侧压A2左伺服10#位
E1_1439 CHANNEL  ; 侧压A2左伺服10#位
E1_144 CHANNEL  ; NC433_2 数据传送写字数
E1_1446 CHANNEL  ; A2两轴回原宽度
E1_145 CHANNEL  ; NC433_2 数据传送写源区域
E1_1450 CHANNEL  ; 侧压A2右伺服自动速度
E1_1451 CHANNEL  ; 侧压A2右伺服自动速度
E1_1452 CHANNEL  ; 侧压A2右伺服JOG高速
E1_1453 CHANNEL  ; 侧压A2右伺服JOG高速
E1_1454 CHANNEL  ; 侧压A2右伺服JOG低速
E1_1455 CHANNEL  ; 侧压A2右伺服JOG低速
E1_1456 CHANNEL  ; 侧压A2右伺服加速时间
E1_1457 CHANNEL  ; 侧压A2右伺服加速时间
E1_1458 CHANNEL  ; 侧压A2右伺服减速时间
E1_1459 CHANNEL  ; 侧压A2右伺服减速时间
E1_146 CHANNEL  ; NC433_2 数据传送定源字
E1_1460 CHANNEL  ; 侧压A2右伺服原点偏移
E1_1461 CHANNEL  ; 侧压A2右伺服原点偏移
E1_1462 CHANNEL  ; 侧压A2右伺服正软极限
E1_1463 CHANNEL  ; 侧压A2右伺服正软极限
E1_1464 CHANNEL  ; 侧压A2右伺服负软极限
E1_1465 CHANNEL  ; 负软极限
E1_147 CHANNEL  ; NC433_2 数据传送定目标地址
E1_1470 CHANNEL  ; 侧压A2右伺服待机位
E1_1471 CHANNEL  ; 侧压A2右伺服待机位
E1_1472 CHANNEL  ; 侧压A2右伺服拨料退回位
E1_1473 CHANNEL  ; 侧压A2右伺服拨料退回位
E1_1474 CHANNEL  ; 侧压A2右伺服拨料位
E1_1475 CHANNEL  ; 侧压A2右伺服拨料位
E1_1476 CHANNEL  ; 侧压A2右伺服减速位
E1_1477 CHANNEL  ; 侧压A2右伺服减速位
E1_1478 CHANNEL  ; 侧压A2右伺服等距热压位
E1_1479 CHANNEL  ; 侧压A2右伺服等距热压位
E1_148 CHANNEL  ; NC433_2 数据传送读字数
E1_1480 CHANNEL  ; 侧压A2右伺服6#位
E1_1481 CHANNEL  ; 侧压A2右伺服6#位
E1_1482 CHANNEL  ; 侧压A2右伺服7#位
E1_1483 CHANNEL  ; 侧压A2右伺服7#位
E1_1484 CHANNEL  ; 侧压A2右伺服8#位
E1_1485 CHANNEL  ; 侧压A2右伺服8#位
E1_1486 CHANNEL  ; 侧压A2右伺服9#位
E1_1487 CHANNEL  ; 侧压A2右伺服9#位
E1_1488 CHANNEL  ; 侧压A2右伺服10#位
E1_1489 CHANNEL  ; 侧压A2右伺服10#位
E1_149 CHANNEL  ; NC433_2 数据传送读源区域
E1_15 CHANNEL  ; NC433_0_X轴直接操作减速时间
E1_150 CHANNEL  ; NC433_2 数据传送读目标区域
E1_1500 CHANNEL  ; 侧压A3左伺服自动速度
E1_1501 CHANNEL  ; 侧压A3左伺服自动速度
E1_1502 CHANNEL  ; 侧压A3左伺服JOG高速
E1_1503 CHANNEL  ; 侧压A3左伺服JOG高速
E1_1504 CHANNEL  ; 侧压A3左伺服JOG低速
E1_1505 CHANNEL  ; 侧压A3左伺服JOG低速
E1_1506 CHANNEL  ; 侧压A3左伺服加速时间
E1_1507 CHANNEL  ; 侧压A3左伺服加速时间
E1_1508 CHANNEL  ; 侧压A3左伺服减速时间
E1_1509 CHANNEL  ; 侧压A3左伺服减速时间
E1_151 CHANNEL  ; NC433_2 数据传送读目标字
E1_1510 CHANNEL  ; 侧压A3左伺服原点偏移
E1_1511 CHANNEL  ; 侧压A3左伺服原点偏移
E1_1512 CHANNEL  ; 侧压A3左伺服正软极限
E1_1513 CHANNEL  ; 侧压A3左伺服正软极限
E1_1514 CHANNEL  ; 侧压A3左伺服负软极限
E1_1515 CHANNEL  ; 负软极限
E1_152 CHANNEL  ; NC433_2_X轴直接操作位置
E1_1520 CHANNEL  ; 侧压A3左伺服待机位
E1_1521 CHANNEL  ; 侧压A3左伺服待机位
E1_1522 CHANNEL  ; 侧压A3左伺服拨料退回位
E1_1523 CHANNEL  ; 侧压A3左伺服拨料退回位
E1_1524 CHANNEL  ; 侧压A3左伺服拨料位
E1_1525 CHANNEL  ; 侧压A3左伺服拨料位
E1_1526 CHANNEL  ; 侧压A3左伺服减速位
E1_1527 CHANNEL  ; 侧压A3左伺服减速位
E1_1528 CHANNEL  ; 侧压A3左伺服等距热压位
E1_1529 CHANNEL  ; 侧压A3左伺服等距热压位
E1_153 CHANNEL  ; NC433_2_X轴直接操作位置
E1_1530 CHANNEL  ; 侧压A3左伺服6#位
E1_1531 CHANNEL  ; 侧压A3左伺服6#位
E1_1532 CHANNEL  ; 侧压A3左伺服7#位
E1_1533 CHANNEL  ; 侧压A3左伺服7#位
E1_1534 CHANNEL  ; 侧压A3左伺服8#位
E1_1535 CHANNEL  ; 侧压A3左伺服8#位
E1_1536 CHANNEL  ; 侧压A3左伺服9#位
E1_1537 CHANNEL  ; 侧压A3左伺服9#位
E1_1538 CHANNEL  ; 侧压A3左伺服10#位
E1_1539 CHANNEL  ; 侧压A3左伺服10#位
E1_154 CHANNEL  ; NC433_2_X轴直接操作速度
E1_1546 CHANNEL  ; A3两轴回原宽度
E1_155 CHANNEL  ; NC433_2_X轴直接操作速度
E1_1550 CHANNEL  ; 侧压A3右伺服自动速度
E1_1551 CHANNEL  ; 侧压A3右伺服自动速度
E1_1552 CHANNEL  ; 侧压A3右伺服JOG高速
E1_1553 CHANNEL  ; 侧压A3右伺服JOG高速
E1_1554 CHANNEL  ; 侧压A3右伺服JOG低速
E1_1555 CHANNEL  ; 侧压A3右伺服JOG低速
E1_1556 CHANNEL  ; 侧压A3右伺服加速时间
E1_1557 CHANNEL  ; 侧压A3右伺服加速时间
E1_1558 CHANNEL  ; 侧压A3右伺服减速时间
E1_1559 CHANNEL  ; 侧压A3右伺服减速时间
E1_156 CHANNEL  ; NC433_2_X轴直接操作加速时间
E1_1560 CHANNEL  ; 侧压A3右伺服原点偏移
E1_1561 CHANNEL  ; 侧压A3右伺服原点偏移
E1_1562 CHANNEL  ; 侧压A3右伺服正软极限
E1_1563 CHANNEL  ; 侧压A3右伺服正软极限
E1_1564 CHANNEL  ; 侧压A3右伺服负软极限
E1_1565 CHANNEL  ; 负软极限
E1_157 CHANNEL  ; NC433_2_X轴直接操作加速时间
E1_1570 CHANNEL  ; 侧压A3右伺服待机位
E1_1571 CHANNEL  ; 侧压A3右伺服待机位
E1_1572 CHANNEL  ; 侧压A3右伺服拨料退回位
E1_1573 CHANNEL  ; 侧压A3右伺服拨料退回位
E1_1574 CHANNEL  ; 侧压A3右伺服拨料位
E1_1575 CHANNEL  ; 侧压A3右伺服拨料位
E1_1576 CHANNEL  ; 侧压A3右伺服减速位
E1_1577 CHANNEL  ; 侧压A3右伺服减速位
E1_1578 CHANNEL  ; 侧压A3右伺服等距热压位
E1_1579 CHANNEL  ; 侧压A3右伺服等距热压位
E1_158 CHANNEL  ; NC433_2_X轴直接操作减速时间
E1_1580 CHANNEL  ; 侧压A3右伺服6#位
E1_1581 CHANNEL  ; 侧压A3右伺服6#位
E1_1582 CHANNEL  ; 侧压A3右伺服7#位
E1_1583 CHANNEL  ; 侧压A3右伺服7#位
E1_1584 CHANNEL  ; 侧压A3右伺服8#位
E1_1585 CHANNEL  ; 侧压A3右伺服8#位
E1_1586 CHANNEL  ; 侧压A3右伺服9#位
E1_1587 CHANNEL  ; 侧压A3右伺服9#位
E1_1588 CHANNEL  ; 侧压A3右伺服10#位
E1_1589 CHANNEL  ; 侧压A3右伺服10#位
E1_159 CHANNEL  ; NC433_2_X轴直接操作减速时间
E1_16 CHANNEL  ; NC433_0_X轴存储器操作序列号
E1_160 CHANNEL  ; NC433_2_X轴存储器操作序列号
E1_1600 CHANNEL  ; 侧压A4左伺服自动速度
E1_1601 CHANNEL  ; 侧压A4左伺服自动速度
E1_1602 CHANNEL  ; 侧压A4左伺服JOG高速
E1_1603 CHANNEL  ; 侧压A4左伺服JOG高速
E1_1604 CHANNEL  ; 侧压A4左伺服JOG低速
E1_1605 CHANNEL  ; 侧压A4左伺服JOG低速
E1_1606 CHANNEL  ; 侧压A4左伺服加速时间
E1_1607 CHANNEL  ; 侧压A4左伺服加速时间
E1_1608 CHANNEL  ; 侧压A4左伺服减速时间
E1_1609 CHANNEL  ; 侧压A4左伺服减速时间
E1_161 CHANNEL  ; NC433_2_X轴特殊操作Override
E1_1610 CHANNEL  ; 侧压A4左伺服原点偏移
E1_1611 CHANNEL  ; 侧压A4左伺服原点偏移
E1_1612 CHANNEL  ; 侧压A4左伺服正软极限
E1_1613 CHANNEL  ; 侧压A4左伺服正软极限
E1_1614 CHANNEL  ; 侧压A4左伺服负软极限
E1_1615 CHANNEL  ; 负软极限
E1_162 CHANNEL  ; NC433_2_X轴特殊操作示教地址
E1_1620 CHANNEL  ; 侧压A4左伺服待机位
E1_1621 CHANNEL  ; 侧压A4左伺服待机位
E1_1622 CHANNEL  ; 侧压A4左伺服拨料退回位
E1_1623 CHANNEL  ; 侧压A4左伺服拨料退回位
E1_1624 CHANNEL  ; 侧压A4左伺服拨料位
E1_1625 CHANNEL  ; 侧压A4左伺服拨料位
E1_1626 CHANNEL  ; 侧压A4左伺服减速位
E1_1627 CHANNEL  ; 侧压A4左伺服减速位
E1_1628 CHANNEL  ; 侧压A4左伺服等距热压位
E1_1629 CHANNEL  ; 侧压A4左伺服等距热压位
E1_163 CHANNEL  ; NC433_2_X轴特殊操作预留
E1_1630 CHANNEL  ; 侧压A4左伺服6#位
E1_1631 CHANNEL  ; 侧压A4左伺服6#位
E1_1632 CHANNEL  ; 侧压A4左伺服7#位
E1_1633 CHANNEL  ; 侧压A4左伺服7#位
E1_1634 CHANNEL  ; 侧压A4左伺服8#位
E1_1635 CHANNEL  ; 侧压A4左伺服8#位
E1_1636 CHANNEL  ; 侧压A4左伺服9#位
E1_1637 CHANNEL  ; 侧压A4左伺服9#位
E1_1638 CHANNEL  ; 侧压A4左伺服10#位
E1_1639 CHANNEL  ; 侧压A4左伺服10#位
E1_164 CHANNEL  ; NC433_2_Y轴直接操作位置
E1_1646 CHANNEL  ; A4两轴回原宽度
E1_165 CHANNEL  ; NC433_2_Y轴直接操作位置
E1_1650 CHANNEL  ; 侧压A4右伺服自动速度
E1_1651 CHANNEL  ; 侧压A4右伺服自动速度
E1_1652 CHANNEL  ; 侧压A4右伺服JOG高速
E1_1653 CHANNEL  ; 侧压A4右伺服JOG高速
E1_1654 CHANNEL  ; 侧压A4右伺服JOG低速
E1_1655 CHANNEL  ; 侧压A4右伺服JOG低速
E1_1656 CHANNEL  ; 侧压A4右伺服加速时间
E1_1657 CHANNEL  ; 侧压A4右伺服加速时间
E1_1658 CHANNEL  ; 侧压A4右伺服减速时间
E1_1659 CHANNEL  ; 侧压A4右伺服减速时间
E1_166 CHANNEL  ; NC433_2_Y轴直接操作速度
E1_1660 CHANNEL  ; 侧压A4右伺服原点偏移
E1_1661 CHANNEL  ; 侧压A4右伺服原点偏移
E1_1662 CHANNEL  ; 侧压A4右伺服正软极限
E1_1663 CHANNEL  ; 侧压A4右伺服正软极限
E1_1664 CHANNEL  ; 侧压A4右伺服负软极限
E1_1665 CHANNEL  ; 负软极限
E1_167 CHANNEL  ; NC433_2_Y轴直接操作速度
E1_1670 CHANNEL  ; 侧压A4右伺服待机位
E1_1671 CHANNEL  ; 侧压A4右伺服待机位
E1_1672 CHANNEL  ; 侧压A4右伺服拨料退回位
E1_1673 CHANNEL  ; 侧压A4右伺服拨料退回位
E1_1674 CHANNEL  ; 侧压A4右伺服拨料位
E1_1675 CHANNEL  ; 侧压A4右伺服拨料位
E1_1676 CHANNEL  ; 侧压A4右伺服减速位
E1_1677 CHANNEL  ; 侧压A4右伺服减速位
E1_1678 CHANNEL  ; 侧压A4右伺服等距热压位
E1_1679 CHANNEL  ; 侧压A4右伺服等距热压位
E1_168 CHANNEL  ; NC433_2_Y轴直接操作加速时间
E1_1680 CHANNEL  ; 侧压A4右伺服6#位
E1_1681 CHANNEL  ; 侧压A4右伺服6#位
E1_1682 CHANNEL  ; 侧压A4右伺服7#位
E1_1683 CHANNEL  ; 侧压A4右伺服7#位
E1_1684 CHANNEL  ; 侧压A4右伺服8#位
E1_1685 CHANNEL  ; 侧压A4右伺服8#位
E1_1686 CHANNEL  ; 侧压A4右伺服9#位
E1_1687 CHANNEL  ; 侧压A4右伺服9#位
E1_1688 CHANNEL  ; 侧压A4右伺服10#位
E1_1689 CHANNEL  ; 侧压A4右伺服10#位
E1_169 CHANNEL  ; NC433_2_Y轴直接操作加速时间
E1_17 CHANNEL  ; NC433_0_X轴特殊操作Override
E1_170 CHANNEL  ; NC433_2_Y轴直接操作减速时间
E1_1700 CHANNEL  ; 正压伺服B自动速度
E1_1701 CHANNEL  ; 正压伺服B自动速度
E1_1702 CHANNEL  ; 正压伺服BJOG高速
E1_1703 CHANNEL  ; 正压伺服BJOG高速
E1_1704 CHANNEL  ; 正压伺服BJOG低速
E1_1705 CHANNEL  ; 正压伺服BJOG低速
E1_1706 CHANNEL  ; 正压伺服B加速时间
E1_1707 CHANNEL  ; 正压伺服B加速时间
E1_1708 CHANNEL  ; 正压伺服B减速时间
E1_1709 CHANNEL  ; 正压伺服B减速时间
E1_171 CHANNEL  ; NC433_2_Y轴直接操作减速时间
E1_1710 CHANNEL  ; 正压伺服B原点偏移
E1_1711 CHANNEL  ; 正压伺服B原点偏移
E1_1712 CHANNEL  ; 正压伺服B正软极限
E1_1713 CHANNEL  ; 正压伺服B正软极限
E1_1714 CHANNEL  ; 正压伺服B负软极限
E1_1715 CHANNEL  ; 负软极限
E1_1718 CHANNEL  ; 正压伺服B动态减速位
E1_172 CHANNEL  ; NC433_2_Y轴存储器操作序列号
E1_1720 CHANNEL  ; 正压伺服B初始位
E1_1721 CHANNEL  ; 正压伺服B初始位
E1_1722 CHANNEL  ; 正压B标准减速位
E1_1723 CHANNEL  ; 正压伺服B减速位
E1_1724 CHANNEL  ; 正压伺服B等距热压位
E1_1725 CHANNEL  ; 正压伺服B等距热压位
E1_1726 CHANNEL  ; 正压伺服B预压退回位
E1_1727 CHANNEL  ; 正压伺服B预压退回位
E1_1728 CHANNEL  ; 正压伺服BMASK测试位
E1_1729 CHANNEL  ; 正压伺服BMASK测试位
E1_173 CHANNEL  ; NC433_2_Y轴特殊操作Override
E1_1730 CHANNEL  ; 正压伺服B6#位
E1_1731 CHANNEL  ; 正压伺服B6#位
E1_1732 CHANNEL  ; 正压伺服B7#位
E1_1733 CHANNEL  ; 正压伺服B7#位
E1_1734 CHANNEL  ; 正压伺服B8#位
E1_1735 CHANNEL  ; 正压伺服B8#位
E1_1736 CHANNEL  ; 正压伺服B9#位
E1_1737 CHANNEL  ; 正压伺服B9#位
E1_1738 CHANNEL  ; 正压伺服B10#位
E1_1739 CHANNEL  ; 正压伺服B10#位
E1_174 CHANNEL  ; NC433_2_Y轴特殊操作示教地址
E1_1746 CHANNEL  ; B工位无料偏差
E1_175 CHANNEL  ; NC433_2_Y轴特殊操作预留
E1_1750 CHANNEL  ; 压板平移伺服B自动速度
E1_1751 CHANNEL  ; 压板平移伺服B自动速度
E1_1752 CHANNEL  ; 压板平移伺服BJOG高速
E1_1753 CHANNEL  ; 压板平移伺服BJOG高速
E1_1754 CHANNEL  ; 压板平移伺服BJOG低速
E1_1755 CHANNEL  ; 压板平移伺服BJOG低速
E1_1756 CHANNEL  ; 压板平移伺服B加速时间
E1_1757 CHANNEL  ; 压板平移伺服B加速时间
E1_1758 CHANNEL  ; 压板平移伺服B减速时间
E1_1759 CHANNEL  ; 压板平移伺服B减速时间
E1_176 CHANNEL  ; NC433_2_Z轴直接操作位置
E1_1760 CHANNEL  ; 压板平移伺服B原点偏移
E1_1761 CHANNEL  ; 压板平移伺服B原点偏移
E1_1762 CHANNEL  ; 压板平移伺服B正软极限
E1_1763 CHANNEL  ; 压板平移伺服B正软极限
E1_1764 CHANNEL  ; 压板平移伺服B负软极限
E1_1765 CHANNEL  ; 负软极限
E1_177 CHANNEL  ; NC433_2_Z轴直接操作位置
E1_1770 CHANNEL  ; 压板平移伺服BA面取放位
E1_1771 CHANNEL  ; 压板平移伺服BA面取放位
E1_1772 CHANNEL  ; 压板平移伺服BB面取放位
E1_1773 CHANNEL  ; 压板平移伺服BB面取放位
E1_1774 CHANNEL  ; 压板平移伺服B3#位
E1_1775 CHANNEL  ; 压板平移伺服B3#位
E1_1776 CHANNEL  ; 压板平移伺服B4#位
E1_1777 CHANNEL  ; 压板平移伺服B4#位
E1_1778 CHANNEL  ; 压板平移伺服B5#位
E1_1779 CHANNEL  ; 压板平移伺服B5#位
E1_178 CHANNEL  ; NC433_2_Z轴直接操作速度
E1_1780 CHANNEL  ; 压板平移伺服B6#位
E1_1781 CHANNEL  ; 压板平移伺服B6#位
E1_1782 CHANNEL  ; 压板平移伺服B7#位
E1_1783 CHANNEL  ; 压板平移伺服B7#位
E1_1784 CHANNEL  ; 压板平移伺服B8#位
E1_1785 CHANNEL  ; 压板平移伺服B8#位
E1_1786 CHANNEL  ; 压板平移伺服B9#位
E1_1787 CHANNEL  ; 压板平移伺服B9#位
E1_1788 CHANNEL  ; 压板平移伺服B10#位
E1_1789 CHANNEL  ; 压板平移伺服B10#位
E1_179 CHANNEL  ; NC433_2_Z轴直接操作速度
E1_18 CHANNEL  ; NC433_0_X轴特殊操作示教地址
E1_180 CHANNEL  ; NC433_2_Z轴直接操作加速时间
E1_1800 CHANNEL  ; 侧压B1左伺服自动速度
E1_1801 CHANNEL  ; 侧压B1左伺服自动速度
E1_1802 CHANNEL  ; 侧压B1左伺服JOG高速
E1_1803 CHANNEL  ; 侧压B1左伺服JOG高速
E1_1804 CHANNEL  ; 侧压B1左伺服JOG低速
E1_1805 CHANNEL  ; 侧压B1左伺服JOG低速
E1_1806 CHANNEL  ; 侧压B1左伺服加速时间
E1_1807 CHANNEL  ; 侧压B1左伺服加速时间
E1_1808 CHANNEL  ; 侧压B1左伺服减速时间
E1_1809 CHANNEL  ; 侧压B1左伺服减速时间
E1_181 CHANNEL  ; NC433_2_Z轴直接操作加速时间
E1_1810 CHANNEL  ; 侧压B1左伺服原点偏移
E1_1811 CHANNEL  ; 侧压B1左伺服原点偏移
E1_1812 CHANNEL  ; 侧压B1左伺服正软极限
E1_1813 CHANNEL  ; 侧压B1左伺服正软极限
E1_1814 CHANNEL  ; 侧压B1左伺服负软极限
E1_1815 CHANNEL  ; 负软极限
E1_182 CHANNEL  ; NC433_2_Z轴直接操作减速时间
E1_1820 CHANNEL  ; 侧压B1左伺服待机位
E1_1821 CHANNEL  ; 侧压B1左伺服待机位
E1_1822 CHANNEL  ; 侧压B1左伺服拨料退回位
E1_1823 CHANNEL  ; 侧压B1左伺服拨料退回位
E1_1824 CHANNEL  ; 侧压B1左伺服拨料位
E1_1825 CHANNEL  ; 侧压B1左伺服拨料位
E1_1826 CHANNEL  ; 侧压B1左伺服减速位
E1_1827 CHANNEL  ; 侧压B1左伺服减速位
E1_1828 CHANNEL  ; 侧压B1左伺服等距热压位
E1_1829 CHANNEL  ; 侧压B1左伺服等距热压位
E1_183 CHANNEL  ; NC433_2_Z轴直接操作减速时间
E1_1830 CHANNEL  ; 侧压B1左伺服6#位
E1_1831 CHANNEL  ; 侧压B1左伺服6#位
E1_1832 CHANNEL  ; 侧压B1左伺服7#位
E1_1833 CHANNEL  ; 侧压B1左伺服7#位
E1_1834 CHANNEL  ; 侧压B1左伺服8#位
E1_1835 CHANNEL  ; 侧压B1左伺服8#位
E1_1836 CHANNEL  ; 侧压B1左伺服9#位
E1_1837 CHANNEL  ; 侧压B1左伺服9#位
E1_1838 CHANNEL  ; 侧压B1左伺服10#位
E1_1839 CHANNEL  ; 侧压B1左伺服10#位
E1_184 CHANNEL  ; NC433_2_Z轴存储器操作序列号
E1_1846 CHANNEL  ; B1两轴回原宽度
E1_185 CHANNEL  ; NC433_2_Z轴特殊操作Override
E1_1850 CHANNEL  ; 侧压B1右伺服自动速度
E1_1851 CHANNEL  ; 侧压B1右伺服自动速度
E1_1852 CHANNEL  ; 侧压B1右伺服JOG高速
E1_1853 CHANNEL  ; 侧压B1右伺服JOG高速
E1_1854 CHANNEL  ; 侧压B1右伺服JOG低速
E1_1855 CHANNEL  ; 侧压B1右伺服JOG低速
E1_1856 CHANNEL  ; 侧压B1右伺服加速时间
E1_1857 CHANNEL  ; 侧压B1右伺服加速时间
E1_1858 CHANNEL  ; 侧压B1右伺服减速时间
E1_1859 CHANNEL  ; 侧压B1右伺服减速时间
E1_186 CHANNEL  ; NC433_2_Z轴特殊操作示教地址
E1_1860 CHANNEL  ; 侧压B1右伺服原点偏移
E1_1861 CHANNEL  ; 侧压B1右伺服原点偏移
E1_1862 CHANNEL  ; 侧压B1右伺服正软极限
E1_1863 CHANNEL  ; 侧压B1右伺服正软极限
E1_1864 CHANNEL  ; 侧压B1右伺服负软极限
E1_1865 CHANNEL  ; 负软极限
E1_187 CHANNEL  ; NC433_2_Z轴特殊操作预留
E1_1870 CHANNEL  ; 侧压B1右伺服待机位
E1_1871 CHANNEL  ; 侧压B1右伺服待机位
E1_1872 CHANNEL  ; 侧压B1右伺服拨料退回位
E1_1873 CHANNEL  ; 侧压B1右伺服拨料退回位
E1_1874 CHANNEL  ; 侧压B1右伺服拨料位
E1_1875 CHANNEL  ; 侧压B1右伺服拨料位
E1_1876 CHANNEL  ; 侧压B1右伺服减速位
E1_1877 CHANNEL  ; 侧压B1右伺服减速位
E1_1878 CHANNEL  ; 侧压B1右伺服等距热压位
E1_1879 CHANNEL  ; 侧压B1右伺服等距热压位
E1_188 CHANNEL  ; NC433_2_U轴直接操作位置
E1_1880 CHANNEL  ; 侧压B1右伺服6#位
E1_1881 CHANNEL  ; 侧压B1右伺服6#位
E1_1882 CHANNEL  ; 侧压B1右伺服7#位
E1_1883 CHANNEL  ; 侧压B1右伺服7#位
E1_1884 CHANNEL  ; 侧压B1右伺服8#位
E1_1885 CHANNEL  ; 侧压B1右伺服8#位
E1_1886 CHANNEL  ; 侧压B1右伺服9#位
E1_1887 CHANNEL  ; 侧压B1右伺服9#位
E1_1888 CHANNEL  ; 侧压B1右伺服10#位
E1_1889 CHANNEL  ; 侧压B1右伺服10#位
E1_189 CHANNEL  ; NC433_2_U轴直接操作位置
E1_19 CHANNEL  ; NC433_0_X轴特殊操作预留
E1_190 CHANNEL  ; NC433_2_U轴直接操作速度
E1_1900 CHANNEL  ; 侧压B2左伺服自动速度
E1_1901 CHANNEL  ; 侧压B2左伺服自动速度
E1_1902 CHANNEL  ; 侧压B2左伺服JOG高速
E1_1903 CHANNEL  ; 侧压B2左伺服JOG高速
E1_1904 CHANNEL  ; 侧压B2左伺服JOG低速
E1_1905 CHANNEL  ; 侧压B2左伺服JOG低速
E1_1906 CHANNEL  ; 侧压B2左伺服加速时间
E1_1907 CHANNEL  ; 侧压B2左伺服加速时间
E1_1908 CHANNEL  ; 侧压B2左伺服减速时间
E1_1909 CHANNEL  ; 侧压B2左伺服减速时间
E1_191 CHANNEL  ; NC433_2_U轴直接操作速度
E1_1910 CHANNEL  ; 侧压B2左伺服原点偏移
E1_1911 CHANNEL  ; 侧压B2左伺服原点偏移
E1_1912 CHANNEL  ; 侧压B2左伺服正软极限
E1_1913 CHANNEL  ; 侧压B2左伺服正软极限
E1_1914 CHANNEL  ; 侧压B2左伺服负软极限
E1_1915 CHANNEL  ; 负软极限
E1_192 CHANNEL  ; NC433_2_U轴直接操作加速时间
E1_1920 CHANNEL  ; 侧压B2左伺服待机位
E1_1921 CHANNEL  ; 侧压B2左伺服待机位
E1_1922 CHANNEL  ; 侧压B2左伺服拨料退回位
E1_1923 CHANNEL  ; 侧压B2左伺服拨料退回位
E1_1924 CHANNEL  ; 侧压B2左伺服拨料位
E1_1925 CHANNEL  ; 侧压B2左伺服拨料位
E1_1926 CHANNEL  ; 侧压B2左伺服减速位
E1_1927 CHANNEL  ; 侧压B2左伺服减速位
E1_1928 CHANNEL  ; 侧压B2左伺服等距热压位
E1_1929 CHANNEL  ; 侧压B2左伺服等距热压位
E1_193 CHANNEL  ; NC433_2_U轴直接操作加速时间
E1_1930 CHANNEL  ; 侧压B2左伺服6#位
E1_1931 CHANNEL  ; 侧压B2左伺服6#位
E1_1932 CHANNEL  ; 侧压B2左伺服7#位
E1_1933 CHANNEL  ; 侧压B2左伺服7#位
E1_1934 CHANNEL  ; 侧压B2左伺服8#位
E1_1935 CHANNEL  ; 侧压B2左伺服8#位
E1_1936 CHANNEL  ; 侧压B2左伺服9#位
E1_1937 CHANNEL  ; 侧压B2左伺服9#位
E1_1938 CHANNEL  ; 侧压B2左伺服10#位
E1_1939 CHANNEL  ; 侧压B2左伺服10#位
E1_194 CHANNEL  ; NC433_2_U轴直接操作减速时间
E1_1946 CHANNEL  ; B2两轴回原宽度
E1_195 CHANNEL  ; NC433_2_U轴直接操作减速时间
E1_1950 CHANNEL  ; 侧压B2右伺服自动速度
E1_1951 CHANNEL  ; 侧压B2右伺服自动速度
E1_1952 CHANNEL  ; 侧压B2右伺服JOG高速
E1_1953 CHANNEL  ; 侧压B2右伺服JOG高速
E1_1954 CHANNEL  ; 侧压B2右伺服JOG低速
E1_1955 CHANNEL  ; 侧压B2右伺服JOG低速
E1_1956 CHANNEL  ; 侧压B2右伺服加速时间
E1_1957 CHANNEL  ; 侧压B2右伺服加速时间
E1_1958 CHANNEL  ; 侧压B2右伺服减速时间
E1_1959 CHANNEL  ; 侧压B2右伺服减速时间
E1_196 CHANNEL  ; NC433_2_U轴存储器操作序列号
E1_1960 CHANNEL  ; 侧压B2右伺服原点偏移
E1_1961 CHANNEL  ; 侧压B2右伺服原点偏移
E1_1962 CHANNEL  ; 侧压B2右伺服正软极限
E1_1963 CHANNEL  ; 侧压B2右伺服正软极限
E1_1964 CHANNEL  ; 侧压B2右伺服负软极限
E1_1965 CHANNEL  ; 负软极限
E1_197 CHANNEL  ; NC433_2_U轴特殊操作Override
E1_1970 CHANNEL  ; 侧压B2右伺服待机位
E1_1971 CHANNEL  ; 侧压B2右伺服待机位
E1_1972 CHANNEL  ; 侧压B2右伺服拨料退回位
E1_1973 CHANNEL  ; 侧压B2右伺服拨料退回位
E1_1974 CHANNEL  ; 侧压B2右伺服拨料位
E1_1975 CHANNEL  ; 侧压B2右伺服拨料位
E1_1976 CHANNEL  ; 侧压B2右伺服减速位
E1_1977 CHANNEL  ; 侧压B2右伺服减速位
E1_1978 CHANNEL  ; 侧压B2右伺服等距热压位
E1_1979 CHANNEL  ; 侧压B2右伺服等距热压位
E1_198 CHANNEL  ; NC433_2_U轴特殊操作示教地址
E1_1980 CHANNEL  ; 侧压B2右伺服6#位
E1_1981 CHANNEL  ; 侧压B2右伺服6#位
E1_1982 CHANNEL  ; 侧压B2右伺服7#位
E1_1983 CHANNEL  ; 侧压B2右伺服7#位
E1_1984 CHANNEL  ; 侧压B2右伺服8#位
E1_1985 CHANNEL  ; 侧压B2右伺服8#位
E1_1986 CHANNEL  ; 侧压B2右伺服9#位
E1_1987 CHANNEL  ; 侧压B2右伺服9#位
E1_1988 CHANNEL  ; 侧压B2右伺服10#位
E1_1989 CHANNEL  ; 侧压B2右伺服10#位
E1_199 CHANNEL  ; NC433_2_U轴特殊操作预留
E1_2 CHANNEL  ; NC433_0 数据传送定源字
E1_20 CHANNEL  ; NC433_0_Y轴直接操作位置
E1_200 CHANNEL  ; NC433_2_X轴当前位置
E1_2000 CHANNEL  ; 侧压B3左伺服自动速度
E1_2001 CHANNEL  ; 侧压B3左伺服自动速度
E1_2002 CHANNEL  ; 侧压B3左伺服JOG高速
E1_2003 CHANNEL  ; 侧压B3左伺服JOG高速
